// TIA Portal V17 export
// export: Created 2025-03-07T09:17:06.8122535Z, ExportSetting WithDefaults, DisplayName Totally Integrated Automation Portal, DisplayVersion V17 Update 8, DisplayName TIA Portal Openness, DisplayVersion V17 Update 8, DisplayName TIA Portal Version Control Interface, DisplayVersion V17, DisplayName SINAMICS Startdrive Advanced, DisplayVersion V17 SP2, DisplayName SINAMICS Startdrive G110M, G120, G120C, G120D, G120P, G115D, DisplayVersion V17 SP2, DisplayName SINAMICS Startdrive G130, G150, S120, S150, SINAMICS MV, S210, DisplayVersion V17 SP2, DisplayName STEP 7 Professional, DisplayVersion V17 Update 8, DisplayName SINUMERIK ONE STEP 7 Toolbox, DisplayVersion V17 Update 12, DisplayName SINUMERIK 840D sl STEP 7 Toolbox, DisplayVersion V17 Update 12, DisplayName STEP 7 Safety, DisplayVersion V17 Update 6, DisplayName WinCC Advanced, DisplayVersion V17 Update 8
FUNCTION "FC8002_UNIT_01_CLADDING" : Void   // FC8002, LAD
{ S7_Optimized_Access := 'FALSE' }
AUTHOR : ETXETAR
VERSION : 1.0
// stored: AutoNumber false, IsIECCheckEnabled false, SetENOAutomatically false, UDAEnableTagReadback false
   VAR_TEMP
      ZERO : Byte;   // ZERO
      STATUS_BLKMOV : Int;   // STATUS BLKMOV
      STATUS_FILL : Int;   // STATUS FILL
      aux_string : String;
      Cnt_Chars : Int;
      Chars_Array : Array[0..63] of Char;
   END_VAR
   VAR CONSTANT
      FC_NUMBER : DInt := 8002;   // FC NUMBER
   END_VAR
   VAR_TEMP   // added for the SCL form of the ladder/FBD networks
      _w1 : Bool;
      _w2 : Bool;
      _w3 : Bool;
      _w4 : Bool;
      _w5 : Bool;
      _w6 : Bool;
      _w7 : Bool;
      _w8 : Bool;
      _w9 : Bool;
   END_VAR
BEGIN

REGION Network 1: ZERO
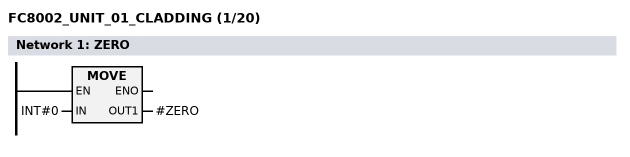
   RUNG wire#powerrail
      { S7_GenerateENO := "TRUE" } Move(in := INT#0, out1 => #ZERO)
   END_RUNG
   // the same network as SCL:
   #ZERO := INT#0;
END_REGION

REGION Network 2: HMI MANUAL PART A FIXTURE 1, 2, 3, 4 STATUS
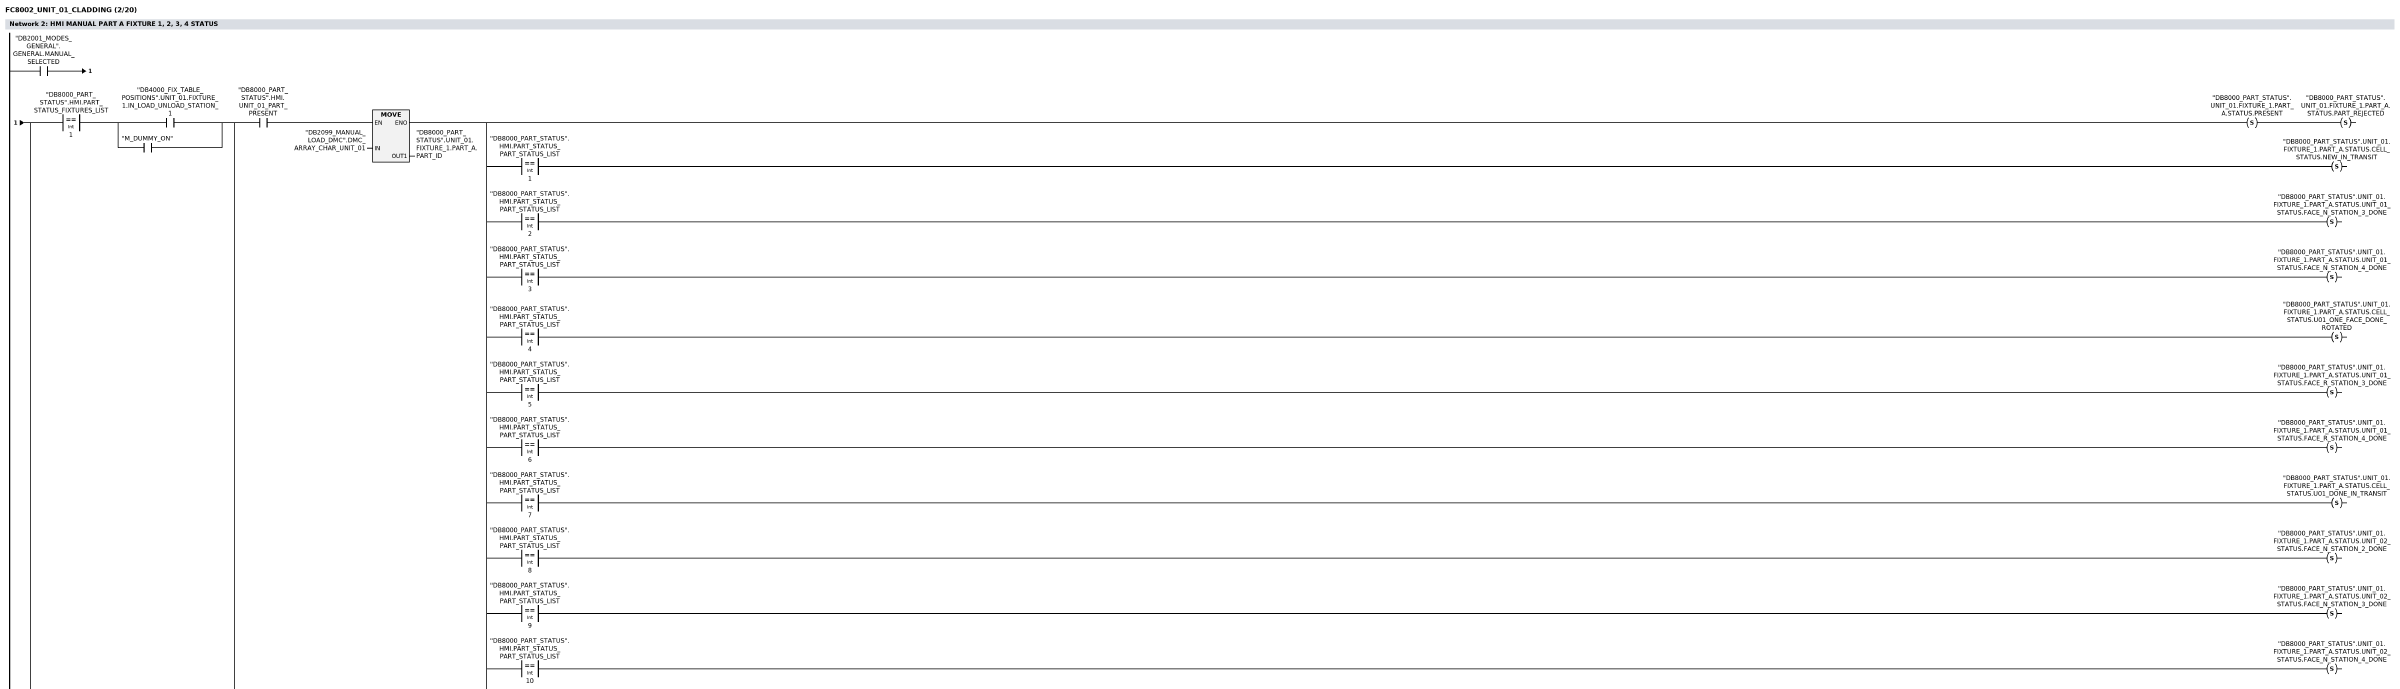
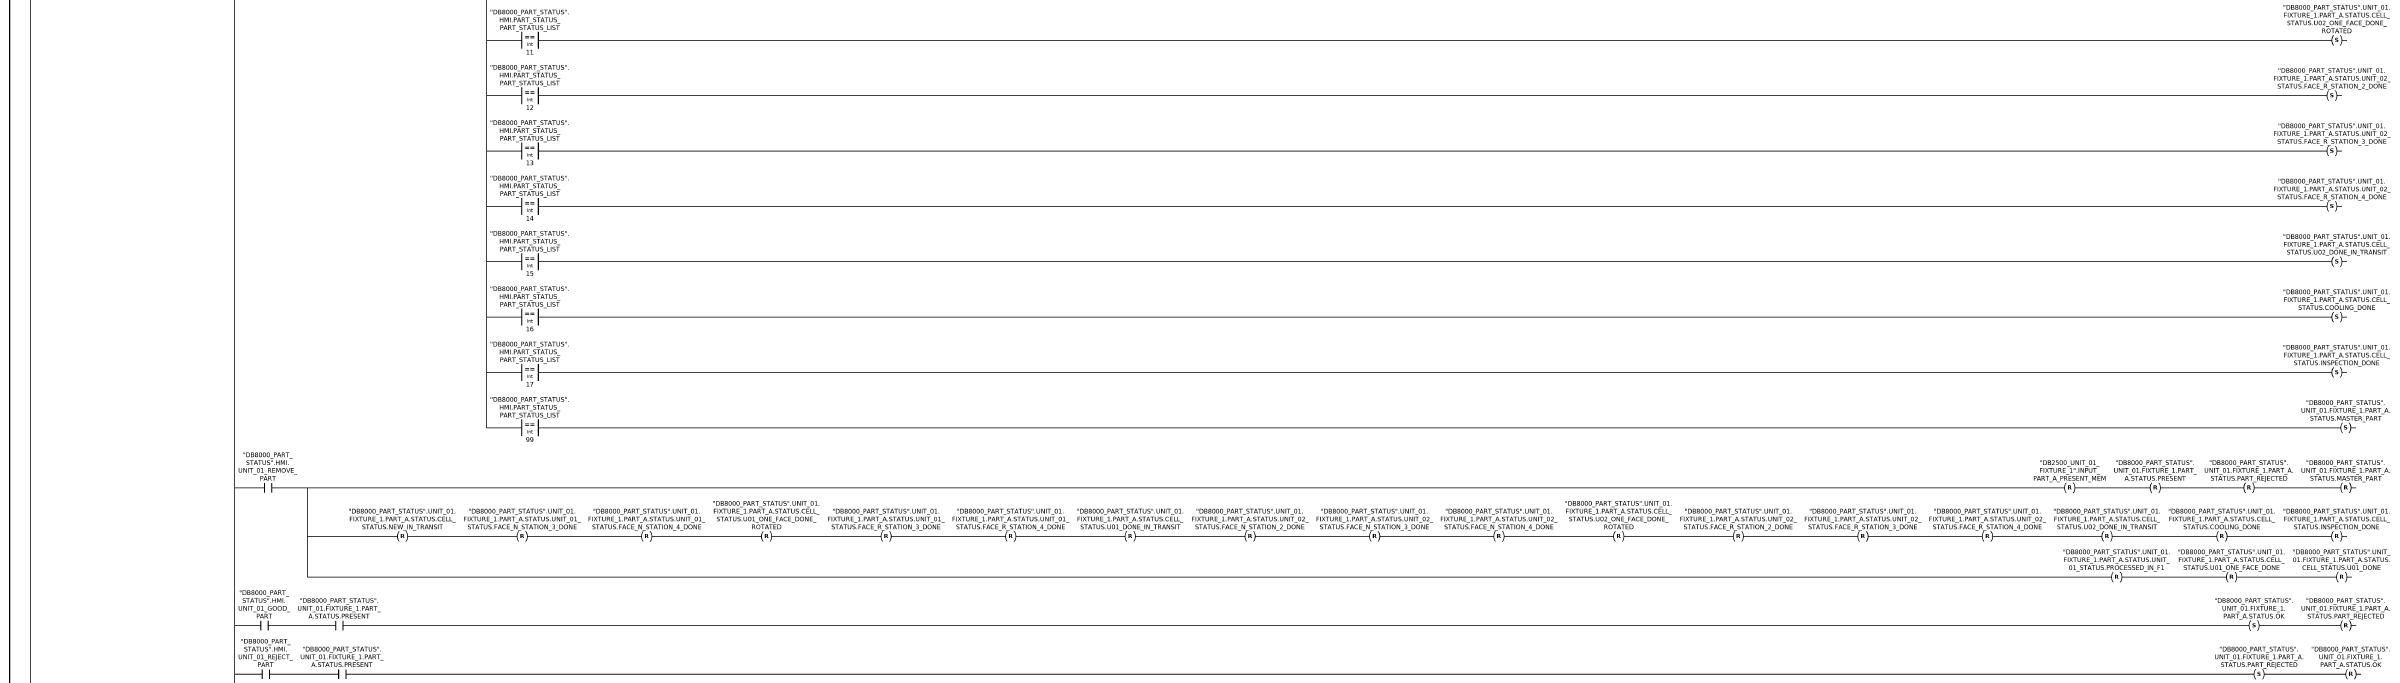
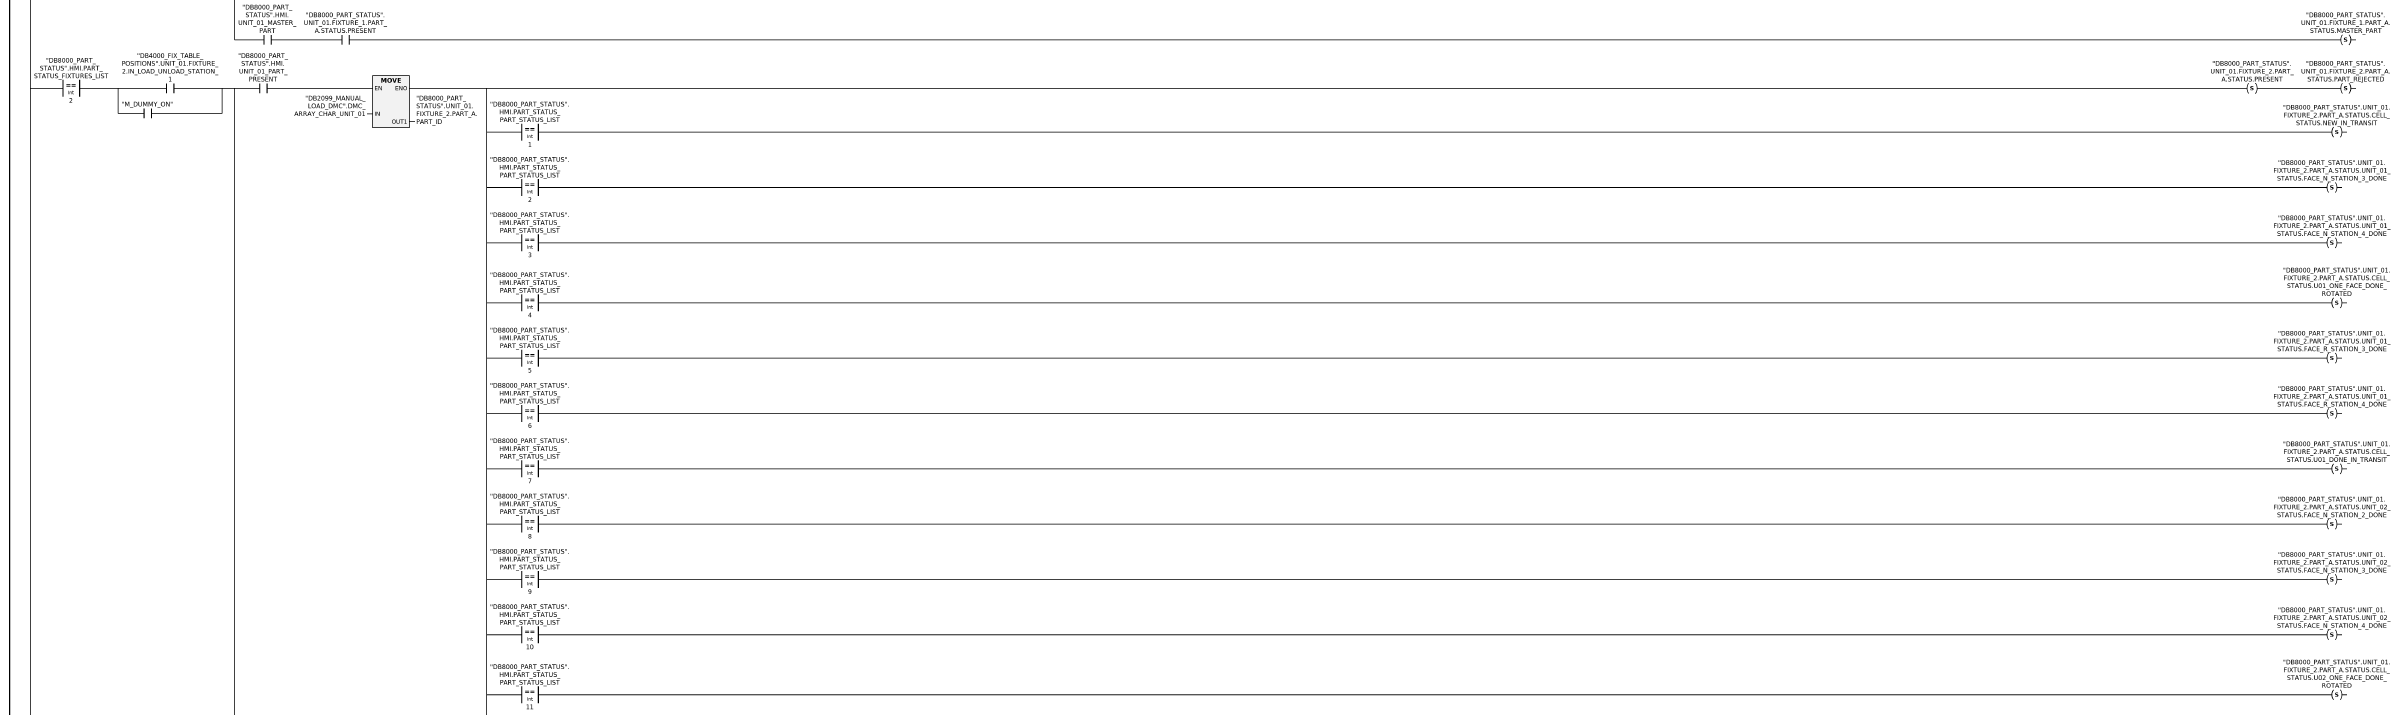
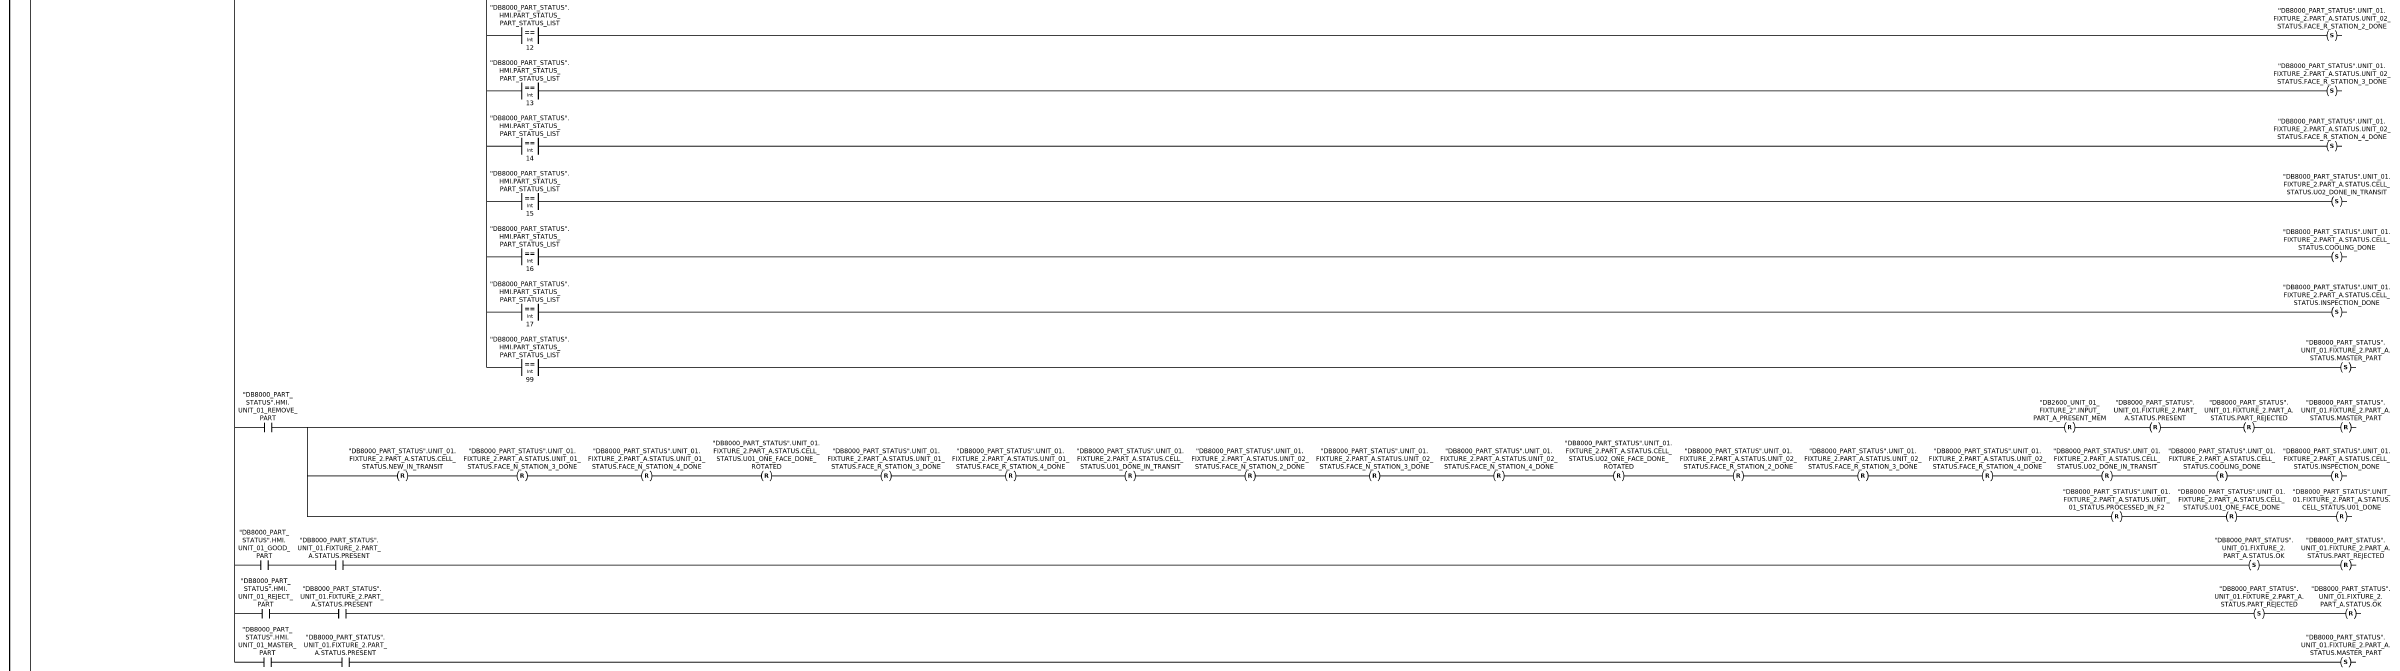
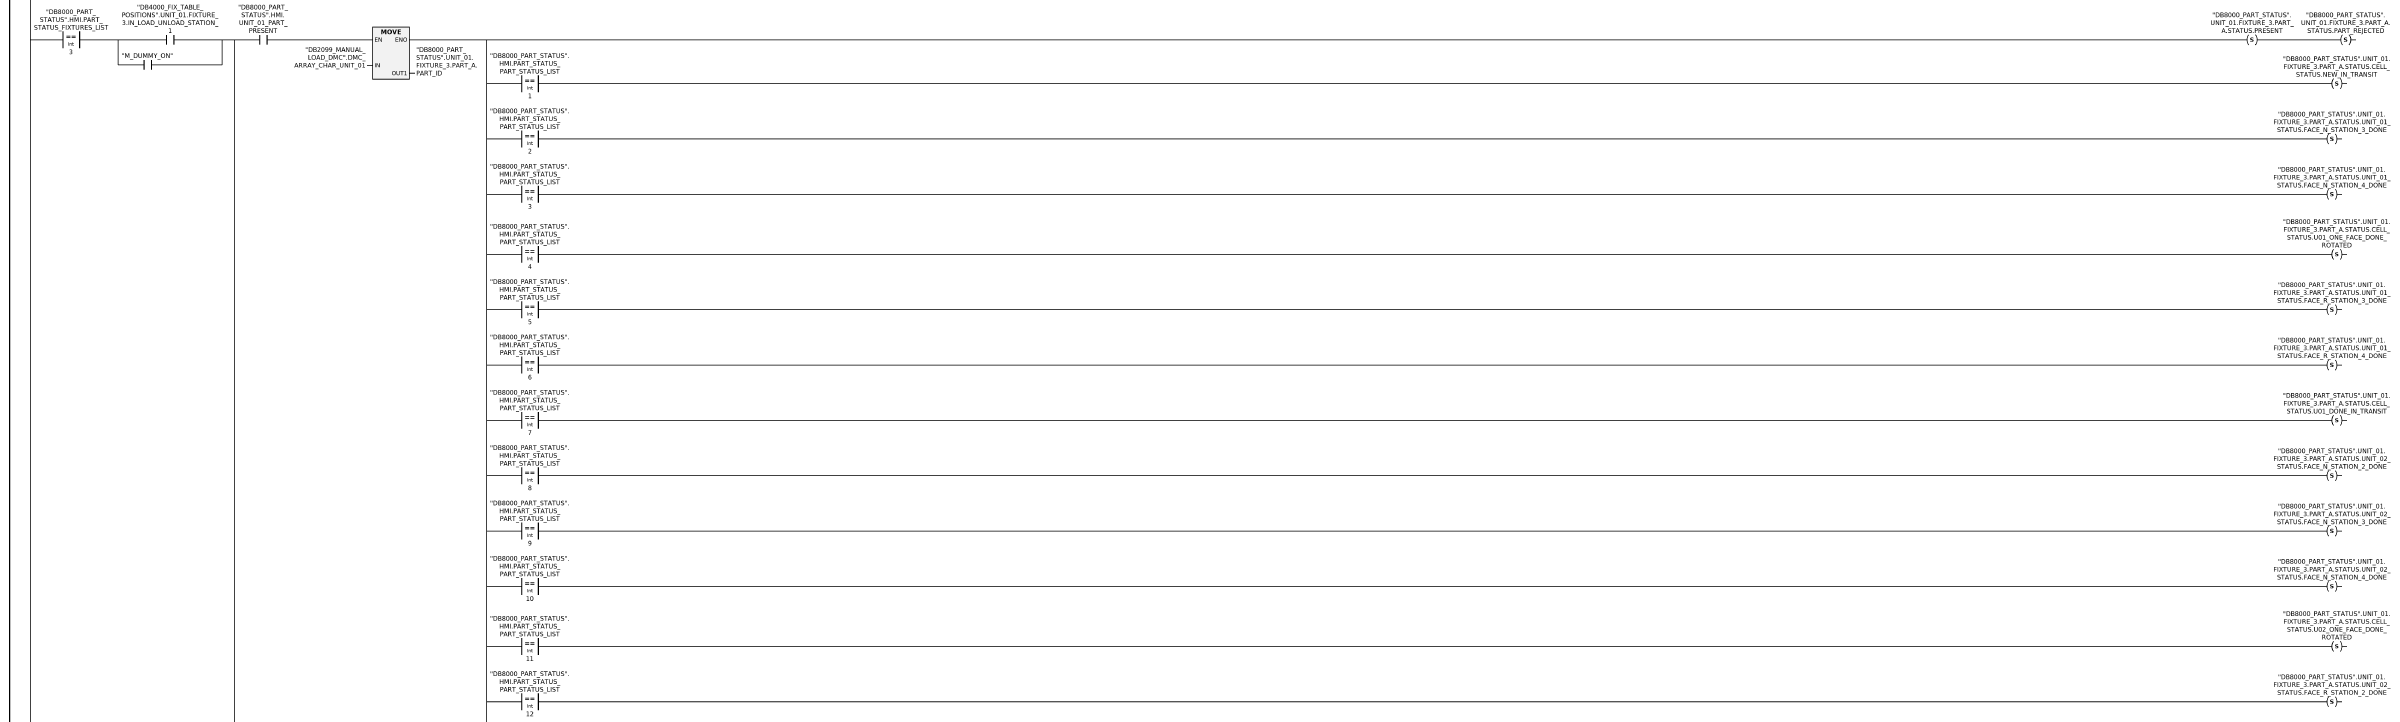
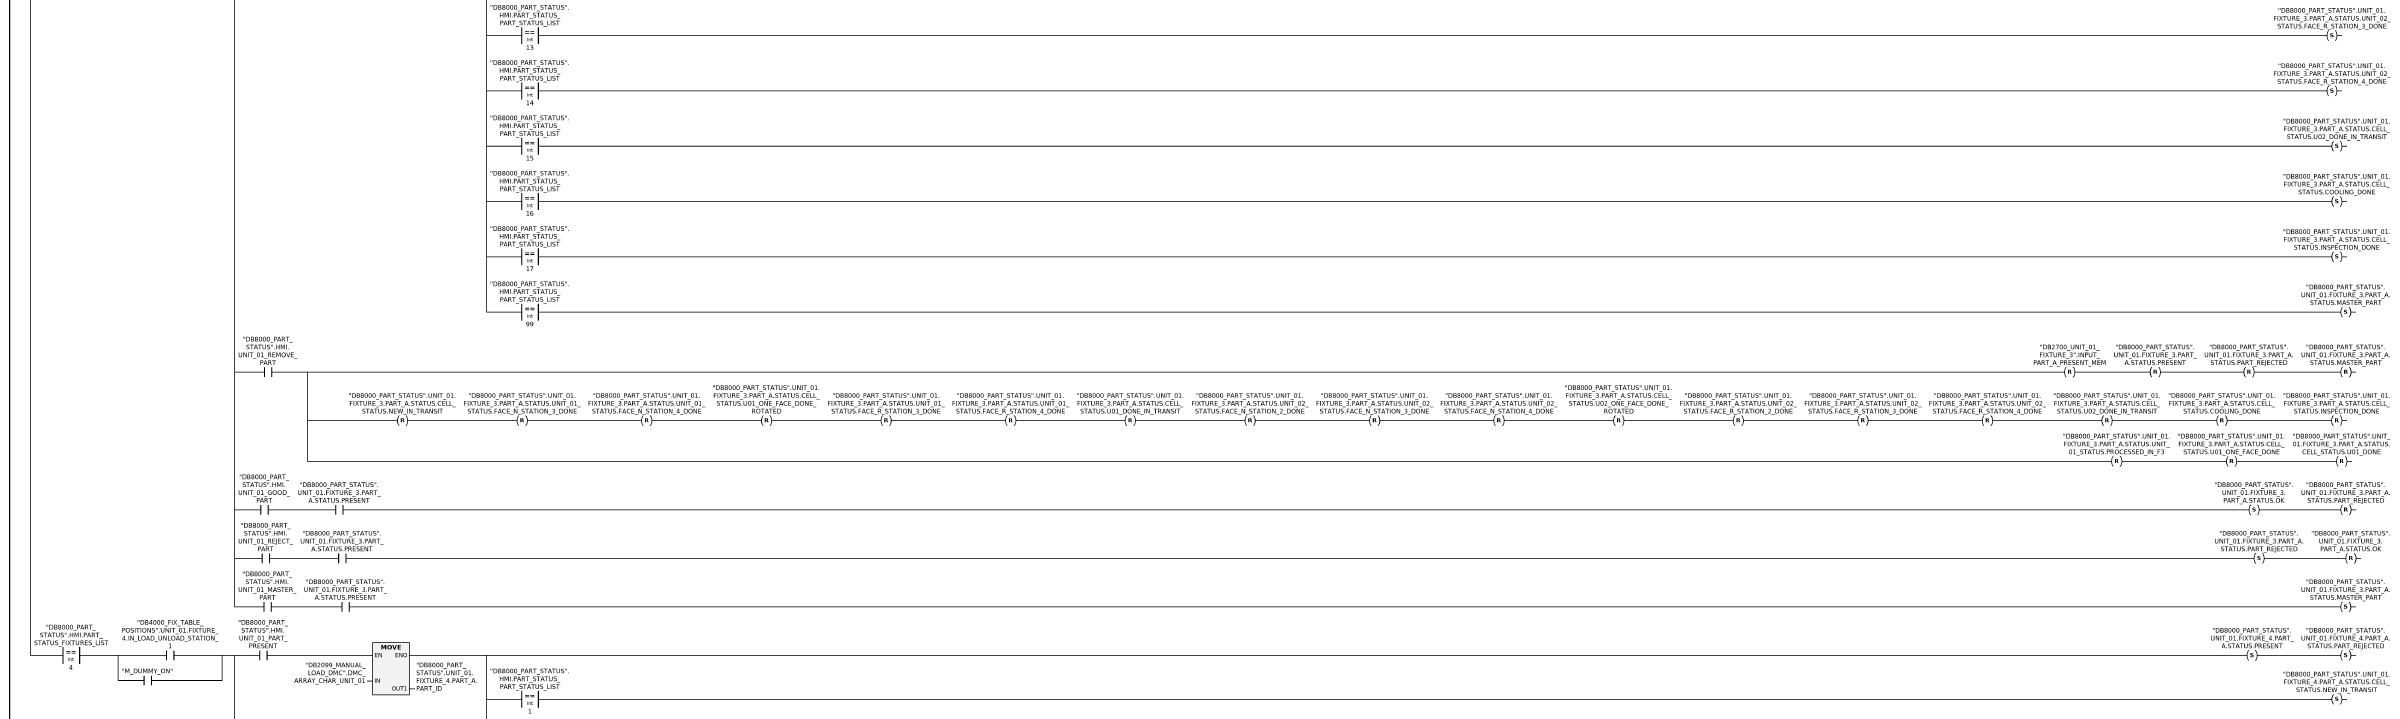
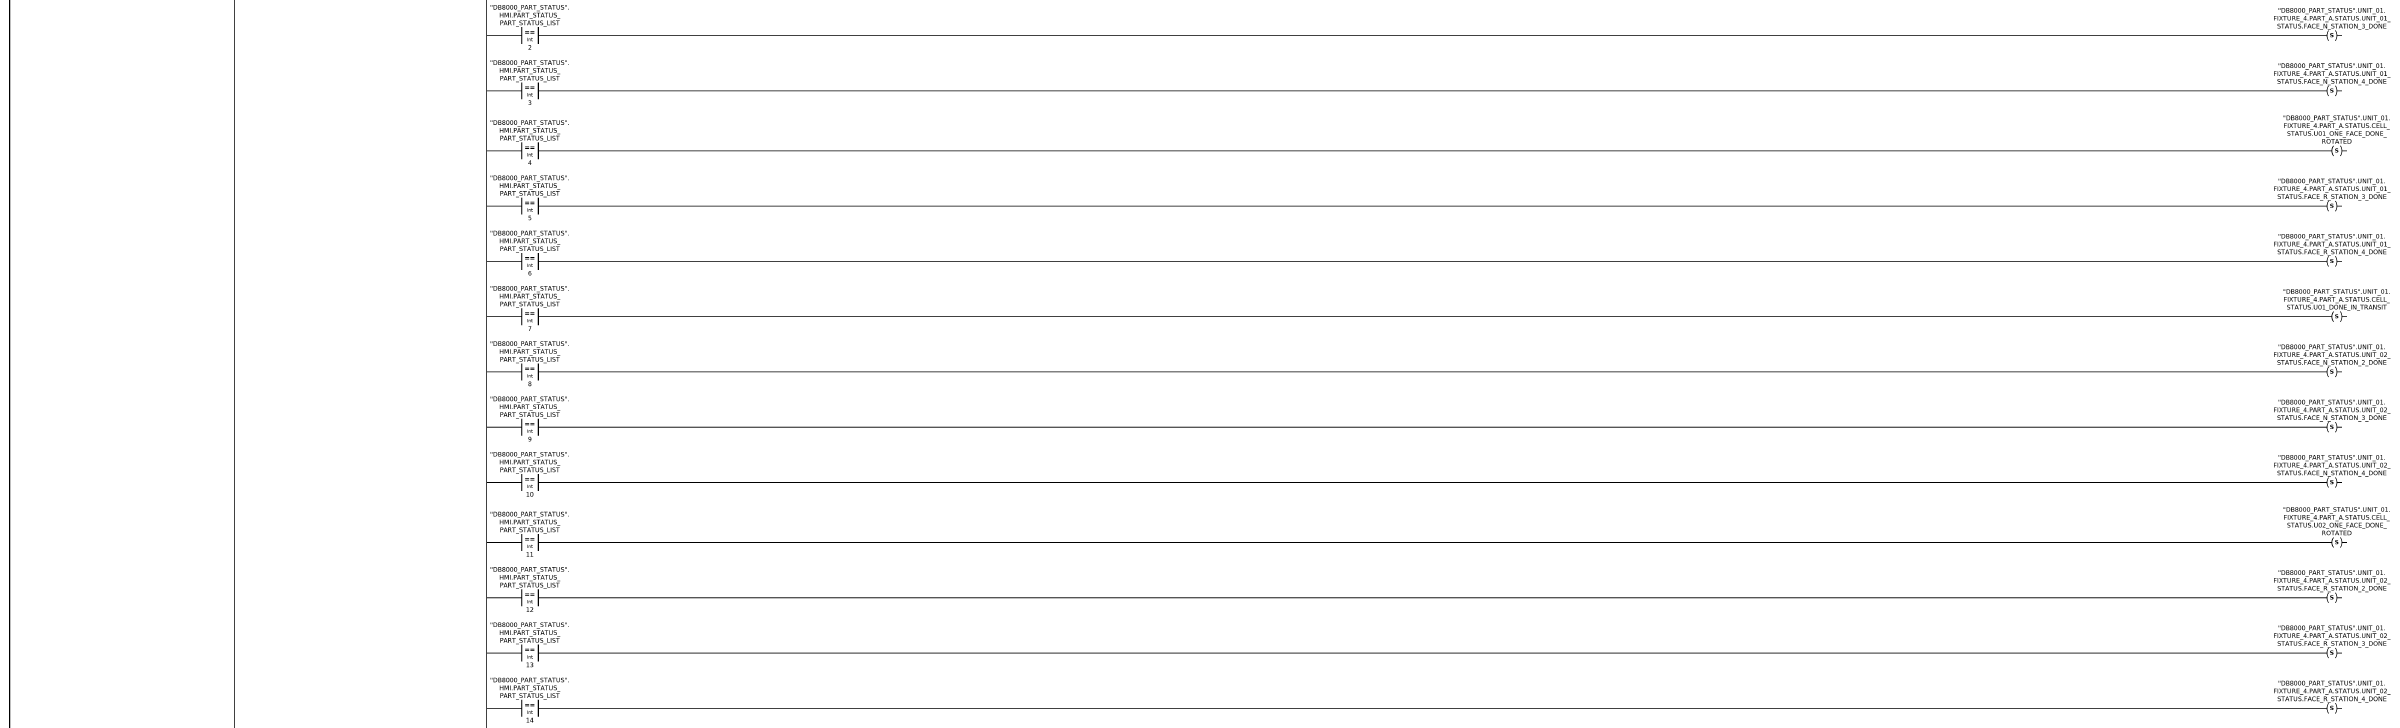
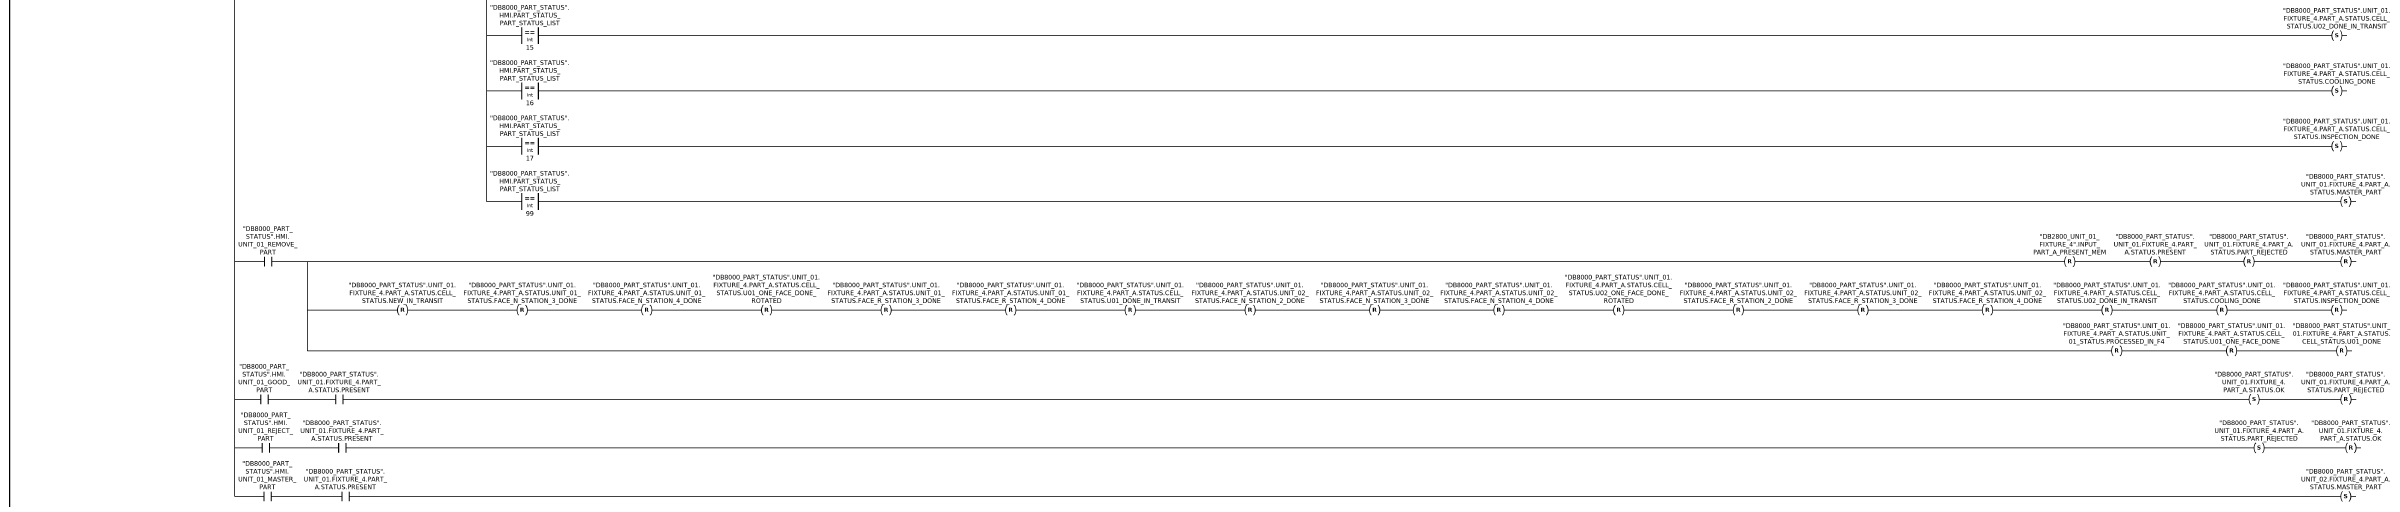
   RUNG wire#powerrail
      Contact( "DB2001_MODES_GENERAL".GENERAL.MANUAL_SELECTED )
      wire#w1
      { S7_Templates := "SrcType := Int" } EQ_Contact(in1 := "DB8000_PART_STATUS".HMI.PART_STATUS_FIXTURES_LIST, in2 := 1)
      wire#w2
      Contact( "DB4000_FIX_TABLE_POSITIONS".UNIT_01.FIXTURE_1.IN_LOAD_UNLOAD_STATION_1 )
      wire#w3
      Contact( "DB8000_PART_STATUS".HMI.UNIT_01_PART_PRESENT )
      Move(in := "DB2099_MANUAL_LOAD_DMC".DMC_ARRAY_CHAR_UNIT_01, out1 => "DB8000_PART_STATUS".UNIT_01.FIXTURE_1.PART_A.PART_ID)
      wire#w4
      S_Coil( "DB8000_PART_STATUS".UNIT_01.FIXTURE_1.PART_A.STATUS.PRESENT )
      S_Coil( "DB8000_PART_STATUS".UNIT_01.FIXTURE_1.PART_A.STATUS.PART_REJECTED )
   END_RUNG
   RUNG wire#w2
      Contact( "M_DUMMY_ON" )
   END_RUNG wire#w3
   RUNG wire#w4
      { S7_Templates := "SrcType := Int" } EQ_Contact(in1 := "DB8000_PART_STATUS".HMI.PART_STATUS_PART_STATUS_LIST, in2 := 1)
      S_Coil( "DB8000_PART_STATUS".UNIT_01.FIXTURE_1.PART_A.STATUS.CELL_STATUS.NEW_IN_TRANSIT )
   END_RUNG
   RUNG wire#w4
      { S7_Templates := "SrcType := Int" } EQ_Contact(in1 := "DB8000_PART_STATUS".HMI.PART_STATUS_PART_STATUS_LIST, in2 := 2)
      S_Coil( "DB8000_PART_STATUS".UNIT_01.FIXTURE_1.PART_A.STATUS.UNIT_01_STATUS.FACE_N_STATION_3_DONE )
   END_RUNG
   RUNG wire#w4
      { S7_Templates := "SrcType := Int" } EQ_Contact(in1 := "DB8000_PART_STATUS".HMI.PART_STATUS_PART_STATUS_LIST, in2 := 3)
      S_Coil( "DB8000_PART_STATUS".UNIT_01.FIXTURE_1.PART_A.STATUS.UNIT_01_STATUS.FACE_N_STATION_4_DONE )
   END_RUNG
   RUNG wire#w4
      { S7_Templates := "SrcType := Int" } EQ_Contact(in1 := "DB8000_PART_STATUS".HMI.PART_STATUS_PART_STATUS_LIST, in2 := 4)
      S_Coil( "DB8000_PART_STATUS".UNIT_01.FIXTURE_1.PART_A.STATUS.CELL_STATUS.U01_ONE_FACE_DONE_ROTATED )
   END_RUNG
   RUNG wire#w4
      { S7_Templates := "SrcType := Int" } EQ_Contact(in1 := "DB8000_PART_STATUS".HMI.PART_STATUS_PART_STATUS_LIST, in2 := 5)
      S_Coil( "DB8000_PART_STATUS".UNIT_01.FIXTURE_1.PART_A.STATUS.UNIT_01_STATUS.FACE_R_STATION_3_DONE )
   END_RUNG
   RUNG wire#w4
      { S7_Templates := "SrcType := Int" } EQ_Contact(in1 := "DB8000_PART_STATUS".HMI.PART_STATUS_PART_STATUS_LIST, in2 := 6)
      S_Coil( "DB8000_PART_STATUS".UNIT_01.FIXTURE_1.PART_A.STATUS.UNIT_01_STATUS.FACE_R_STATION_4_DONE )
   END_RUNG
   RUNG wire#w4
      { S7_Templates := "SrcType := Int" } EQ_Contact(in1 := "DB8000_PART_STATUS".HMI.PART_STATUS_PART_STATUS_LIST, in2 := 7)
      S_Coil( "DB8000_PART_STATUS".UNIT_01.FIXTURE_1.PART_A.STATUS.CELL_STATUS.U01_DONE_IN_TRANSIT )
   END_RUNG
   RUNG wire#w4
      { S7_Templates := "SrcType := Int" } EQ_Contact(in1 := "DB8000_PART_STATUS".HMI.PART_STATUS_PART_STATUS_LIST, in2 := 8)
      S_Coil( "DB8000_PART_STATUS".UNIT_01.FIXTURE_1.PART_A.STATUS.UNIT_02_STATUS.FACE_N_STATION_2_DONE )
   END_RUNG
   RUNG wire#w4
      { S7_Templates := "SrcType := Int" } EQ_Contact(in1 := "DB8000_PART_STATUS".HMI.PART_STATUS_PART_STATUS_LIST, in2 := 9)
      S_Coil( "DB8000_PART_STATUS".UNIT_01.FIXTURE_1.PART_A.STATUS.UNIT_02_STATUS.FACE_N_STATION_3_DONE )
   END_RUNG
   RUNG wire#w4
      { S7_Templates := "SrcType := Int" } EQ_Contact(in1 := "DB8000_PART_STATUS".HMI.PART_STATUS_PART_STATUS_LIST, in2 := 10)
      S_Coil( "DB8000_PART_STATUS".UNIT_01.FIXTURE_1.PART_A.STATUS.UNIT_02_STATUS.FACE_N_STATION_4_DONE )
   END_RUNG
   RUNG wire#w4
      { S7_Templates := "SrcType := Int" } EQ_Contact(in1 := "DB8000_PART_STATUS".HMI.PART_STATUS_PART_STATUS_LIST, in2 := 11)
      S_Coil( "DB8000_PART_STATUS".UNIT_01.FIXTURE_1.PART_A.STATUS.CELL_STATUS.U02_ONE_FACE_DONE_ROTATED )
   END_RUNG
   RUNG wire#w4
      { S7_Templates := "SrcType := Int" } EQ_Contact(in1 := "DB8000_PART_STATUS".HMI.PART_STATUS_PART_STATUS_LIST, in2 := 12)
      S_Coil( "DB8000_PART_STATUS".UNIT_01.FIXTURE_1.PART_A.STATUS.UNIT_02_STATUS.FACE_R_STATION_2_DONE )
   END_RUNG
   RUNG wire#w4
      { S7_Templates := "SrcType := Int" } EQ_Contact(in1 := "DB8000_PART_STATUS".HMI.PART_STATUS_PART_STATUS_LIST, in2 := 13)
      S_Coil( "DB8000_PART_STATUS".UNIT_01.FIXTURE_1.PART_A.STATUS.UNIT_02_STATUS.FACE_R_STATION_3_DONE )
   END_RUNG
   RUNG wire#w4
      { S7_Templates := "SrcType := Int" } EQ_Contact(in1 := "DB8000_PART_STATUS".HMI.PART_STATUS_PART_STATUS_LIST, in2 := 14)
      S_Coil( "DB8000_PART_STATUS".UNIT_01.FIXTURE_1.PART_A.STATUS.UNIT_02_STATUS.FACE_R_STATION_4_DONE )
   END_RUNG
   RUNG wire#w4
      { S7_Templates := "SrcType := Int" } EQ_Contact(in1 := "DB8000_PART_STATUS".HMI.PART_STATUS_PART_STATUS_LIST, in2 := 15)
      S_Coil( "DB8000_PART_STATUS".UNIT_01.FIXTURE_1.PART_A.STATUS.CELL_STATUS.U02_DONE_IN_TRANSIT )
   END_RUNG
   RUNG wire#w4
      { S7_Templates := "SrcType := Int" } EQ_Contact(in1 := "DB8000_PART_STATUS".HMI.PART_STATUS_PART_STATUS_LIST, in2 := 16)
      S_Coil( "DB8000_PART_STATUS".UNIT_01.FIXTURE_1.PART_A.STATUS.CELL_STATUS.COOLING_DONE )
   END_RUNG
   RUNG wire#w4
      { S7_Templates := "SrcType := Int" } EQ_Contact(in1 := "DB8000_PART_STATUS".HMI.PART_STATUS_PART_STATUS_LIST, in2 := 17)
      S_Coil( "DB8000_PART_STATUS".UNIT_01.FIXTURE_1.PART_A.STATUS.CELL_STATUS.INSPECTION_DONE )
   END_RUNG
   RUNG wire#w4
      { S7_Templates := "SrcType := Int" } EQ_Contact(in1 := "DB8000_PART_STATUS".HMI.PART_STATUS_PART_STATUS_LIST, in2 := 99)
      S_Coil( "DB8000_PART_STATUS".UNIT_01.FIXTURE_1.PART_A.STATUS.MASTER_PART )
   END_RUNG
   RUNG wire#w3
      Contact( "DB8000_PART_STATUS".HMI.UNIT_01_REMOVE_PART )
      wire#w5
      R_Coil( "DB2500_UNIT_01_FIXTURE_1".INPUT_PART_A_PRESENT_MEM )
      R_Coil( "DB8000_PART_STATUS".UNIT_01.FIXTURE_1.PART_A.STATUS.PRESENT )
      R_Coil( "DB8000_PART_STATUS".UNIT_01.FIXTURE_1.PART_A.STATUS.PART_REJECTED )
      R_Coil( "DB8000_PART_STATUS".UNIT_01.FIXTURE_1.PART_A.STATUS.MASTER_PART )
   END_RUNG
   RUNG wire#w5
      R_Coil( "DB8000_PART_STATUS".UNIT_01.FIXTURE_1.PART_A.STATUS.CELL_STATUS.NEW_IN_TRANSIT )
      R_Coil( "DB8000_PART_STATUS".UNIT_01.FIXTURE_1.PART_A.STATUS.UNIT_01_STATUS.FACE_N_STATION_3_DONE )
      R_Coil( "DB8000_PART_STATUS".UNIT_01.FIXTURE_1.PART_A.STATUS.UNIT_01_STATUS.FACE_N_STATION_4_DONE )
      R_Coil( "DB8000_PART_STATUS".UNIT_01.FIXTURE_1.PART_A.STATUS.CELL_STATUS.U01_ONE_FACE_DONE_ROTATED )
      R_Coil( "DB8000_PART_STATUS".UNIT_01.FIXTURE_1.PART_A.STATUS.UNIT_01_STATUS.FACE_R_STATION_3_DONE )
      R_Coil( "DB8000_PART_STATUS".UNIT_01.FIXTURE_1.PART_A.STATUS.UNIT_01_STATUS.FACE_R_STATION_4_DONE )
      R_Coil( "DB8000_PART_STATUS".UNIT_01.FIXTURE_1.PART_A.STATUS.CELL_STATUS.U01_DONE_IN_TRANSIT )
      R_Coil( "DB8000_PART_STATUS".UNIT_01.FIXTURE_1.PART_A.STATUS.UNIT_02_STATUS.FACE_N_STATION_2_DONE )
      R_Coil( "DB8000_PART_STATUS".UNIT_01.FIXTURE_1.PART_A.STATUS.UNIT_02_STATUS.FACE_N_STATION_3_DONE )
      R_Coil( "DB8000_PART_STATUS".UNIT_01.FIXTURE_1.PART_A.STATUS.UNIT_02_STATUS.FACE_N_STATION_4_DONE )
      R_Coil( "DB8000_PART_STATUS".UNIT_01.FIXTURE_1.PART_A.STATUS.CELL_STATUS.U02_ONE_FACE_DONE_ROTATED )
      R_Coil( "DB8000_PART_STATUS".UNIT_01.FIXTURE_1.PART_A.STATUS.UNIT_02_STATUS.FACE_R_STATION_2_DONE )
      R_Coil( "DB8000_PART_STATUS".UNIT_01.FIXTURE_1.PART_A.STATUS.UNIT_02_STATUS.FACE_R_STATION_3_DONE )
      R_Coil( "DB8000_PART_STATUS".UNIT_01.FIXTURE_1.PART_A.STATUS.UNIT_02_STATUS.FACE_R_STATION_4_DONE )
      R_Coil( "DB8000_PART_STATUS".UNIT_01.FIXTURE_1.PART_A.STATUS.CELL_STATUS.U02_DONE_IN_TRANSIT )
      R_Coil( "DB8000_PART_STATUS".UNIT_01.FIXTURE_1.PART_A.STATUS.CELL_STATUS.COOLING_DONE )
      R_Coil( "DB8000_PART_STATUS".UNIT_01.FIXTURE_1.PART_A.STATUS.CELL_STATUS.INSPECTION_DONE )
   END_RUNG
   RUNG wire#w5
      R_Coil( "DB8000_PART_STATUS".UNIT_01.FIXTURE_1.PART_A.STATUS.UNIT_01_STATUS.PROCESSED_IN_F1 )
      R_Coil( "DB8000_PART_STATUS".UNIT_01.FIXTURE_1.PART_A.STATUS.CELL_STATUS.U01_ONE_FACE_DONE )
      R_Coil( "DB8000_PART_STATUS".UNIT_01.FIXTURE_1.PART_A.STATUS.CELL_STATUS.U01_DONE )
   END_RUNG
   RUNG wire#w3
      Contact( "DB8000_PART_STATUS".HMI.UNIT_01_GOOD_PART )
      Contact( "DB8000_PART_STATUS".UNIT_01.FIXTURE_1.PART_A.STATUS.PRESENT )
      S_Coil( "DB8000_PART_STATUS".UNIT_01.FIXTURE_1.PART_A.STATUS.OK )
      R_Coil( "DB8000_PART_STATUS".UNIT_01.FIXTURE_1.PART_A.STATUS.PART_REJECTED )
   END_RUNG
   RUNG wire#w3
      Contact( "DB8000_PART_STATUS".HMI.UNIT_01_REJECT_PART )
      Contact( "DB8000_PART_STATUS".UNIT_01.FIXTURE_1.PART_A.STATUS.PRESENT )
      S_Coil( "DB8000_PART_STATUS".UNIT_01.FIXTURE_1.PART_A.STATUS.PART_REJECTED )
      R_Coil( "DB8000_PART_STATUS".UNIT_01.FIXTURE_1.PART_A.STATUS.OK )
   END_RUNG
   RUNG wire#w3
      Contact( "DB8000_PART_STATUS".HMI.UNIT_01_MASTER_PART )
      Contact( "DB8000_PART_STATUS".UNIT_01.FIXTURE_1.PART_A.STATUS.PRESENT )
      S_Coil( "DB8000_PART_STATUS".UNIT_01.FIXTURE_1.PART_A.STATUS.MASTER_PART )
   END_RUNG
   RUNG wire#w1
      { S7_Templates := "SrcType := Int" } EQ_Contact(in1 := "DB8000_PART_STATUS".HMI.PART_STATUS_FIXTURES_LIST, in2 := 2)
      wire#w6
      Contact( "DB4000_FIX_TABLE_POSITIONS".UNIT_01.FIXTURE_2.IN_LOAD_UNLOAD_STATION_1 )
      wire#w7
      Contact( "DB8000_PART_STATUS".HMI.UNIT_01_PART_PRESENT )
      Move(in := "DB2099_MANUAL_LOAD_DMC".DMC_ARRAY_CHAR_UNIT_01, out1 => "DB8000_PART_STATUS".UNIT_01.FIXTURE_2.PART_A.PART_ID)
      wire#w8
      S_Coil( "DB8000_PART_STATUS".UNIT_01.FIXTURE_2.PART_A.STATUS.PRESENT )
      S_Coil( "DB8000_PART_STATUS".UNIT_01.FIXTURE_2.PART_A.STATUS.PART_REJECTED )
   END_RUNG
   RUNG wire#w6
      Contact( "M_DUMMY_ON" )
   END_RUNG wire#w7
   RUNG wire#w8
      { S7_Templates := "SrcType := Int" } EQ_Contact(in1 := "DB8000_PART_STATUS".HMI.PART_STATUS_PART_STATUS_LIST, in2 := 1)
      S_Coil( "DB8000_PART_STATUS".UNIT_01.FIXTURE_2.PART_A.STATUS.CELL_STATUS.NEW_IN_TRANSIT )
   END_RUNG
   RUNG wire#w8
      { S7_Templates := "SrcType := Int" } EQ_Contact(in1 := "DB8000_PART_STATUS".HMI.PART_STATUS_PART_STATUS_LIST, in2 := 2)
      S_Coil( "DB8000_PART_STATUS".UNIT_01.FIXTURE_2.PART_A.STATUS.UNIT_01_STATUS.FACE_N_STATION_3_DONE )
   END_RUNG
   RUNG wire#w8
      { S7_Templates := "SrcType := Int" } EQ_Contact(in1 := "DB8000_PART_STATUS".HMI.PART_STATUS_PART_STATUS_LIST, in2 := 3)
      S_Coil( "DB8000_PART_STATUS".UNIT_01.FIXTURE_2.PART_A.STATUS.UNIT_01_STATUS.FACE_N_STATION_4_DONE )
   END_RUNG
   RUNG wire#w8
      { S7_Templates := "SrcType := Int" } EQ_Contact(in1 := "DB8000_PART_STATUS".HMI.PART_STATUS_PART_STATUS_LIST, in2 := 4)
      S_Coil( "DB8000_PART_STATUS".UNIT_01.FIXTURE_2.PART_A.STATUS.CELL_STATUS.U01_ONE_FACE_DONE_ROTATED )
   END_RUNG
   RUNG wire#w8
      { S7_Templates := "SrcType := Int" } EQ_Contact(in1 := "DB8000_PART_STATUS".HMI.PART_STATUS_PART_STATUS_LIST, in2 := 5)
      S_Coil( "DB8000_PART_STATUS".UNIT_01.FIXTURE_2.PART_A.STATUS.UNIT_01_STATUS.FACE_R_STATION_3_DONE )
   END_RUNG
   RUNG wire#w8
      { S7_Templates := "SrcType := Int" } EQ_Contact(in1 := "DB8000_PART_STATUS".HMI.PART_STATUS_PART_STATUS_LIST, in2 := 6)
      S_Coil( "DB8000_PART_STATUS".UNIT_01.FIXTURE_2.PART_A.STATUS.UNIT_01_STATUS.FACE_R_STATION_4_DONE )
   END_RUNG
   RUNG wire#w8
      { S7_Templates := "SrcType := Int" } EQ_Contact(in1 := "DB8000_PART_STATUS".HMI.PART_STATUS_PART_STATUS_LIST, in2 := 7)
      S_Coil( "DB8000_PART_STATUS".UNIT_01.FIXTURE_2.PART_A.STATUS.CELL_STATUS.U01_DONE_IN_TRANSIT )
   END_RUNG
   RUNG wire#w8
      { S7_Templates := "SrcType := Int" } EQ_Contact(in1 := "DB8000_PART_STATUS".HMI.PART_STATUS_PART_STATUS_LIST, in2 := 8)
      S_Coil( "DB8000_PART_STATUS".UNIT_01.FIXTURE_2.PART_A.STATUS.UNIT_02_STATUS.FACE_N_STATION_2_DONE )
   END_RUNG
   RUNG wire#w8
      { S7_Templates := "SrcType := Int" } EQ_Contact(in1 := "DB8000_PART_STATUS".HMI.PART_STATUS_PART_STATUS_LIST, in2 := 9)
      S_Coil( "DB8000_PART_STATUS".UNIT_01.FIXTURE_2.PART_A.STATUS.UNIT_02_STATUS.FACE_N_STATION_3_DONE )
   END_RUNG
   RUNG wire#w8
      { S7_Templates := "SrcType := Int" } EQ_Contact(in1 := "DB8000_PART_STATUS".HMI.PART_STATUS_PART_STATUS_LIST, in2 := 10)
      S_Coil( "DB8000_PART_STATUS".UNIT_01.FIXTURE_2.PART_A.STATUS.UNIT_02_STATUS.FACE_N_STATION_4_DONE )
   END_RUNG
   RUNG wire#w8
      { S7_Templates := "SrcType := Int" } EQ_Contact(in1 := "DB8000_PART_STATUS".HMI.PART_STATUS_PART_STATUS_LIST, in2 := 11)
      S_Coil( "DB8000_PART_STATUS".UNIT_01.FIXTURE_2.PART_A.STATUS.CELL_STATUS.U02_ONE_FACE_DONE_ROTATED )
   END_RUNG
   RUNG wire#w8
      { S7_Templates := "SrcType := Int" } EQ_Contact(in1 := "DB8000_PART_STATUS".HMI.PART_STATUS_PART_STATUS_LIST, in2 := 12)
      S_Coil( "DB8000_PART_STATUS".UNIT_01.FIXTURE_2.PART_A.STATUS.UNIT_02_STATUS.FACE_R_STATION_2_DONE )
   END_RUNG
   RUNG wire#w8
      { S7_Templates := "SrcType := Int" } EQ_Contact(in1 := "DB8000_PART_STATUS".HMI.PART_STATUS_PART_STATUS_LIST, in2 := 13)
      S_Coil( "DB8000_PART_STATUS".UNIT_01.FIXTURE_2.PART_A.STATUS.UNIT_02_STATUS.FACE_R_STATION_3_DONE )
   END_RUNG
   RUNG wire#w8
      { S7_Templates := "SrcType := Int" } EQ_Contact(in1 := "DB8000_PART_STATUS".HMI.PART_STATUS_PART_STATUS_LIST, in2 := 14)
      S_Coil( "DB8000_PART_STATUS".UNIT_01.FIXTURE_2.PART_A.STATUS.UNIT_02_STATUS.FACE_R_STATION_4_DONE )
   END_RUNG
   RUNG wire#w8
      { S7_Templates := "SrcType := Int" } EQ_Contact(in1 := "DB8000_PART_STATUS".HMI.PART_STATUS_PART_STATUS_LIST, in2 := 15)
      S_Coil( "DB8000_PART_STATUS".UNIT_01.FIXTURE_2.PART_A.STATUS.CELL_STATUS.U02_DONE_IN_TRANSIT )
   END_RUNG
   RUNG wire#w8
      { S7_Templates := "SrcType := Int" } EQ_Contact(in1 := "DB8000_PART_STATUS".HMI.PART_STATUS_PART_STATUS_LIST, in2 := 16)
      S_Coil( "DB8000_PART_STATUS".UNIT_01.FIXTURE_2.PART_A.STATUS.CELL_STATUS.COOLING_DONE )
   END_RUNG
   RUNG wire#w8
      { S7_Templates := "SrcType := Int" } EQ_Contact(in1 := "DB8000_PART_STATUS".HMI.PART_STATUS_PART_STATUS_LIST, in2 := 17)
      S_Coil( "DB8000_PART_STATUS".UNIT_01.FIXTURE_2.PART_A.STATUS.CELL_STATUS.INSPECTION_DONE )
   END_RUNG
   RUNG wire#w8
      { S7_Templates := "SrcType := Int" } EQ_Contact(in1 := "DB8000_PART_STATUS".HMI.PART_STATUS_PART_STATUS_LIST, in2 := 99)
      S_Coil( "DB8000_PART_STATUS".UNIT_01.FIXTURE_2.PART_A.STATUS.MASTER_PART )
   END_RUNG
   RUNG wire#w7
      Contact( "DB8000_PART_STATUS".HMI.UNIT_01_REMOVE_PART )
      wire#w9
      R_Coil( "DB2600_UNIT_01_FIXTURE_2".INPUT_PART_A_PRESENT_MEM )
      R_Coil( "DB8000_PART_STATUS".UNIT_01.FIXTURE_2.PART_A.STATUS.PRESENT )
      R_Coil( "DB8000_PART_STATUS".UNIT_01.FIXTURE_2.PART_A.STATUS.PART_REJECTED )
      R_Coil( "DB8000_PART_STATUS".UNIT_01.FIXTURE_2.PART_A.STATUS.MASTER_PART )
   END_RUNG
   RUNG wire#w9
      R_Coil( "DB8000_PART_STATUS".UNIT_01.FIXTURE_2.PART_A.STATUS.CELL_STATUS.NEW_IN_TRANSIT )
      R_Coil( "DB8000_PART_STATUS".UNIT_01.FIXTURE_2.PART_A.STATUS.UNIT_01_STATUS.FACE_N_STATION_3_DONE )
      R_Coil( "DB8000_PART_STATUS".UNIT_01.FIXTURE_2.PART_A.STATUS.UNIT_01_STATUS.FACE_N_STATION_4_DONE )
      R_Coil( "DB8000_PART_STATUS".UNIT_01.FIXTURE_2.PART_A.STATUS.CELL_STATUS.U01_ONE_FACE_DONE_ROTATED )
      R_Coil( "DB8000_PART_STATUS".UNIT_01.FIXTURE_2.PART_A.STATUS.UNIT_01_STATUS.FACE_R_STATION_3_DONE )
      R_Coil( "DB8000_PART_STATUS".UNIT_01.FIXTURE_2.PART_A.STATUS.UNIT_01_STATUS.FACE_R_STATION_4_DONE )
      R_Coil( "DB8000_PART_STATUS".UNIT_01.FIXTURE_2.PART_A.STATUS.CELL_STATUS.U01_DONE_IN_TRANSIT )
      R_Coil( "DB8000_PART_STATUS".UNIT_01.FIXTURE_2.PART_A.STATUS.UNIT_02_STATUS.FACE_N_STATION_2_DONE )
      R_Coil( "DB8000_PART_STATUS".UNIT_01.FIXTURE_2.PART_A.STATUS.UNIT_02_STATUS.FACE_N_STATION_3_DONE )
      R_Coil( "DB8000_PART_STATUS".UNIT_01.FIXTURE_2.PART_A.STATUS.UNIT_02_STATUS.FACE_N_STATION_4_DONE )
      R_Coil( "DB8000_PART_STATUS".UNIT_01.FIXTURE_2.PART_A.STATUS.CELL_STATUS.U02_ONE_FACE_DONE_ROTATED )
      R_Coil( "DB8000_PART_STATUS".UNIT_01.FIXTURE_2.PART_A.STATUS.UNIT_02_STATUS.FACE_R_STATION_2_DONE )
      R_Coil( "DB8000_PART_STATUS".UNIT_01.FIXTURE_2.PART_A.STATUS.UNIT_02_STATUS.FACE_R_STATION_3_DONE )
      R_Coil( "DB8000_PART_STATUS".UNIT_01.FIXTURE_2.PART_A.STATUS.UNIT_02_STATUS.FACE_R_STATION_4_DONE )
      R_Coil( "DB8000_PART_STATUS".UNIT_01.FIXTURE_2.PART_A.STATUS.CELL_STATUS.U02_DONE_IN_TRANSIT )
      R_Coil( "DB8000_PART_STATUS".UNIT_01.FIXTURE_2.PART_A.STATUS.CELL_STATUS.COOLING_DONE )
      R_Coil( "DB8000_PART_STATUS".UNIT_01.FIXTURE_2.PART_A.STATUS.CELL_STATUS.INSPECTION_DONE )
   END_RUNG
   RUNG wire#w9
      R_Coil( "DB8000_PART_STATUS".UNIT_01.FIXTURE_2.PART_A.STATUS.UNIT_01_STATUS.PROCESSED_IN_F2 )
      R_Coil( "DB8000_PART_STATUS".UNIT_01.FIXTURE_2.PART_A.STATUS.CELL_STATUS.U01_ONE_FACE_DONE )
      R_Coil( "DB8000_PART_STATUS".UNIT_01.FIXTURE_2.PART_A.STATUS.CELL_STATUS.U01_DONE )
   END_RUNG
   RUNG wire#w7
      Contact( "DB8000_PART_STATUS".HMI.UNIT_01_GOOD_PART )
      Contact( "DB8000_PART_STATUS".UNIT_01.FIXTURE_2.PART_A.STATUS.PRESENT )
      S_Coil( "DB8000_PART_STATUS".UNIT_01.FIXTURE_2.PART_A.STATUS.OK )
      R_Coil( "DB8000_PART_STATUS".UNIT_01.FIXTURE_2.PART_A.STATUS.PART_REJECTED )
   END_RUNG
   RUNG wire#w7
      Contact( "DB8000_PART_STATUS".HMI.UNIT_01_REJECT_PART )
      Contact( "DB8000_PART_STATUS".UNIT_01.FIXTURE_2.PART_A.STATUS.PRESENT )
      S_Coil( "DB8000_PART_STATUS".UNIT_01.FIXTURE_2.PART_A.STATUS.PART_REJECTED )
      R_Coil( "DB8000_PART_STATUS".UNIT_01.FIXTURE_2.PART_A.STATUS.OK )
   END_RUNG
   RUNG wire#w7
      Contact( "DB8000_PART_STATUS".HMI.UNIT_01_MASTER_PART )
      Contact( "DB8000_PART_STATUS".UNIT_01.FIXTURE_2.PART_A.STATUS.PRESENT )
      S_Coil( "DB8000_PART_STATUS".UNIT_01.FIXTURE_2.PART_A.STATUS.MASTER_PART )
   END_RUNG
   RUNG wire#w1
      { S7_Templates := "SrcType := Int" } EQ_Contact(in1 := "DB8000_PART_STATUS".HMI.PART_STATUS_FIXTURES_LIST, in2 := 3)
      wire#w10
      Contact( "DB4000_FIX_TABLE_POSITIONS".UNIT_01.FIXTURE_3.IN_LOAD_UNLOAD_STATION_1 )
      wire#w11
      Contact( "DB8000_PART_STATUS".HMI.UNIT_01_PART_PRESENT )
      Move(in := "DB2099_MANUAL_LOAD_DMC".DMC_ARRAY_CHAR_UNIT_01, out1 => "DB8000_PART_STATUS".UNIT_01.FIXTURE_3.PART_A.PART_ID)
      wire#w12
      S_Coil( "DB8000_PART_STATUS".UNIT_01.FIXTURE_3.PART_A.STATUS.PRESENT )
      S_Coil( "DB8000_PART_STATUS".UNIT_01.FIXTURE_3.PART_A.STATUS.PART_REJECTED )
   END_RUNG
   RUNG wire#w10
      Contact( "M_DUMMY_ON" )
   END_RUNG wire#w11
   RUNG wire#w12
      { S7_Templates := "SrcType := Int" } EQ_Contact(in1 := "DB8000_PART_STATUS".HMI.PART_STATUS_PART_STATUS_LIST, in2 := 1)
      S_Coil( "DB8000_PART_STATUS".UNIT_01.FIXTURE_3.PART_A.STATUS.CELL_STATUS.NEW_IN_TRANSIT )
   END_RUNG
   RUNG wire#w12
      { S7_Templates := "SrcType := Int" } EQ_Contact(in1 := "DB8000_PART_STATUS".HMI.PART_STATUS_PART_STATUS_LIST, in2 := 2)
      S_Coil( "DB8000_PART_STATUS".UNIT_01.FIXTURE_3.PART_A.STATUS.UNIT_01_STATUS.FACE_N_STATION_3_DONE )
   END_RUNG
   RUNG wire#w12
      { S7_Templates := "SrcType := Int" } EQ_Contact(in1 := "DB8000_PART_STATUS".HMI.PART_STATUS_PART_STATUS_LIST, in2 := 3)
      S_Coil( "DB8000_PART_STATUS".UNIT_01.FIXTURE_3.PART_A.STATUS.UNIT_01_STATUS.FACE_N_STATION_4_DONE )
   END_RUNG
   RUNG wire#w12
      { S7_Templates := "SrcType := Int" } EQ_Contact(in1 := "DB8000_PART_STATUS".HMI.PART_STATUS_PART_STATUS_LIST, in2 := 4)
      S_Coil( "DB8000_PART_STATUS".UNIT_01.FIXTURE_3.PART_A.STATUS.CELL_STATUS.U01_ONE_FACE_DONE_ROTATED )
   END_RUNG
   RUNG wire#w12
      { S7_Templates := "SrcType := Int" } EQ_Contact(in1 := "DB8000_PART_STATUS".HMI.PART_STATUS_PART_STATUS_LIST, in2 := 5)
      S_Coil( "DB8000_PART_STATUS".UNIT_01.FIXTURE_3.PART_A.STATUS.UNIT_01_STATUS.FACE_R_STATION_3_DONE )
   END_RUNG
   RUNG wire#w12
      { S7_Templates := "SrcType := Int" } EQ_Contact(in1 := "DB8000_PART_STATUS".HMI.PART_STATUS_PART_STATUS_LIST, in2 := 6)
      S_Coil( "DB8000_PART_STATUS".UNIT_01.FIXTURE_3.PART_A.STATUS.UNIT_01_STATUS.FACE_R_STATION_4_DONE )
   END_RUNG
   RUNG wire#w12
      { S7_Templates := "SrcType := Int" } EQ_Contact(in1 := "DB8000_PART_STATUS".HMI.PART_STATUS_PART_STATUS_LIST, in2 := 7)
      S_Coil( "DB8000_PART_STATUS".UNIT_01.FIXTURE_3.PART_A.STATUS.CELL_STATUS.U01_DONE_IN_TRANSIT )
   END_RUNG
   RUNG wire#w12
      { S7_Templates := "SrcType := Int" } EQ_Contact(in1 := "DB8000_PART_STATUS".HMI.PART_STATUS_PART_STATUS_LIST, in2 := 8)
      S_Coil( "DB8000_PART_STATUS".UNIT_01.FIXTURE_3.PART_A.STATUS.UNIT_02_STATUS.FACE_N_STATION_2_DONE )
   END_RUNG
   RUNG wire#w12
      { S7_Templates := "SrcType := Int" } EQ_Contact(in1 := "DB8000_PART_STATUS".HMI.PART_STATUS_PART_STATUS_LIST, in2 := 9)
      S_Coil( "DB8000_PART_STATUS".UNIT_01.FIXTURE_3.PART_A.STATUS.UNIT_02_STATUS.FACE_N_STATION_3_DONE )
   END_RUNG
   RUNG wire#w12
      { S7_Templates := "SrcType := Int" } EQ_Contact(in1 := "DB8000_PART_STATUS".HMI.PART_STATUS_PART_STATUS_LIST, in2 := 10)
      S_Coil( "DB8000_PART_STATUS".UNIT_01.FIXTURE_3.PART_A.STATUS.UNIT_02_STATUS.FACE_N_STATION_4_DONE )
   END_RUNG
   RUNG wire#w12
      { S7_Templates := "SrcType := Int" } EQ_Contact(in1 := "DB8000_PART_STATUS".HMI.PART_STATUS_PART_STATUS_LIST, in2 := 11)
      S_Coil( "DB8000_PART_STATUS".UNIT_01.FIXTURE_3.PART_A.STATUS.CELL_STATUS.U02_ONE_FACE_DONE_ROTATED )
   END_RUNG
   RUNG wire#w12
      { S7_Templates := "SrcType := Int" } EQ_Contact(in1 := "DB8000_PART_STATUS".HMI.PART_STATUS_PART_STATUS_LIST, in2 := 12)
      S_Coil( "DB8000_PART_STATUS".UNIT_01.FIXTURE_3.PART_A.STATUS.UNIT_02_STATUS.FACE_R_STATION_2_DONE )
   END_RUNG
   RUNG wire#w12
      { S7_Templates := "SrcType := Int" } EQ_Contact(in1 := "DB8000_PART_STATUS".HMI.PART_STATUS_PART_STATUS_LIST, in2 := 13)
      S_Coil( "DB8000_PART_STATUS".UNIT_01.FIXTURE_3.PART_A.STATUS.UNIT_02_STATUS.FACE_R_STATION_3_DONE )
   END_RUNG
   RUNG wire#w12
      { S7_Templates := "SrcType := Int" } EQ_Contact(in1 := "DB8000_PART_STATUS".HMI.PART_STATUS_PART_STATUS_LIST, in2 := 14)
      S_Coil( "DB8000_PART_STATUS".UNIT_01.FIXTURE_3.PART_A.STATUS.UNIT_02_STATUS.FACE_R_STATION_4_DONE )
   END_RUNG
   RUNG wire#w12
      { S7_Templates := "SrcType := Int" } EQ_Contact(in1 := "DB8000_PART_STATUS".HMI.PART_STATUS_PART_STATUS_LIST, in2 := 15)
      S_Coil( "DB8000_PART_STATUS".UNIT_01.FIXTURE_3.PART_A.STATUS.CELL_STATUS.U02_DONE_IN_TRANSIT )
   END_RUNG
   RUNG wire#w12
      { S7_Templates := "SrcType := Int" } EQ_Contact(in1 := "DB8000_PART_STATUS".HMI.PART_STATUS_PART_STATUS_LIST, in2 := 16)
      S_Coil( "DB8000_PART_STATUS".UNIT_01.FIXTURE_3.PART_A.STATUS.CELL_STATUS.COOLING_DONE )
   END_RUNG
   RUNG wire#w12
      { S7_Templates := "SrcType := Int" } EQ_Contact(in1 := "DB8000_PART_STATUS".HMI.PART_STATUS_PART_STATUS_LIST, in2 := 17)
      S_Coil( "DB8000_PART_STATUS".UNIT_01.FIXTURE_3.PART_A.STATUS.CELL_STATUS.INSPECTION_DONE )
   END_RUNG
   RUNG wire#w12
      { S7_Templates := "SrcType := Int" } EQ_Contact(in1 := "DB8000_PART_STATUS".HMI.PART_STATUS_PART_STATUS_LIST, in2 := 99)
      S_Coil( "DB8000_PART_STATUS".UNIT_01.FIXTURE_3.PART_A.STATUS.MASTER_PART )
   END_RUNG
   RUNG wire#w11
      Contact( "DB8000_PART_STATUS".HMI.UNIT_01_REMOVE_PART )
      wire#w13
      R_Coil( "DB2700_UNIT_01_FIXTURE_3".INPUT_PART_A_PRESENT_MEM )
      R_Coil( "DB8000_PART_STATUS".UNIT_01.FIXTURE_3.PART_A.STATUS.PRESENT )
      R_Coil( "DB8000_PART_STATUS".UNIT_01.FIXTURE_3.PART_A.STATUS.PART_REJECTED )
      R_Coil( "DB8000_PART_STATUS".UNIT_01.FIXTURE_3.PART_A.STATUS.MASTER_PART )
   END_RUNG
   RUNG wire#w13
      R_Coil( "DB8000_PART_STATUS".UNIT_01.FIXTURE_3.PART_A.STATUS.CELL_STATUS.NEW_IN_TRANSIT )
      R_Coil( "DB8000_PART_STATUS".UNIT_01.FIXTURE_3.PART_A.STATUS.UNIT_01_STATUS.FACE_N_STATION_3_DONE )
      R_Coil( "DB8000_PART_STATUS".UNIT_01.FIXTURE_3.PART_A.STATUS.UNIT_01_STATUS.FACE_N_STATION_4_DONE )
      R_Coil( "DB8000_PART_STATUS".UNIT_01.FIXTURE_3.PART_A.STATUS.CELL_STATUS.U01_ONE_FACE_DONE_ROTATED )
      R_Coil( "DB8000_PART_STATUS".UNIT_01.FIXTURE_3.PART_A.STATUS.UNIT_01_STATUS.FACE_R_STATION_3_DONE )
      R_Coil( "DB8000_PART_STATUS".UNIT_01.FIXTURE_3.PART_A.STATUS.UNIT_01_STATUS.FACE_R_STATION_4_DONE )
      R_Coil( "DB8000_PART_STATUS".UNIT_01.FIXTURE_3.PART_A.STATUS.CELL_STATUS.U01_DONE_IN_TRANSIT )
      R_Coil( "DB8000_PART_STATUS".UNIT_01.FIXTURE_3.PART_A.STATUS.UNIT_02_STATUS.FACE_N_STATION_2_DONE )
      R_Coil( "DB8000_PART_STATUS".UNIT_01.FIXTURE_3.PART_A.STATUS.UNIT_02_STATUS.FACE_N_STATION_3_DONE )
      R_Coil( "DB8000_PART_STATUS".UNIT_01.FIXTURE_3.PART_A.STATUS.UNIT_02_STATUS.FACE_N_STATION_4_DONE )
      R_Coil( "DB8000_PART_STATUS".UNIT_01.FIXTURE_3.PART_A.STATUS.CELL_STATUS.U02_ONE_FACE_DONE_ROTATED )
      R_Coil( "DB8000_PART_STATUS".UNIT_01.FIXTURE_3.PART_A.STATUS.UNIT_02_STATUS.FACE_R_STATION_2_DONE )
      R_Coil( "DB8000_PART_STATUS".UNIT_01.FIXTURE_3.PART_A.STATUS.UNIT_02_STATUS.FACE_R_STATION_3_DONE )
      R_Coil( "DB8000_PART_STATUS".UNIT_01.FIXTURE_3.PART_A.STATUS.UNIT_02_STATUS.FACE_R_STATION_4_DONE )
      R_Coil( "DB8000_PART_STATUS".UNIT_01.FIXTURE_3.PART_A.STATUS.CELL_STATUS.U02_DONE_IN_TRANSIT )
      R_Coil( "DB8000_PART_STATUS".UNIT_01.FIXTURE_3.PART_A.STATUS.CELL_STATUS.COOLING_DONE )
      R_Coil( "DB8000_PART_STATUS".UNIT_01.FIXTURE_3.PART_A.STATUS.CELL_STATUS.INSPECTION_DONE )
   END_RUNG
   RUNG wire#w13
      R_Coil( "DB8000_PART_STATUS".UNIT_01.FIXTURE_3.PART_A.STATUS.UNIT_01_STATUS.PROCESSED_IN_F3 )
      R_Coil( "DB8000_PART_STATUS".UNIT_01.FIXTURE_3.PART_A.STATUS.CELL_STATUS.U01_ONE_FACE_DONE )
      R_Coil( "DB8000_PART_STATUS".UNIT_01.FIXTURE_3.PART_A.STATUS.CELL_STATUS.U01_DONE )
   END_RUNG
   RUNG wire#w11
      Contact( "DB8000_PART_STATUS".HMI.UNIT_01_GOOD_PART )
      Contact( "DB8000_PART_STATUS".UNIT_01.FIXTURE_3.PART_A.STATUS.PRESENT )
      S_Coil( "DB8000_PART_STATUS".UNIT_01.FIXTURE_3.PART_A.STATUS.OK )
      R_Coil( "DB8000_PART_STATUS".UNIT_01.FIXTURE_3.PART_A.STATUS.PART_REJECTED )
   END_RUNG
   RUNG wire#w11
      Contact( "DB8000_PART_STATUS".HMI.UNIT_01_REJECT_PART )
      Contact( "DB8000_PART_STATUS".UNIT_01.FIXTURE_3.PART_A.STATUS.PRESENT )
      S_Coil( "DB8000_PART_STATUS".UNIT_01.FIXTURE_3.PART_A.STATUS.PART_REJECTED )
      R_Coil( "DB8000_PART_STATUS".UNIT_01.FIXTURE_3.PART_A.STATUS.OK )
   END_RUNG
   RUNG wire#w11
      Contact( "DB8000_PART_STATUS".HMI.UNIT_01_MASTER_PART )
      Contact( "DB8000_PART_STATUS".UNIT_01.FIXTURE_3.PART_A.STATUS.PRESENT )
      S_Coil( "DB8000_PART_STATUS".UNIT_01.FIXTURE_3.PART_A.STATUS.MASTER_PART )
   END_RUNG
   RUNG wire#w1
      { S7_Templates := "SrcType := Int" } EQ_Contact(in1 := "DB8000_PART_STATUS".HMI.PART_STATUS_FIXTURES_LIST, in2 := 4)
      wire#w14
      Contact( "DB4000_FIX_TABLE_POSITIONS".UNIT_01.FIXTURE_4.IN_LOAD_UNLOAD_STATION_1 )
      wire#w15
      Contact( "DB8000_PART_STATUS".HMI.UNIT_01_PART_PRESENT )
      Move(in := "DB2099_MANUAL_LOAD_DMC".DMC_ARRAY_CHAR_UNIT_01, out1 => "DB8000_PART_STATUS".UNIT_01.FIXTURE_4.PART_A.PART_ID)
      wire#w16
      S_Coil( "DB8000_PART_STATUS".UNIT_01.FIXTURE_4.PART_A.STATUS.PRESENT )
      S_Coil( "DB8000_PART_STATUS".UNIT_01.FIXTURE_4.PART_A.STATUS.PART_REJECTED )
   END_RUNG
   RUNG wire#w14
      Contact( "M_DUMMY_ON" )
   END_RUNG wire#w15
   RUNG wire#w16
      { S7_Templates := "SrcType := Int" } EQ_Contact(in1 := "DB8000_PART_STATUS".HMI.PART_STATUS_PART_STATUS_LIST, in2 := 1)
      S_Coil( "DB8000_PART_STATUS".UNIT_01.FIXTURE_4.PART_A.STATUS.CELL_STATUS.NEW_IN_TRANSIT )
   END_RUNG
   RUNG wire#w16
      { S7_Templates := "SrcType := Int" } EQ_Contact(in1 := "DB8000_PART_STATUS".HMI.PART_STATUS_PART_STATUS_LIST, in2 := 2)
      S_Coil( "DB8000_PART_STATUS".UNIT_01.FIXTURE_4.PART_A.STATUS.UNIT_01_STATUS.FACE_N_STATION_3_DONE )
   END_RUNG
   RUNG wire#w16
      { S7_Templates := "SrcType := Int" } EQ_Contact(in1 := "DB8000_PART_STATUS".HMI.PART_STATUS_PART_STATUS_LIST, in2 := 3)
      S_Coil( "DB8000_PART_STATUS".UNIT_01.FIXTURE_4.PART_A.STATUS.UNIT_01_STATUS.FACE_N_STATION_4_DONE )
   END_RUNG
   RUNG wire#w16
      { S7_Templates := "SrcType := Int" } EQ_Contact(in1 := "DB8000_PART_STATUS".HMI.PART_STATUS_PART_STATUS_LIST, in2 := 4)
      S_Coil( "DB8000_PART_STATUS".UNIT_01.FIXTURE_4.PART_A.STATUS.CELL_STATUS.U01_ONE_FACE_DONE_ROTATED )
   END_RUNG
   RUNG wire#w16
      { S7_Templates := "SrcType := Int" } EQ_Contact(in1 := "DB8000_PART_STATUS".HMI.PART_STATUS_PART_STATUS_LIST, in2 := 5)
      S_Coil( "DB8000_PART_STATUS".UNIT_01.FIXTURE_4.PART_A.STATUS.UNIT_01_STATUS.FACE_R_STATION_3_DONE )
   END_RUNG
   RUNG wire#w16
      { S7_Templates := "SrcType := Int" } EQ_Contact(in1 := "DB8000_PART_STATUS".HMI.PART_STATUS_PART_STATUS_LIST, in2 := 6)
      S_Coil( "DB8000_PART_STATUS".UNIT_01.FIXTURE_4.PART_A.STATUS.UNIT_01_STATUS.FACE_R_STATION_4_DONE )
   END_RUNG
   RUNG wire#w16
      { S7_Templates := "SrcType := Int" } EQ_Contact(in1 := "DB8000_PART_STATUS".HMI.PART_STATUS_PART_STATUS_LIST, in2 := 7)
      S_Coil( "DB8000_PART_STATUS".UNIT_01.FIXTURE_4.PART_A.STATUS.CELL_STATUS.U01_DONE_IN_TRANSIT )
   END_RUNG
   RUNG wire#w16
      { S7_Templates := "SrcType := Int" } EQ_Contact(in1 := "DB8000_PART_STATUS".HMI.PART_STATUS_PART_STATUS_LIST, in2 := 8)
      S_Coil( "DB8000_PART_STATUS".UNIT_01.FIXTURE_4.PART_A.STATUS.UNIT_02_STATUS.FACE_N_STATION_2_DONE )
   END_RUNG
   RUNG wire#w16
      { S7_Templates := "SrcType := Int" } EQ_Contact(in1 := "DB8000_PART_STATUS".HMI.PART_STATUS_PART_STATUS_LIST, in2 := 9)
      S_Coil( "DB8000_PART_STATUS".UNIT_01.FIXTURE_4.PART_A.STATUS.UNIT_02_STATUS.FACE_N_STATION_3_DONE )
   END_RUNG
   RUNG wire#w16
      { S7_Templates := "SrcType := Int" } EQ_Contact(in1 := "DB8000_PART_STATUS".HMI.PART_STATUS_PART_STATUS_LIST, in2 := 10)
      S_Coil( "DB8000_PART_STATUS".UNIT_01.FIXTURE_4.PART_A.STATUS.UNIT_02_STATUS.FACE_N_STATION_4_DONE )
   END_RUNG
   RUNG wire#w16
      { S7_Templates := "SrcType := Int" } EQ_Contact(in1 := "DB8000_PART_STATUS".HMI.PART_STATUS_PART_STATUS_LIST, in2 := 11)
      S_Coil( "DB8000_PART_STATUS".UNIT_01.FIXTURE_4.PART_A.STATUS.CELL_STATUS.U02_ONE_FACE_DONE_ROTATED )
   END_RUNG
   RUNG wire#w16
      { S7_Templates := "SrcType := Int" } EQ_Contact(in1 := "DB8000_PART_STATUS".HMI.PART_STATUS_PART_STATUS_LIST, in2 := 12)
      S_Coil( "DB8000_PART_STATUS".UNIT_01.FIXTURE_4.PART_A.STATUS.UNIT_02_STATUS.FACE_R_STATION_2_DONE )
   END_RUNG
   RUNG wire#w16
      { S7_Templates := "SrcType := Int" } EQ_Contact(in1 := "DB8000_PART_STATUS".HMI.PART_STATUS_PART_STATUS_LIST, in2 := 13)
      S_Coil( "DB8000_PART_STATUS".UNIT_01.FIXTURE_4.PART_A.STATUS.UNIT_02_STATUS.FACE_R_STATION_3_DONE )
   END_RUNG
   RUNG wire#w16
      { S7_Templates := "SrcType := Int" } EQ_Contact(in1 := "DB8000_PART_STATUS".HMI.PART_STATUS_PART_STATUS_LIST, in2 := 14)
      S_Coil( "DB8000_PART_STATUS".UNIT_01.FIXTURE_4.PART_A.STATUS.UNIT_02_STATUS.FACE_R_STATION_4_DONE )
   END_RUNG
   RUNG wire#w16
      { S7_Templates := "SrcType := Int" } EQ_Contact(in1 := "DB8000_PART_STATUS".HMI.PART_STATUS_PART_STATUS_LIST, in2 := 15)
      S_Coil( "DB8000_PART_STATUS".UNIT_01.FIXTURE_4.PART_A.STATUS.CELL_STATUS.U02_DONE_IN_TRANSIT )
   END_RUNG
   RUNG wire#w16
      { S7_Templates := "SrcType := Int" } EQ_Contact(in1 := "DB8000_PART_STATUS".HMI.PART_STATUS_PART_STATUS_LIST, in2 := 16)
      S_Coil( "DB8000_PART_STATUS".UNIT_01.FIXTURE_4.PART_A.STATUS.CELL_STATUS.COOLING_DONE )
   END_RUNG
   RUNG wire#w16
      { S7_Templates := "SrcType := Int" } EQ_Contact(in1 := "DB8000_PART_STATUS".HMI.PART_STATUS_PART_STATUS_LIST, in2 := 17)
      S_Coil( "DB8000_PART_STATUS".UNIT_01.FIXTURE_4.PART_A.STATUS.CELL_STATUS.INSPECTION_DONE )
   END_RUNG
   RUNG wire#w16
      { S7_Templates := "SrcType := Int" } EQ_Contact(in1 := "DB8000_PART_STATUS".HMI.PART_STATUS_PART_STATUS_LIST, in2 := 99)
      S_Coil( "DB8000_PART_STATUS".UNIT_01.FIXTURE_4.PART_A.STATUS.MASTER_PART )
   END_RUNG
   RUNG wire#w15
      Contact( "DB8000_PART_STATUS".HMI.UNIT_01_REMOVE_PART )
      wire#w17
      R_Coil( "DB2800_UNIT_01_FIXTURE_4".INPUT_PART_A_PRESENT_MEM )
      R_Coil( "DB8000_PART_STATUS".UNIT_01.FIXTURE_4.PART_A.STATUS.PRESENT )
      R_Coil( "DB8000_PART_STATUS".UNIT_01.FIXTURE_4.PART_A.STATUS.PART_REJECTED )
      R_Coil( "DB8000_PART_STATUS".UNIT_01.FIXTURE_4.PART_A.STATUS.MASTER_PART )
   END_RUNG
   RUNG wire#w17
      R_Coil( "DB8000_PART_STATUS".UNIT_01.FIXTURE_4.PART_A.STATUS.CELL_STATUS.NEW_IN_TRANSIT )
      R_Coil( "DB8000_PART_STATUS".UNIT_01.FIXTURE_4.PART_A.STATUS.UNIT_01_STATUS.FACE_N_STATION_3_DONE )
      R_Coil( "DB8000_PART_STATUS".UNIT_01.FIXTURE_4.PART_A.STATUS.UNIT_01_STATUS.FACE_N_STATION_4_DONE )
      R_Coil( "DB8000_PART_STATUS".UNIT_01.FIXTURE_4.PART_A.STATUS.CELL_STATUS.U01_ONE_FACE_DONE_ROTATED )
      R_Coil( "DB8000_PART_STATUS".UNIT_01.FIXTURE_4.PART_A.STATUS.UNIT_01_STATUS.FACE_R_STATION_3_DONE )
      R_Coil( "DB8000_PART_STATUS".UNIT_01.FIXTURE_4.PART_A.STATUS.UNIT_01_STATUS.FACE_R_STATION_4_DONE )
      R_Coil( "DB8000_PART_STATUS".UNIT_01.FIXTURE_4.PART_A.STATUS.CELL_STATUS.U01_DONE_IN_TRANSIT )
      R_Coil( "DB8000_PART_STATUS".UNIT_01.FIXTURE_4.PART_A.STATUS.UNIT_02_STATUS.FACE_N_STATION_2_DONE )
      R_Coil( "DB8000_PART_STATUS".UNIT_01.FIXTURE_4.PART_A.STATUS.UNIT_02_STATUS.FACE_N_STATION_3_DONE )
      R_Coil( "DB8000_PART_STATUS".UNIT_01.FIXTURE_4.PART_A.STATUS.UNIT_02_STATUS.FACE_N_STATION_4_DONE )
      R_Coil( "DB8000_PART_STATUS".UNIT_01.FIXTURE_4.PART_A.STATUS.CELL_STATUS.U02_ONE_FACE_DONE_ROTATED )
      R_Coil( "DB8000_PART_STATUS".UNIT_01.FIXTURE_4.PART_A.STATUS.UNIT_02_STATUS.FACE_R_STATION_2_DONE )
      R_Coil( "DB8000_PART_STATUS".UNIT_01.FIXTURE_4.PART_A.STATUS.UNIT_02_STATUS.FACE_R_STATION_3_DONE )
      R_Coil( "DB8000_PART_STATUS".UNIT_01.FIXTURE_4.PART_A.STATUS.UNIT_02_STATUS.FACE_R_STATION_4_DONE )
      R_Coil( "DB8000_PART_STATUS".UNIT_01.FIXTURE_4.PART_A.STATUS.CELL_STATUS.U02_DONE_IN_TRANSIT )
      R_Coil( "DB8000_PART_STATUS".UNIT_01.FIXTURE_4.PART_A.STATUS.CELL_STATUS.COOLING_DONE )
      R_Coil( "DB8000_PART_STATUS".UNIT_01.FIXTURE_4.PART_A.STATUS.CELL_STATUS.INSPECTION_DONE )
   END_RUNG
   RUNG wire#w17
      R_Coil( "DB8000_PART_STATUS".UNIT_01.FIXTURE_4.PART_A.STATUS.UNIT_01_STATUS.PROCESSED_IN_F4 )
      R_Coil( "DB8000_PART_STATUS".UNIT_01.FIXTURE_4.PART_A.STATUS.CELL_STATUS.U01_ONE_FACE_DONE )
      R_Coil( "DB8000_PART_STATUS".UNIT_01.FIXTURE_4.PART_A.STATUS.CELL_STATUS.U01_DONE )
   END_RUNG
   RUNG wire#w15
      Contact( "DB8000_PART_STATUS".HMI.UNIT_01_GOOD_PART )
      Contact( "DB8000_PART_STATUS".UNIT_01.FIXTURE_4.PART_A.STATUS.PRESENT )
      S_Coil( "DB8000_PART_STATUS".UNIT_01.FIXTURE_4.PART_A.STATUS.OK )
      R_Coil( "DB8000_PART_STATUS".UNIT_01.FIXTURE_4.PART_A.STATUS.PART_REJECTED )
   END_RUNG
   RUNG wire#w15
      Contact( "DB8000_PART_STATUS".HMI.UNIT_01_REJECT_PART )
      Contact( "DB8000_PART_STATUS".UNIT_01.FIXTURE_4.PART_A.STATUS.PRESENT )
      S_Coil( "DB8000_PART_STATUS".UNIT_01.FIXTURE_4.PART_A.STATUS.PART_REJECTED )
      R_Coil( "DB8000_PART_STATUS".UNIT_01.FIXTURE_4.PART_A.STATUS.OK )
   END_RUNG
   RUNG wire#w15
      Contact( "DB8000_PART_STATUS".HMI.UNIT_01_MASTER_PART )
      Contact( "DB8000_PART_STATUS".UNIT_01.FIXTURE_4.PART_A.STATUS.PRESENT )
      S_Coil( "DB8000_PART_STATUS".UNIT_02.FIXTURE_4.PART_A.STATUS.MASTER_PART )
   END_RUNG
   // the same network as SCL:
   #_w1 := "DB2001_MODES_GENERAL".GENERAL.MANUAL_SELECTED AND ("DB8000_PART_STATUS".HMI.PART_STATUS_FIXTURES_LIST = 1) AND ("DB4000_FIX_TABLE_POSITIONS".UNIT_01.FIXTURE_1.IN_LOAD_UNLOAD_STATION_1 OR "M_DUMMY_ON");
   #_w2 := #_w1 AND "DB8000_PART_STATUS".HMI.UNIT_01_PART_PRESENT;
   IF #_w2 THEN
       "DB8000_PART_STATUS".UNIT_01.FIXTURE_1.PART_A.PART_ID := "DB2099_MANUAL_LOAD_DMC".DMC_ARRAY_CHAR_UNIT_01;
       "DB8000_PART_STATUS".UNIT_01.FIXTURE_1.PART_A.STATUS.PRESENT := TRUE;
       "DB8000_PART_STATUS".UNIT_01.FIXTURE_1.PART_A.STATUS.PART_REJECTED := TRUE;
   END_IF;
   IF #_w2 AND ("DB8000_PART_STATUS".HMI.PART_STATUS_PART_STATUS_LIST = 1) THEN
       "DB8000_PART_STATUS".UNIT_01.FIXTURE_1.PART_A.STATUS.CELL_STATUS.NEW_IN_TRANSIT := TRUE;
   END_IF;
   IF #_w2 AND ("DB8000_PART_STATUS".HMI.PART_STATUS_PART_STATUS_LIST = 2) THEN
       "DB8000_PART_STATUS".UNIT_01.FIXTURE_1.PART_A.STATUS.UNIT_01_STATUS.FACE_N_STATION_3_DONE := TRUE;
   END_IF;
   IF #_w2 AND ("DB8000_PART_STATUS".HMI.PART_STATUS_PART_STATUS_LIST = 3) THEN
       "DB8000_PART_STATUS".UNIT_01.FIXTURE_1.PART_A.STATUS.UNIT_01_STATUS.FACE_N_STATION_4_DONE := TRUE;
   END_IF;
   IF #_w2 AND ("DB8000_PART_STATUS".HMI.PART_STATUS_PART_STATUS_LIST = 4) THEN
       "DB8000_PART_STATUS".UNIT_01.FIXTURE_1.PART_A.STATUS.CELL_STATUS.U01_ONE_FACE_DONE_ROTATED := TRUE;
   END_IF;
   IF #_w2 AND ("DB8000_PART_STATUS".HMI.PART_STATUS_PART_STATUS_LIST = 5) THEN
       "DB8000_PART_STATUS".UNIT_01.FIXTURE_1.PART_A.STATUS.UNIT_01_STATUS.FACE_R_STATION_3_DONE := TRUE;
   END_IF;
   IF #_w2 AND ("DB8000_PART_STATUS".HMI.PART_STATUS_PART_STATUS_LIST = 6) THEN
       "DB8000_PART_STATUS".UNIT_01.FIXTURE_1.PART_A.STATUS.UNIT_01_STATUS.FACE_R_STATION_4_DONE := TRUE;
   END_IF;
   IF #_w2 AND ("DB8000_PART_STATUS".HMI.PART_STATUS_PART_STATUS_LIST = 7) THEN
       "DB8000_PART_STATUS".UNIT_01.FIXTURE_1.PART_A.STATUS.CELL_STATUS.U01_DONE_IN_TRANSIT := TRUE;
   END_IF;
   IF #_w2 AND ("DB8000_PART_STATUS".HMI.PART_STATUS_PART_STATUS_LIST = 8) THEN
       "DB8000_PART_STATUS".UNIT_01.FIXTURE_1.PART_A.STATUS.UNIT_02_STATUS.FACE_N_STATION_2_DONE := TRUE;
   END_IF;
   IF #_w2 AND ("DB8000_PART_STATUS".HMI.PART_STATUS_PART_STATUS_LIST = 9) THEN
       "DB8000_PART_STATUS".UNIT_01.FIXTURE_1.PART_A.STATUS.UNIT_02_STATUS.FACE_N_STATION_3_DONE := TRUE;
   END_IF;
   IF #_w2 AND ("DB8000_PART_STATUS".HMI.PART_STATUS_PART_STATUS_LIST = 10) THEN
       "DB8000_PART_STATUS".UNIT_01.FIXTURE_1.PART_A.STATUS.UNIT_02_STATUS.FACE_N_STATION_4_DONE := TRUE;
   END_IF;
   IF #_w2 AND ("DB8000_PART_STATUS".HMI.PART_STATUS_PART_STATUS_LIST = 11) THEN
       "DB8000_PART_STATUS".UNIT_01.FIXTURE_1.PART_A.STATUS.CELL_STATUS.U02_ONE_FACE_DONE_ROTATED := TRUE;
   END_IF;
   IF #_w2 AND ("DB8000_PART_STATUS".HMI.PART_STATUS_PART_STATUS_LIST = 12) THEN
       "DB8000_PART_STATUS".UNIT_01.FIXTURE_1.PART_A.STATUS.UNIT_02_STATUS.FACE_R_STATION_2_DONE := TRUE;
   END_IF;
   IF #_w2 AND ("DB8000_PART_STATUS".HMI.PART_STATUS_PART_STATUS_LIST = 13) THEN
       "DB8000_PART_STATUS".UNIT_01.FIXTURE_1.PART_A.STATUS.UNIT_02_STATUS.FACE_R_STATION_3_DONE := TRUE;
   END_IF;
   IF #_w2 AND ("DB8000_PART_STATUS".HMI.PART_STATUS_PART_STATUS_LIST = 14) THEN
       "DB8000_PART_STATUS".UNIT_01.FIXTURE_1.PART_A.STATUS.UNIT_02_STATUS.FACE_R_STATION_4_DONE := TRUE;
   END_IF;
   IF #_w2 AND ("DB8000_PART_STATUS".HMI.PART_STATUS_PART_STATUS_LIST = 15) THEN
       "DB8000_PART_STATUS".UNIT_01.FIXTURE_1.PART_A.STATUS.CELL_STATUS.U02_DONE_IN_TRANSIT := TRUE;
   END_IF;
   IF #_w2 AND ("DB8000_PART_STATUS".HMI.PART_STATUS_PART_STATUS_LIST = 16) THEN
       "DB8000_PART_STATUS".UNIT_01.FIXTURE_1.PART_A.STATUS.CELL_STATUS.COOLING_DONE := TRUE;
   END_IF;
   IF #_w2 AND ("DB8000_PART_STATUS".HMI.PART_STATUS_PART_STATUS_LIST = 17) THEN
       "DB8000_PART_STATUS".UNIT_01.FIXTURE_1.PART_A.STATUS.CELL_STATUS.INSPECTION_DONE := TRUE;
   END_IF;
   IF #_w2 AND ("DB8000_PART_STATUS".HMI.PART_STATUS_PART_STATUS_LIST = 99) THEN
       "DB8000_PART_STATUS".UNIT_01.FIXTURE_1.PART_A.STATUS.MASTER_PART := TRUE;
   END_IF;
   IF #_w1 AND "DB8000_PART_STATUS".HMI.UNIT_01_REMOVE_PART THEN
       "DB2500_UNIT_01_FIXTURE_1".INPUT_PART_A_PRESENT_MEM := FALSE;
       "DB8000_PART_STATUS".UNIT_01.FIXTURE_1.PART_A.STATUS.PRESENT := FALSE;
       "DB8000_PART_STATUS".UNIT_01.FIXTURE_1.PART_A.STATUS.PART_REJECTED := FALSE;
       "DB8000_PART_STATUS".UNIT_01.FIXTURE_1.PART_A.STATUS.MASTER_PART := FALSE;
       "DB8000_PART_STATUS".UNIT_01.FIXTURE_1.PART_A.STATUS.CELL_STATUS.NEW_IN_TRANSIT := FALSE;
       "DB8000_PART_STATUS".UNIT_01.FIXTURE_1.PART_A.STATUS.UNIT_01_STATUS.FACE_N_STATION_3_DONE := FALSE;
       "DB8000_PART_STATUS".UNIT_01.FIXTURE_1.PART_A.STATUS.UNIT_01_STATUS.FACE_N_STATION_4_DONE := FALSE;
       "DB8000_PART_STATUS".UNIT_01.FIXTURE_1.PART_A.STATUS.CELL_STATUS.U01_ONE_FACE_DONE_ROTATED := FALSE;
       "DB8000_PART_STATUS".UNIT_01.FIXTURE_1.PART_A.STATUS.UNIT_01_STATUS.FACE_R_STATION_3_DONE := FALSE;
       "DB8000_PART_STATUS".UNIT_01.FIXTURE_1.PART_A.STATUS.UNIT_01_STATUS.FACE_R_STATION_4_DONE := FALSE;
       "DB8000_PART_STATUS".UNIT_01.FIXTURE_1.PART_A.STATUS.CELL_STATUS.U01_DONE_IN_TRANSIT := FALSE;
       "DB8000_PART_STATUS".UNIT_01.FIXTURE_1.PART_A.STATUS.UNIT_02_STATUS.FACE_N_STATION_2_DONE := FALSE;
       "DB8000_PART_STATUS".UNIT_01.FIXTURE_1.PART_A.STATUS.UNIT_02_STATUS.FACE_N_STATION_3_DONE := FALSE;
       "DB8000_PART_STATUS".UNIT_01.FIXTURE_1.PART_A.STATUS.UNIT_02_STATUS.FACE_N_STATION_4_DONE := FALSE;
       "DB8000_PART_STATUS".UNIT_01.FIXTURE_1.PART_A.STATUS.CELL_STATUS.U02_ONE_FACE_DONE_ROTATED := FALSE;
       "DB8000_PART_STATUS".UNIT_01.FIXTURE_1.PART_A.STATUS.UNIT_02_STATUS.FACE_R_STATION_2_DONE := FALSE;
       "DB8000_PART_STATUS".UNIT_01.FIXTURE_1.PART_A.STATUS.UNIT_02_STATUS.FACE_R_STATION_3_DONE := FALSE;
       "DB8000_PART_STATUS".UNIT_01.FIXTURE_1.PART_A.STATUS.UNIT_02_STATUS.FACE_R_STATION_4_DONE := FALSE;
       "DB8000_PART_STATUS".UNIT_01.FIXTURE_1.PART_A.STATUS.CELL_STATUS.U02_DONE_IN_TRANSIT := FALSE;
       "DB8000_PART_STATUS".UNIT_01.FIXTURE_1.PART_A.STATUS.CELL_STATUS.COOLING_DONE := FALSE;
       "DB8000_PART_STATUS".UNIT_01.FIXTURE_1.PART_A.STATUS.CELL_STATUS.INSPECTION_DONE := FALSE;
       "DB8000_PART_STATUS".UNIT_01.FIXTURE_1.PART_A.STATUS.UNIT_01_STATUS.PROCESSED_IN_F1 := FALSE;
       "DB8000_PART_STATUS".UNIT_01.FIXTURE_1.PART_A.STATUS.CELL_STATUS.U01_ONE_FACE_DONE := FALSE;
       "DB8000_PART_STATUS".UNIT_01.FIXTURE_1.PART_A.STATUS.CELL_STATUS.U01_DONE := FALSE;
   END_IF;
   IF #_w1 AND "DB8000_PART_STATUS".HMI.UNIT_01_GOOD_PART AND "DB8000_PART_STATUS".UNIT_01.FIXTURE_1.PART_A.STATUS.PRESENT THEN
       "DB8000_PART_STATUS".UNIT_01.FIXTURE_1.PART_A.STATUS.OK := TRUE;
       "DB8000_PART_STATUS".UNIT_01.FIXTURE_1.PART_A.STATUS.PART_REJECTED := FALSE;
   END_IF;
   IF #_w1 AND "DB8000_PART_STATUS".HMI.UNIT_01_REJECT_PART AND "DB8000_PART_STATUS".UNIT_01.FIXTURE_1.PART_A.STATUS.PRESENT THEN
       "DB8000_PART_STATUS".UNIT_01.FIXTURE_1.PART_A.STATUS.PART_REJECTED := TRUE;
       "DB8000_PART_STATUS".UNIT_01.FIXTURE_1.PART_A.STATUS.OK := FALSE;
   END_IF;
   IF #_w1 AND "DB8000_PART_STATUS".HMI.UNIT_01_MASTER_PART AND "DB8000_PART_STATUS".UNIT_01.FIXTURE_1.PART_A.STATUS.PRESENT THEN
       "DB8000_PART_STATUS".UNIT_01.FIXTURE_1.PART_A.STATUS.MASTER_PART := TRUE;
   END_IF;
   #_w3 := "DB2001_MODES_GENERAL".GENERAL.MANUAL_SELECTED AND ("DB8000_PART_STATUS".HMI.PART_STATUS_FIXTURES_LIST = 2) AND ("DB4000_FIX_TABLE_POSITIONS".UNIT_01.FIXTURE_2.IN_LOAD_UNLOAD_STATION_1 OR "M_DUMMY_ON");
   #_w4 := #_w3 AND "DB8000_PART_STATUS".HMI.UNIT_01_PART_PRESENT;
   IF #_w4 THEN
       "DB8000_PART_STATUS".UNIT_01.FIXTURE_2.PART_A.PART_ID := "DB2099_MANUAL_LOAD_DMC".DMC_ARRAY_CHAR_UNIT_01;
       "DB8000_PART_STATUS".UNIT_01.FIXTURE_2.PART_A.STATUS.PRESENT := TRUE;
       "DB8000_PART_STATUS".UNIT_01.FIXTURE_2.PART_A.STATUS.PART_REJECTED := TRUE;
   END_IF;
   IF #_w4 AND ("DB8000_PART_STATUS".HMI.PART_STATUS_PART_STATUS_LIST = 1) THEN
       "DB8000_PART_STATUS".UNIT_01.FIXTURE_2.PART_A.STATUS.CELL_STATUS.NEW_IN_TRANSIT := TRUE;
   END_IF;
   IF #_w4 AND ("DB8000_PART_STATUS".HMI.PART_STATUS_PART_STATUS_LIST = 2) THEN
       "DB8000_PART_STATUS".UNIT_01.FIXTURE_2.PART_A.STATUS.UNIT_01_STATUS.FACE_N_STATION_3_DONE := TRUE;
   END_IF;
   IF #_w4 AND ("DB8000_PART_STATUS".HMI.PART_STATUS_PART_STATUS_LIST = 3) THEN
       "DB8000_PART_STATUS".UNIT_01.FIXTURE_2.PART_A.STATUS.UNIT_01_STATUS.FACE_N_STATION_4_DONE := TRUE;
   END_IF;
   IF #_w4 AND ("DB8000_PART_STATUS".HMI.PART_STATUS_PART_STATUS_LIST = 4) THEN
       "DB8000_PART_STATUS".UNIT_01.FIXTURE_2.PART_A.STATUS.CELL_STATUS.U01_ONE_FACE_DONE_ROTATED := TRUE;
   END_IF;
   IF #_w4 AND ("DB8000_PART_STATUS".HMI.PART_STATUS_PART_STATUS_LIST = 5) THEN
       "DB8000_PART_STATUS".UNIT_01.FIXTURE_2.PART_A.STATUS.UNIT_01_STATUS.FACE_R_STATION_3_DONE := TRUE;
   END_IF;
   IF #_w4 AND ("DB8000_PART_STATUS".HMI.PART_STATUS_PART_STATUS_LIST = 6) THEN
       "DB8000_PART_STATUS".UNIT_01.FIXTURE_2.PART_A.STATUS.UNIT_01_STATUS.FACE_R_STATION_4_DONE := TRUE;
   END_IF;
   IF #_w4 AND ("DB8000_PART_STATUS".HMI.PART_STATUS_PART_STATUS_LIST = 7) THEN
       "DB8000_PART_STATUS".UNIT_01.FIXTURE_2.PART_A.STATUS.CELL_STATUS.U01_DONE_IN_TRANSIT := TRUE;
   END_IF;
   IF #_w4 AND ("DB8000_PART_STATUS".HMI.PART_STATUS_PART_STATUS_LIST = 8) THEN
       "DB8000_PART_STATUS".UNIT_01.FIXTURE_2.PART_A.STATUS.UNIT_02_STATUS.FACE_N_STATION_2_DONE := TRUE;
   END_IF;
   IF #_w4 AND ("DB8000_PART_STATUS".HMI.PART_STATUS_PART_STATUS_LIST = 9) THEN
       "DB8000_PART_STATUS".UNIT_01.FIXTURE_2.PART_A.STATUS.UNIT_02_STATUS.FACE_N_STATION_3_DONE := TRUE;
   END_IF;
   IF #_w4 AND ("DB8000_PART_STATUS".HMI.PART_STATUS_PART_STATUS_LIST = 10) THEN
       "DB8000_PART_STATUS".UNIT_01.FIXTURE_2.PART_A.STATUS.UNIT_02_STATUS.FACE_N_STATION_4_DONE := TRUE;
   END_IF;
   IF #_w4 AND ("DB8000_PART_STATUS".HMI.PART_STATUS_PART_STATUS_LIST = 11) THEN
       "DB8000_PART_STATUS".UNIT_01.FIXTURE_2.PART_A.STATUS.CELL_STATUS.U02_ONE_FACE_DONE_ROTATED := TRUE;
   END_IF;
   IF #_w4 AND ("DB8000_PART_STATUS".HMI.PART_STATUS_PART_STATUS_LIST = 12) THEN
       "DB8000_PART_STATUS".UNIT_01.FIXTURE_2.PART_A.STATUS.UNIT_02_STATUS.FACE_R_STATION_2_DONE := TRUE;
   END_IF;
   IF #_w4 AND ("DB8000_PART_STATUS".HMI.PART_STATUS_PART_STATUS_LIST = 13) THEN
       "DB8000_PART_STATUS".UNIT_01.FIXTURE_2.PART_A.STATUS.UNIT_02_STATUS.FACE_R_STATION_3_DONE := TRUE;
   END_IF;
   IF #_w4 AND ("DB8000_PART_STATUS".HMI.PART_STATUS_PART_STATUS_LIST = 14) THEN
       "DB8000_PART_STATUS".UNIT_01.FIXTURE_2.PART_A.STATUS.UNIT_02_STATUS.FACE_R_STATION_4_DONE := TRUE;
   END_IF;
   IF #_w4 AND ("DB8000_PART_STATUS".HMI.PART_STATUS_PART_STATUS_LIST = 15) THEN
       "DB8000_PART_STATUS".UNIT_01.FIXTURE_2.PART_A.STATUS.CELL_STATUS.U02_DONE_IN_TRANSIT := TRUE;
   END_IF;
   IF #_w4 AND ("DB8000_PART_STATUS".HMI.PART_STATUS_PART_STATUS_LIST = 16) THEN
       "DB8000_PART_STATUS".UNIT_01.FIXTURE_2.PART_A.STATUS.CELL_STATUS.COOLING_DONE := TRUE;
   END_IF;
   IF #_w4 AND ("DB8000_PART_STATUS".HMI.PART_STATUS_PART_STATUS_LIST = 17) THEN
       "DB8000_PART_STATUS".UNIT_01.FIXTURE_2.PART_A.STATUS.CELL_STATUS.INSPECTION_DONE := TRUE;
   END_IF;
   IF #_w4 AND ("DB8000_PART_STATUS".HMI.PART_STATUS_PART_STATUS_LIST = 99) THEN
       "DB8000_PART_STATUS".UNIT_01.FIXTURE_2.PART_A.STATUS.MASTER_PART := TRUE;
   END_IF;
   IF #_w3 AND "DB8000_PART_STATUS".HMI.UNIT_01_REMOVE_PART THEN
       "DB2600_UNIT_01_FIXTURE_2".INPUT_PART_A_PRESENT_MEM := FALSE;
       "DB8000_PART_STATUS".UNIT_01.FIXTURE_2.PART_A.STATUS.PRESENT := FALSE;
       "DB8000_PART_STATUS".UNIT_01.FIXTURE_2.PART_A.STATUS.PART_REJECTED := FALSE;
       "DB8000_PART_STATUS".UNIT_01.FIXTURE_2.PART_A.STATUS.MASTER_PART := FALSE;
       "DB8000_PART_STATUS".UNIT_01.FIXTURE_2.PART_A.STATUS.CELL_STATUS.NEW_IN_TRANSIT := FALSE;
       "DB8000_PART_STATUS".UNIT_01.FIXTURE_2.PART_A.STATUS.UNIT_01_STATUS.FACE_N_STATION_3_DONE := FALSE;
       "DB8000_PART_STATUS".UNIT_01.FIXTURE_2.PART_A.STATUS.UNIT_01_STATUS.FACE_N_STATION_4_DONE := FALSE;
       "DB8000_PART_STATUS".UNIT_01.FIXTURE_2.PART_A.STATUS.CELL_STATUS.U01_ONE_FACE_DONE_ROTATED := FALSE;
       "DB8000_PART_STATUS".UNIT_01.FIXTURE_2.PART_A.STATUS.UNIT_01_STATUS.FACE_R_STATION_3_DONE := FALSE;
       "DB8000_PART_STATUS".UNIT_01.FIXTURE_2.PART_A.STATUS.UNIT_01_STATUS.FACE_R_STATION_4_DONE := FALSE;
       "DB8000_PART_STATUS".UNIT_01.FIXTURE_2.PART_A.STATUS.CELL_STATUS.U01_DONE_IN_TRANSIT := FALSE;
       "DB8000_PART_STATUS".UNIT_01.FIXTURE_2.PART_A.STATUS.UNIT_02_STATUS.FACE_N_STATION_2_DONE := FALSE;
       "DB8000_PART_STATUS".UNIT_01.FIXTURE_2.PART_A.STATUS.UNIT_02_STATUS.FACE_N_STATION_3_DONE := FALSE;
       "DB8000_PART_STATUS".UNIT_01.FIXTURE_2.PART_A.STATUS.UNIT_02_STATUS.FACE_N_STATION_4_DONE := FALSE;
       "DB8000_PART_STATUS".UNIT_01.FIXTURE_2.PART_A.STATUS.CELL_STATUS.U02_ONE_FACE_DONE_ROTATED := FALSE;
       "DB8000_PART_STATUS".UNIT_01.FIXTURE_2.PART_A.STATUS.UNIT_02_STATUS.FACE_R_STATION_2_DONE := FALSE;
       "DB8000_PART_STATUS".UNIT_01.FIXTURE_2.PART_A.STATUS.UNIT_02_STATUS.FACE_R_STATION_3_DONE := FALSE;
       "DB8000_PART_STATUS".UNIT_01.FIXTURE_2.PART_A.STATUS.UNIT_02_STATUS.FACE_R_STATION_4_DONE := FALSE;
       "DB8000_PART_STATUS".UNIT_01.FIXTURE_2.PART_A.STATUS.CELL_STATUS.U02_DONE_IN_TRANSIT := FALSE;
       "DB8000_PART_STATUS".UNIT_01.FIXTURE_2.PART_A.STATUS.CELL_STATUS.COOLING_DONE := FALSE;
       "DB8000_PART_STATUS".UNIT_01.FIXTURE_2.PART_A.STATUS.CELL_STATUS.INSPECTION_DONE := FALSE;
       "DB8000_PART_STATUS".UNIT_01.FIXTURE_2.PART_A.STATUS.UNIT_01_STATUS.PROCESSED_IN_F2 := FALSE;
       "DB8000_PART_STATUS".UNIT_01.FIXTURE_2.PART_A.STATUS.CELL_STATUS.U01_ONE_FACE_DONE := FALSE;
       "DB8000_PART_STATUS".UNIT_01.FIXTURE_2.PART_A.STATUS.CELL_STATUS.U01_DONE := FALSE;
   END_IF;
   IF #_w3 AND "DB8000_PART_STATUS".HMI.UNIT_01_GOOD_PART AND "DB8000_PART_STATUS".UNIT_01.FIXTURE_2.PART_A.STATUS.PRESENT THEN
       "DB8000_PART_STATUS".UNIT_01.FIXTURE_2.PART_A.STATUS.OK := TRUE;
       "DB8000_PART_STATUS".UNIT_01.FIXTURE_2.PART_A.STATUS.PART_REJECTED := FALSE;
   END_IF;
   IF #_w3 AND "DB8000_PART_STATUS".HMI.UNIT_01_REJECT_PART AND "DB8000_PART_STATUS".UNIT_01.FIXTURE_2.PART_A.STATUS.PRESENT THEN
       "DB8000_PART_STATUS".UNIT_01.FIXTURE_2.PART_A.STATUS.PART_REJECTED := TRUE;
       "DB8000_PART_STATUS".UNIT_01.FIXTURE_2.PART_A.STATUS.OK := FALSE;
   END_IF;
   IF #_w3 AND "DB8000_PART_STATUS".HMI.UNIT_01_MASTER_PART AND "DB8000_PART_STATUS".UNIT_01.FIXTURE_2.PART_A.STATUS.PRESENT THEN
       "DB8000_PART_STATUS".UNIT_01.FIXTURE_2.PART_A.STATUS.MASTER_PART := TRUE;
   END_IF;
   #_w5 := "DB2001_MODES_GENERAL".GENERAL.MANUAL_SELECTED AND ("DB8000_PART_STATUS".HMI.PART_STATUS_FIXTURES_LIST = 3) AND ("DB4000_FIX_TABLE_POSITIONS".UNIT_01.FIXTURE_3.IN_LOAD_UNLOAD_STATION_1 OR "M_DUMMY_ON");
   #_w6 := #_w5 AND "DB8000_PART_STATUS".HMI.UNIT_01_PART_PRESENT;
   IF #_w6 THEN
       "DB8000_PART_STATUS".UNIT_01.FIXTURE_3.PART_A.PART_ID := "DB2099_MANUAL_LOAD_DMC".DMC_ARRAY_CHAR_UNIT_01;
       "DB8000_PART_STATUS".UNIT_01.FIXTURE_3.PART_A.STATUS.PRESENT := TRUE;
       "DB8000_PART_STATUS".UNIT_01.FIXTURE_3.PART_A.STATUS.PART_REJECTED := TRUE;
   END_IF;
   IF #_w6 AND ("DB8000_PART_STATUS".HMI.PART_STATUS_PART_STATUS_LIST = 1) THEN
       "DB8000_PART_STATUS".UNIT_01.FIXTURE_3.PART_A.STATUS.CELL_STATUS.NEW_IN_TRANSIT := TRUE;
   END_IF;
   IF #_w6 AND ("DB8000_PART_STATUS".HMI.PART_STATUS_PART_STATUS_LIST = 2) THEN
       "DB8000_PART_STATUS".UNIT_01.FIXTURE_3.PART_A.STATUS.UNIT_01_STATUS.FACE_N_STATION_3_DONE := TRUE;
   END_IF;
   IF #_w6 AND ("DB8000_PART_STATUS".HMI.PART_STATUS_PART_STATUS_LIST = 3) THEN
       "DB8000_PART_STATUS".UNIT_01.FIXTURE_3.PART_A.STATUS.UNIT_01_STATUS.FACE_N_STATION_4_DONE := TRUE;
   END_IF;
   IF #_w6 AND ("DB8000_PART_STATUS".HMI.PART_STATUS_PART_STATUS_LIST = 4) THEN
       "DB8000_PART_STATUS".UNIT_01.FIXTURE_3.PART_A.STATUS.CELL_STATUS.U01_ONE_FACE_DONE_ROTATED := TRUE;
   END_IF;
   IF #_w6 AND ("DB8000_PART_STATUS".HMI.PART_STATUS_PART_STATUS_LIST = 5) THEN
       "DB8000_PART_STATUS".UNIT_01.FIXTURE_3.PART_A.STATUS.UNIT_01_STATUS.FACE_R_STATION_3_DONE := TRUE;
   END_IF;
   IF #_w6 AND ("DB8000_PART_STATUS".HMI.PART_STATUS_PART_STATUS_LIST = 6) THEN
       "DB8000_PART_STATUS".UNIT_01.FIXTURE_3.PART_A.STATUS.UNIT_01_STATUS.FACE_R_STATION_4_DONE := TRUE;
   END_IF;
   IF #_w6 AND ("DB8000_PART_STATUS".HMI.PART_STATUS_PART_STATUS_LIST = 7) THEN
       "DB8000_PART_STATUS".UNIT_01.FIXTURE_3.PART_A.STATUS.CELL_STATUS.U01_DONE_IN_TRANSIT := TRUE;
   END_IF;
   IF #_w6 AND ("DB8000_PART_STATUS".HMI.PART_STATUS_PART_STATUS_LIST = 8) THEN
       "DB8000_PART_STATUS".UNIT_01.FIXTURE_3.PART_A.STATUS.UNIT_02_STATUS.FACE_N_STATION_2_DONE := TRUE;
   END_IF;
   IF #_w6 AND ("DB8000_PART_STATUS".HMI.PART_STATUS_PART_STATUS_LIST = 9) THEN
       "DB8000_PART_STATUS".UNIT_01.FIXTURE_3.PART_A.STATUS.UNIT_02_STATUS.FACE_N_STATION_3_DONE := TRUE;
   END_IF;
   IF #_w6 AND ("DB8000_PART_STATUS".HMI.PART_STATUS_PART_STATUS_LIST = 10) THEN
       "DB8000_PART_STATUS".UNIT_01.FIXTURE_3.PART_A.STATUS.UNIT_02_STATUS.FACE_N_STATION_4_DONE := TRUE;
   END_IF;
   IF #_w6 AND ("DB8000_PART_STATUS".HMI.PART_STATUS_PART_STATUS_LIST = 11) THEN
       "DB8000_PART_STATUS".UNIT_01.FIXTURE_3.PART_A.STATUS.CELL_STATUS.U02_ONE_FACE_DONE_ROTATED := TRUE;
   END_IF;
   IF #_w6 AND ("DB8000_PART_STATUS".HMI.PART_STATUS_PART_STATUS_LIST = 12) THEN
       "DB8000_PART_STATUS".UNIT_01.FIXTURE_3.PART_A.STATUS.UNIT_02_STATUS.FACE_R_STATION_2_DONE := TRUE;
   END_IF;
   IF #_w6 AND ("DB8000_PART_STATUS".HMI.PART_STATUS_PART_STATUS_LIST = 13) THEN
       "DB8000_PART_STATUS".UNIT_01.FIXTURE_3.PART_A.STATUS.UNIT_02_STATUS.FACE_R_STATION_3_DONE := TRUE;
   END_IF;
   IF #_w6 AND ("DB8000_PART_STATUS".HMI.PART_STATUS_PART_STATUS_LIST = 14) THEN
       "DB8000_PART_STATUS".UNIT_01.FIXTURE_3.PART_A.STATUS.UNIT_02_STATUS.FACE_R_STATION_4_DONE := TRUE;
   END_IF;
   IF #_w6 AND ("DB8000_PART_STATUS".HMI.PART_STATUS_PART_STATUS_LIST = 15) THEN
       "DB8000_PART_STATUS".UNIT_01.FIXTURE_3.PART_A.STATUS.CELL_STATUS.U02_DONE_IN_TRANSIT := TRUE;
   END_IF;
   IF #_w6 AND ("DB8000_PART_STATUS".HMI.PART_STATUS_PART_STATUS_LIST = 16) THEN
       "DB8000_PART_STATUS".UNIT_01.FIXTURE_3.PART_A.STATUS.CELL_STATUS.COOLING_DONE := TRUE;
   END_IF;
   IF #_w6 AND ("DB8000_PART_STATUS".HMI.PART_STATUS_PART_STATUS_LIST = 17) THEN
       "DB8000_PART_STATUS".UNIT_01.FIXTURE_3.PART_A.STATUS.CELL_STATUS.INSPECTION_DONE := TRUE;
   END_IF;
   IF #_w6 AND ("DB8000_PART_STATUS".HMI.PART_STATUS_PART_STATUS_LIST = 99) THEN
       "DB8000_PART_STATUS".UNIT_01.FIXTURE_3.PART_A.STATUS.MASTER_PART := TRUE;
   END_IF;
   IF #_w5 AND "DB8000_PART_STATUS".HMI.UNIT_01_REMOVE_PART THEN
       "DB2700_UNIT_01_FIXTURE_3".INPUT_PART_A_PRESENT_MEM := FALSE;
       "DB8000_PART_STATUS".UNIT_01.FIXTURE_3.PART_A.STATUS.PRESENT := FALSE;
       "DB8000_PART_STATUS".UNIT_01.FIXTURE_3.PART_A.STATUS.PART_REJECTED := FALSE;
       "DB8000_PART_STATUS".UNIT_01.FIXTURE_3.PART_A.STATUS.MASTER_PART := FALSE;
       "DB8000_PART_STATUS".UNIT_01.FIXTURE_3.PART_A.STATUS.CELL_STATUS.NEW_IN_TRANSIT := FALSE;
       "DB8000_PART_STATUS".UNIT_01.FIXTURE_3.PART_A.STATUS.UNIT_01_STATUS.FACE_N_STATION_3_DONE := FALSE;
       "DB8000_PART_STATUS".UNIT_01.FIXTURE_3.PART_A.STATUS.UNIT_01_STATUS.FACE_N_STATION_4_DONE := FALSE;
       "DB8000_PART_STATUS".UNIT_01.FIXTURE_3.PART_A.STATUS.CELL_STATUS.U01_ONE_FACE_DONE_ROTATED := FALSE;
       "DB8000_PART_STATUS".UNIT_01.FIXTURE_3.PART_A.STATUS.UNIT_01_STATUS.FACE_R_STATION_3_DONE := FALSE;
       "DB8000_PART_STATUS".UNIT_01.FIXTURE_3.PART_A.STATUS.UNIT_01_STATUS.FACE_R_STATION_4_DONE := FALSE;
       "DB8000_PART_STATUS".UNIT_01.FIXTURE_3.PART_A.STATUS.CELL_STATUS.U01_DONE_IN_TRANSIT := FALSE;
       "DB8000_PART_STATUS".UNIT_01.FIXTURE_3.PART_A.STATUS.UNIT_02_STATUS.FACE_N_STATION_2_DONE := FALSE;
       "DB8000_PART_STATUS".UNIT_01.FIXTURE_3.PART_A.STATUS.UNIT_02_STATUS.FACE_N_STATION_3_DONE := FALSE;
       "DB8000_PART_STATUS".UNIT_01.FIXTURE_3.PART_A.STATUS.UNIT_02_STATUS.FACE_N_STATION_4_DONE := FALSE;
       "DB8000_PART_STATUS".UNIT_01.FIXTURE_3.PART_A.STATUS.CELL_STATUS.U02_ONE_FACE_DONE_ROTATED := FALSE;
       "DB8000_PART_STATUS".UNIT_01.FIXTURE_3.PART_A.STATUS.UNIT_02_STATUS.FACE_R_STATION_2_DONE := FALSE;
       "DB8000_PART_STATUS".UNIT_01.FIXTURE_3.PART_A.STATUS.UNIT_02_STATUS.FACE_R_STATION_3_DONE := FALSE;
       "DB8000_PART_STATUS".UNIT_01.FIXTURE_3.PART_A.STATUS.UNIT_02_STATUS.FACE_R_STATION_4_DONE := FALSE;
       "DB8000_PART_STATUS".UNIT_01.FIXTURE_3.PART_A.STATUS.CELL_STATUS.U02_DONE_IN_TRANSIT := FALSE;
       "DB8000_PART_STATUS".UNIT_01.FIXTURE_3.PART_A.STATUS.CELL_STATUS.COOLING_DONE := FALSE;
       "DB8000_PART_STATUS".UNIT_01.FIXTURE_3.PART_A.STATUS.CELL_STATUS.INSPECTION_DONE := FALSE;
       "DB8000_PART_STATUS".UNIT_01.FIXTURE_3.PART_A.STATUS.UNIT_01_STATUS.PROCESSED_IN_F3 := FALSE;
       "DB8000_PART_STATUS".UNIT_01.FIXTURE_3.PART_A.STATUS.CELL_STATUS.U01_ONE_FACE_DONE := FALSE;
       "DB8000_PART_STATUS".UNIT_01.FIXTURE_3.PART_A.STATUS.CELL_STATUS.U01_DONE := FALSE;
   END_IF;
   IF #_w5 AND "DB8000_PART_STATUS".HMI.UNIT_01_GOOD_PART AND "DB8000_PART_STATUS".UNIT_01.FIXTURE_3.PART_A.STATUS.PRESENT THEN
       "DB8000_PART_STATUS".UNIT_01.FIXTURE_3.PART_A.STATUS.OK := TRUE;
       "DB8000_PART_STATUS".UNIT_01.FIXTURE_3.PART_A.STATUS.PART_REJECTED := FALSE;
   END_IF;
   IF #_w5 AND "DB8000_PART_STATUS".HMI.UNIT_01_REJECT_PART AND "DB8000_PART_STATUS".UNIT_01.FIXTURE_3.PART_A.STATUS.PRESENT THEN
       "DB8000_PART_STATUS".UNIT_01.FIXTURE_3.PART_A.STATUS.PART_REJECTED := TRUE;
       "DB8000_PART_STATUS".UNIT_01.FIXTURE_3.PART_A.STATUS.OK := FALSE;
   END_IF;
   IF #_w5 AND "DB8000_PART_STATUS".HMI.UNIT_01_MASTER_PART AND "DB8000_PART_STATUS".UNIT_01.FIXTURE_3.PART_A.STATUS.PRESENT THEN
       "DB8000_PART_STATUS".UNIT_01.FIXTURE_3.PART_A.STATUS.MASTER_PART := TRUE;
   END_IF;
   #_w7 := "DB2001_MODES_GENERAL".GENERAL.MANUAL_SELECTED AND ("DB8000_PART_STATUS".HMI.PART_STATUS_FIXTURES_LIST = 4) AND ("DB4000_FIX_TABLE_POSITIONS".UNIT_01.FIXTURE_4.IN_LOAD_UNLOAD_STATION_1 OR "M_DUMMY_ON");
   #_w8 := #_w7 AND "DB8000_PART_STATUS".HMI.UNIT_01_PART_PRESENT;
   IF #_w8 THEN
       "DB8000_PART_STATUS".UNIT_01.FIXTURE_4.PART_A.PART_ID := "DB2099_MANUAL_LOAD_DMC".DMC_ARRAY_CHAR_UNIT_01;
       "DB8000_PART_STATUS".UNIT_01.FIXTURE_4.PART_A.STATUS.PRESENT := TRUE;
       "DB8000_PART_STATUS".UNIT_01.FIXTURE_4.PART_A.STATUS.PART_REJECTED := TRUE;
   END_IF;
   IF #_w8 AND ("DB8000_PART_STATUS".HMI.PART_STATUS_PART_STATUS_LIST = 1) THEN
       "DB8000_PART_STATUS".UNIT_01.FIXTURE_4.PART_A.STATUS.CELL_STATUS.NEW_IN_TRANSIT := TRUE;
   END_IF;
   IF #_w8 AND ("DB8000_PART_STATUS".HMI.PART_STATUS_PART_STATUS_LIST = 2) THEN
       "DB8000_PART_STATUS".UNIT_01.FIXTURE_4.PART_A.STATUS.UNIT_01_STATUS.FACE_N_STATION_3_DONE := TRUE;
   END_IF;
   IF #_w8 AND ("DB8000_PART_STATUS".HMI.PART_STATUS_PART_STATUS_LIST = 3) THEN
       "DB8000_PART_STATUS".UNIT_01.FIXTURE_4.PART_A.STATUS.UNIT_01_STATUS.FACE_N_STATION_4_DONE := TRUE;
   END_IF;
   IF #_w8 AND ("DB8000_PART_STATUS".HMI.PART_STATUS_PART_STATUS_LIST = 4) THEN
       "DB8000_PART_STATUS".UNIT_01.FIXTURE_4.PART_A.STATUS.CELL_STATUS.U01_ONE_FACE_DONE_ROTATED := TRUE;
   END_IF;
   IF #_w8 AND ("DB8000_PART_STATUS".HMI.PART_STATUS_PART_STATUS_LIST = 5) THEN
       "DB8000_PART_STATUS".UNIT_01.FIXTURE_4.PART_A.STATUS.UNIT_01_STATUS.FACE_R_STATION_3_DONE := TRUE;
   END_IF;
   IF #_w8 AND ("DB8000_PART_STATUS".HMI.PART_STATUS_PART_STATUS_LIST = 6) THEN
       "DB8000_PART_STATUS".UNIT_01.FIXTURE_4.PART_A.STATUS.UNIT_01_STATUS.FACE_R_STATION_4_DONE := TRUE;
   END_IF;
   IF #_w8 AND ("DB8000_PART_STATUS".HMI.PART_STATUS_PART_STATUS_LIST = 7) THEN
       "DB8000_PART_STATUS".UNIT_01.FIXTURE_4.PART_A.STATUS.CELL_STATUS.U01_DONE_IN_TRANSIT := TRUE;
   END_IF;
   IF #_w8 AND ("DB8000_PART_STATUS".HMI.PART_STATUS_PART_STATUS_LIST = 8) THEN
       "DB8000_PART_STATUS".UNIT_01.FIXTURE_4.PART_A.STATUS.UNIT_02_STATUS.FACE_N_STATION_2_DONE := TRUE;
   END_IF;
   IF #_w8 AND ("DB8000_PART_STATUS".HMI.PART_STATUS_PART_STATUS_LIST = 9) THEN
       "DB8000_PART_STATUS".UNIT_01.FIXTURE_4.PART_A.STATUS.UNIT_02_STATUS.FACE_N_STATION_3_DONE := TRUE;
   END_IF;
   IF #_w8 AND ("DB8000_PART_STATUS".HMI.PART_STATUS_PART_STATUS_LIST = 10) THEN
       "DB8000_PART_STATUS".UNIT_01.FIXTURE_4.PART_A.STATUS.UNIT_02_STATUS.FACE_N_STATION_4_DONE := TRUE;
   END_IF;
   IF #_w8 AND ("DB8000_PART_STATUS".HMI.PART_STATUS_PART_STATUS_LIST = 11) THEN
       "DB8000_PART_STATUS".UNIT_01.FIXTURE_4.PART_A.STATUS.CELL_STATUS.U02_ONE_FACE_DONE_ROTATED := TRUE;
   END_IF;
   IF #_w8 AND ("DB8000_PART_STATUS".HMI.PART_STATUS_PART_STATUS_LIST = 12) THEN
       "DB8000_PART_STATUS".UNIT_01.FIXTURE_4.PART_A.STATUS.UNIT_02_STATUS.FACE_R_STATION_2_DONE := TRUE;
   END_IF;
   IF #_w8 AND ("DB8000_PART_STATUS".HMI.PART_STATUS_PART_STATUS_LIST = 13) THEN
       "DB8000_PART_STATUS".UNIT_01.FIXTURE_4.PART_A.STATUS.UNIT_02_STATUS.FACE_R_STATION_3_DONE := TRUE;
   END_IF;
   IF #_w8 AND ("DB8000_PART_STATUS".HMI.PART_STATUS_PART_STATUS_LIST = 14) THEN
       "DB8000_PART_STATUS".UNIT_01.FIXTURE_4.PART_A.STATUS.UNIT_02_STATUS.FACE_R_STATION_4_DONE := TRUE;
   END_IF;
   IF #_w8 AND ("DB8000_PART_STATUS".HMI.PART_STATUS_PART_STATUS_LIST = 15) THEN
       "DB8000_PART_STATUS".UNIT_01.FIXTURE_4.PART_A.STATUS.CELL_STATUS.U02_DONE_IN_TRANSIT := TRUE;
   END_IF;
   IF #_w8 AND ("DB8000_PART_STATUS".HMI.PART_STATUS_PART_STATUS_LIST = 16) THEN
       "DB8000_PART_STATUS".UNIT_01.FIXTURE_4.PART_A.STATUS.CELL_STATUS.COOLING_DONE := TRUE;
   END_IF;
   IF #_w8 AND ("DB8000_PART_STATUS".HMI.PART_STATUS_PART_STATUS_LIST = 17) THEN
       "DB8000_PART_STATUS".UNIT_01.FIXTURE_4.PART_A.STATUS.CELL_STATUS.INSPECTION_DONE := TRUE;
   END_IF;
   IF #_w8 AND ("DB8000_PART_STATUS".HMI.PART_STATUS_PART_STATUS_LIST = 99) THEN
       "DB8000_PART_STATUS".UNIT_01.FIXTURE_4.PART_A.STATUS.MASTER_PART := TRUE;
   END_IF;
   IF #_w7 AND "DB8000_PART_STATUS".HMI.UNIT_01_REMOVE_PART THEN
       "DB2800_UNIT_01_FIXTURE_4".INPUT_PART_A_PRESENT_MEM := FALSE;
       "DB8000_PART_STATUS".UNIT_01.FIXTURE_4.PART_A.STATUS.PRESENT := FALSE;
       "DB8000_PART_STATUS".UNIT_01.FIXTURE_4.PART_A.STATUS.PART_REJECTED := FALSE;
       "DB8000_PART_STATUS".UNIT_01.FIXTURE_4.PART_A.STATUS.MASTER_PART := FALSE;
       "DB8000_PART_STATUS".UNIT_01.FIXTURE_4.PART_A.STATUS.CELL_STATUS.NEW_IN_TRANSIT := FALSE;
       "DB8000_PART_STATUS".UNIT_01.FIXTURE_4.PART_A.STATUS.UNIT_01_STATUS.FACE_N_STATION_3_DONE := FALSE;
       "DB8000_PART_STATUS".UNIT_01.FIXTURE_4.PART_A.STATUS.UNIT_01_STATUS.FACE_N_STATION_4_DONE := FALSE;
       "DB8000_PART_STATUS".UNIT_01.FIXTURE_4.PART_A.STATUS.CELL_STATUS.U01_ONE_FACE_DONE_ROTATED := FALSE;
       "DB8000_PART_STATUS".UNIT_01.FIXTURE_4.PART_A.STATUS.UNIT_01_STATUS.FACE_R_STATION_3_DONE := FALSE;
       "DB8000_PART_STATUS".UNIT_01.FIXTURE_4.PART_A.STATUS.UNIT_01_STATUS.FACE_R_STATION_4_DONE := FALSE;
       "DB8000_PART_STATUS".UNIT_01.FIXTURE_4.PART_A.STATUS.CELL_STATUS.U01_DONE_IN_TRANSIT := FALSE;
       "DB8000_PART_STATUS".UNIT_01.FIXTURE_4.PART_A.STATUS.UNIT_02_STATUS.FACE_N_STATION_2_DONE := FALSE;
       "DB8000_PART_STATUS".UNIT_01.FIXTURE_4.PART_A.STATUS.UNIT_02_STATUS.FACE_N_STATION_3_DONE := FALSE;
       "DB8000_PART_STATUS".UNIT_01.FIXTURE_4.PART_A.STATUS.UNIT_02_STATUS.FACE_N_STATION_4_DONE := FALSE;
       "DB8000_PART_STATUS".UNIT_01.FIXTURE_4.PART_A.STATUS.CELL_STATUS.U02_ONE_FACE_DONE_ROTATED := FALSE;
       "DB8000_PART_STATUS".UNIT_01.FIXTURE_4.PART_A.STATUS.UNIT_02_STATUS.FACE_R_STATION_2_DONE := FALSE;
       "DB8000_PART_STATUS".UNIT_01.FIXTURE_4.PART_A.STATUS.UNIT_02_STATUS.FACE_R_STATION_3_DONE := FALSE;
       "DB8000_PART_STATUS".UNIT_01.FIXTURE_4.PART_A.STATUS.UNIT_02_STATUS.FACE_R_STATION_4_DONE := FALSE;
       "DB8000_PART_STATUS".UNIT_01.FIXTURE_4.PART_A.STATUS.CELL_STATUS.U02_DONE_IN_TRANSIT := FALSE;
       "DB8000_PART_STATUS".UNIT_01.FIXTURE_4.PART_A.STATUS.CELL_STATUS.COOLING_DONE := FALSE;
       "DB8000_PART_STATUS".UNIT_01.FIXTURE_4.PART_A.STATUS.CELL_STATUS.INSPECTION_DONE := FALSE;
       "DB8000_PART_STATUS".UNIT_01.FIXTURE_4.PART_A.STATUS.UNIT_01_STATUS.PROCESSED_IN_F4 := FALSE;
       "DB8000_PART_STATUS".UNIT_01.FIXTURE_4.PART_A.STATUS.CELL_STATUS.U01_ONE_FACE_DONE := FALSE;
       "DB8000_PART_STATUS".UNIT_01.FIXTURE_4.PART_A.STATUS.CELL_STATUS.U01_DONE := FALSE;
   END_IF;
   IF #_w7 AND "DB8000_PART_STATUS".HMI.UNIT_01_GOOD_PART AND "DB8000_PART_STATUS".UNIT_01.FIXTURE_4.PART_A.STATUS.PRESENT THEN
       "DB8000_PART_STATUS".UNIT_01.FIXTURE_4.PART_A.STATUS.OK := TRUE;
       "DB8000_PART_STATUS".UNIT_01.FIXTURE_4.PART_A.STATUS.PART_REJECTED := FALSE;
   END_IF;
   IF #_w7 AND "DB8000_PART_STATUS".HMI.UNIT_01_REJECT_PART AND "DB8000_PART_STATUS".UNIT_01.FIXTURE_4.PART_A.STATUS.PRESENT THEN
       "DB8000_PART_STATUS".UNIT_01.FIXTURE_4.PART_A.STATUS.PART_REJECTED := TRUE;
       "DB8000_PART_STATUS".UNIT_01.FIXTURE_4.PART_A.STATUS.OK := FALSE;
   END_IF;
   IF #_w7 AND "DB8000_PART_STATUS".HMI.UNIT_01_MASTER_PART AND "DB8000_PART_STATUS".UNIT_01.FIXTURE_4.PART_A.STATUS.PRESENT THEN
       "DB8000_PART_STATUS".UNIT_02.FIXTURE_4.PART_A.STATUS.MASTER_PART := TRUE;
   END_IF;
END_REGION

REGION Network 3: OPERATOR HELP
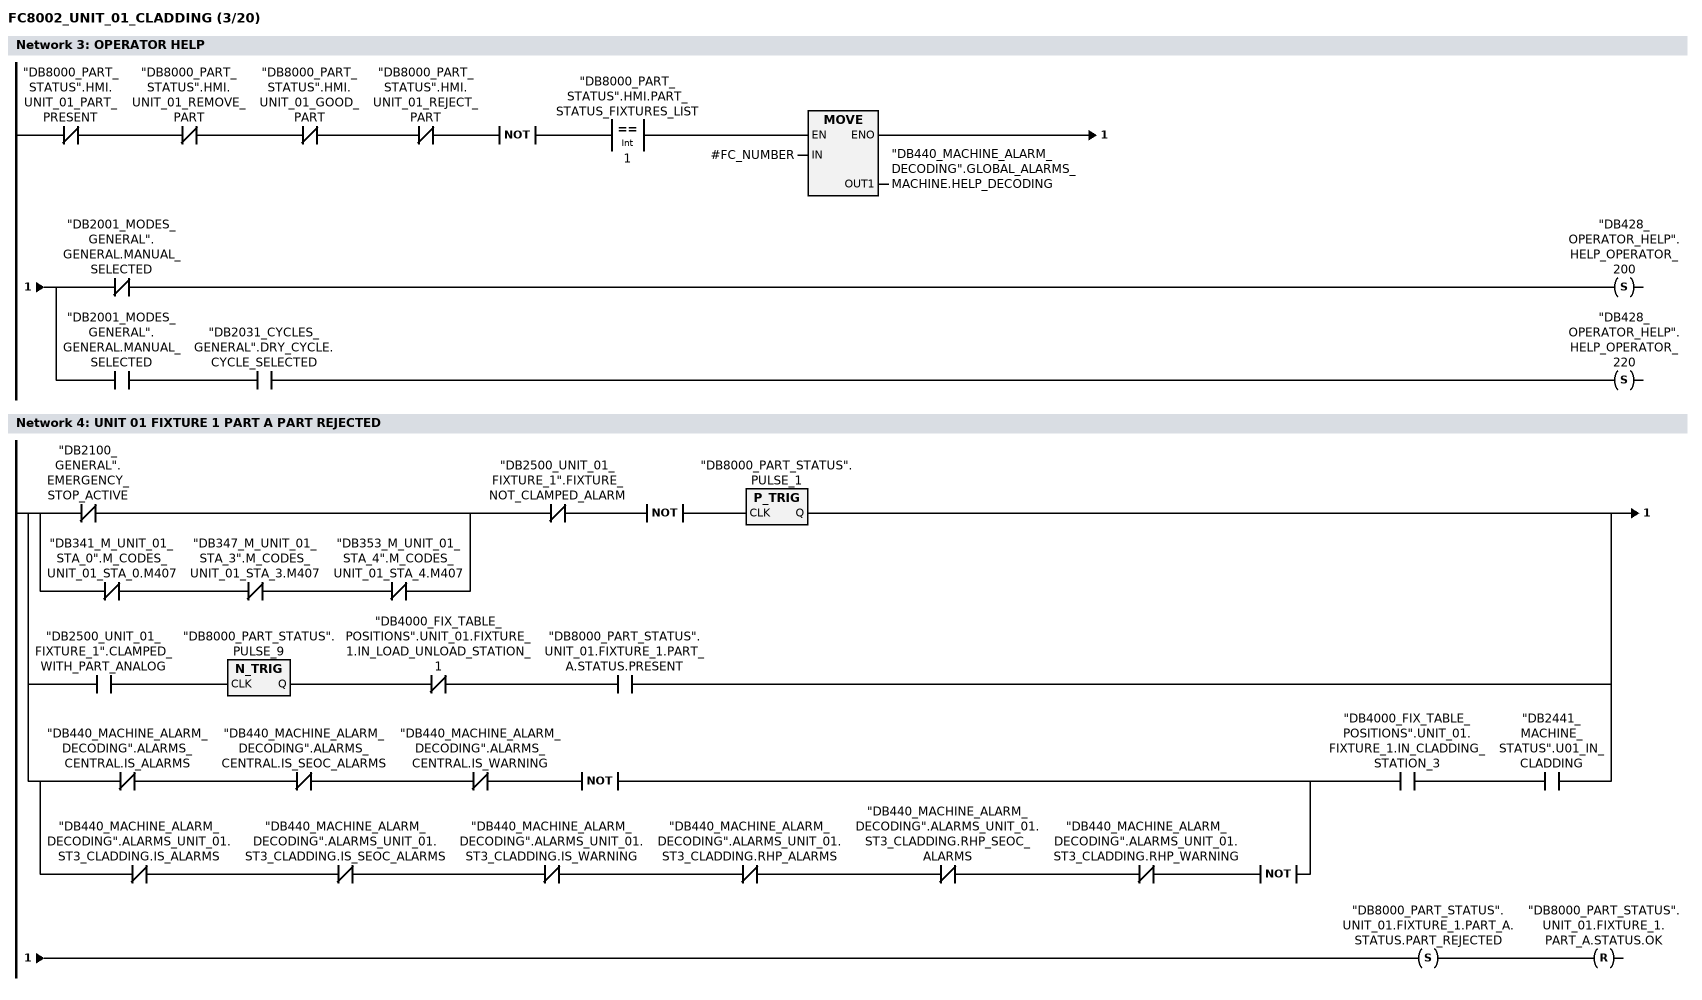
   RUNG wire#powerrail
      I_Contact( "DB8000_PART_STATUS".HMI.UNIT_01_PART_PRESENT )
      I_Contact( "DB8000_PART_STATUS".HMI.UNIT_01_REMOVE_PART )
      I_Contact( "DB8000_PART_STATUS".HMI.UNIT_01_GOOD_PART )
      I_Contact( "DB8000_PART_STATUS".HMI.UNIT_01_REJECT_PART )
      Not()
      { S7_Templates := "SrcType := Int" } EQ_Contact(in1 := "DB8000_PART_STATUS".HMI.PART_STATUS_FIXTURES_LIST, in2 := 1)
      { S7_GenerateENO := "TRUE" } Move(in := #FC_NUMBER, out1 => "DB440_MACHINE_ALARM_DECODING".GLOBAL_ALARMS_MACHINE.HELP_DECODING)
      wire#w1
      I_Contact( "DB2001_MODES_GENERAL".GENERAL.MANUAL_SELECTED )
      S_Coil( "DB428_OPERATOR_HELP".HELP_OPERATOR_200 )
   END_RUNG
   RUNG wire#w1
      Contact( "DB2001_MODES_GENERAL".GENERAL.MANUAL_SELECTED )
      Contact( "DB2031_CYCLES_GENERAL".DRY_CYCLE.CYCLE_SELECTED )
      S_Coil( "DB428_OPERATOR_HELP".HELP_OPERATOR_220 )
   END_RUNG
   // the same network as SCL:
   // ENO of a box is taken as its EN; it also drops when the box reports an error
   #_w1 := NOT (NOT "DB8000_PART_STATUS".HMI.UNIT_01_PART_PRESENT AND NOT "DB8000_PART_STATUS".HMI.UNIT_01_REMOVE_PART AND NOT "DB8000_PART_STATUS".HMI.UNIT_01_GOOD_PART AND NOT "DB8000_PART_STATUS".HMI.UNIT_01_REJECT_PART) AND ("DB8000_PART_STATUS".HMI.PART_STATUS_FIXTURES_LIST = 1);
   IF #_w1 THEN "DB440_MACHINE_ALARM_DECODING".GLOBAL_ALARMS_MACHINE.HELP_DECODING := #FC_NUMBER; END_IF;
   IF #_w1 AND NOT "DB2001_MODES_GENERAL".GENERAL.MANUAL_SELECTED THEN
       "DB428_OPERATOR_HELP".HELP_OPERATOR_200 := TRUE;
   END_IF;
   IF #_w1 AND "DB2001_MODES_GENERAL".GENERAL.MANUAL_SELECTED AND "DB2031_CYCLES_GENERAL".DRY_CYCLE.CYCLE_SELECTED THEN
       "DB428_OPERATOR_HELP".HELP_OPERATOR_220 := TRUE;
   END_IF;
END_REGION

REGION Network 4: UNIT 01 FIXTURE 1 PART A PART REJECTED
   RUNG wire#powerrail
      I_Contact( "DB2100_GENERAL".EMERGENCY_STOP_ACTIVE )
      wire#w1
      I_Contact( "DB2500_UNIT_01_FIXTURE_1".FIXTURE_NOT_CLAMPED_ALARM )
      Not()
      P_Trig( "DB8000_PART_STATUS".PULSE_1 )
      wire#w2
      S_Coil( "DB8000_PART_STATUS".UNIT_01.FIXTURE_1.PART_A.STATUS.PART_REJECTED )
      R_Coil( "DB8000_PART_STATUS".UNIT_01.FIXTURE_1.PART_A.STATUS.OK )
   END_RUNG
   RUNG wire#powerrail
      I_Contact( "DB341_M_UNIT_01_STA_0".M_CODES_UNIT_01_STA_0.M407 )
      I_Contact( "DB347_M_UNIT_01_STA_3".M_CODES_UNIT_01_STA_3.M407 )
      I_Contact( "DB353_M_UNIT_01_STA_4".M_CODES_UNIT_01_STA_4.M407 )
   END_RUNG wire#w1
   RUNG wire#powerrail
      Contact( "DB2500_UNIT_01_FIXTURE_1".CLAMPED_WITH_PART_ANALOG )
      N_Trig( "DB8000_PART_STATUS".PULSE_9 )
      I_Contact( "DB4000_FIX_TABLE_POSITIONS".UNIT_01.FIXTURE_1.IN_LOAD_UNLOAD_STATION_1 )
      Contact( "DB8000_PART_STATUS".UNIT_01.FIXTURE_1.PART_A.STATUS.PRESENT )
   END_RUNG wire#w2
   RUNG wire#powerrail
      I_Contact( "DB440_MACHINE_ALARM_DECODING".ALARMS_CENTRAL.IS_ALARMS )
      I_Contact( "DB440_MACHINE_ALARM_DECODING".ALARMS_CENTRAL.IS_SEOC_ALARMS )
      I_Contact( "DB440_MACHINE_ALARM_DECODING".ALARMS_CENTRAL.IS_WARNING )
      Not()
      wire#w3
      Contact( "DB4000_FIX_TABLE_POSITIONS".UNIT_01.FIXTURE_1.IN_CLADDING_STATION_3 )
      Contact( "DB2441_MACHINE_STATUS".U01_IN_CLADDING )
   END_RUNG wire#w2
   RUNG wire#powerrail
      I_Contact( "DB440_MACHINE_ALARM_DECODING".ALARMS_UNIT_01.ST3_CLADDING.IS_ALARMS )
      I_Contact( "DB440_MACHINE_ALARM_DECODING".ALARMS_UNIT_01.ST3_CLADDING.IS_SEOC_ALARMS )
      I_Contact( "DB440_MACHINE_ALARM_DECODING".ALARMS_UNIT_01.ST3_CLADDING.IS_WARNING )
      I_Contact( "DB440_MACHINE_ALARM_DECODING".ALARMS_UNIT_01.ST3_CLADDING.RHP_ALARMS )
      I_Contact( "DB440_MACHINE_ALARM_DECODING".ALARMS_UNIT_01.ST3_CLADDING.RHP_SEOC_ALARMS )
      I_Contact( "DB440_MACHINE_ALARM_DECODING".ALARMS_UNIT_01.ST3_CLADDING.RHP_WARNING )
      Not()
   END_RUNG wire#w3
   // the same network as SCL:
   #_w1 := NOT ((NOT "DB2100_GENERAL".EMERGENCY_STOP_ACTIVE OR (NOT "DB341_M_UNIT_01_STA_0".M_CODES_UNIT_01_STA_0.M407 AND NOT "DB347_M_UNIT_01_STA_3".M_CODES_UNIT_01_STA_3.M407 AND NOT "DB353_M_UNIT_01_STA_4".M_CODES_UNIT_01_STA_4.M407)) AND NOT "DB2500_UNIT_01_FIXTURE_1".FIXTURE_NOT_CLAMPED_ALARM);
   #_w2 := #_w1 AND NOT "DB8000_PART_STATUS".PULSE_1;   // rising edge
   "DB8000_PART_STATUS".PULSE_1 := #_w1;
   #_w3 := NOT "DB2500_UNIT_01_FIXTURE_1".CLAMPED_WITH_PART_ANALOG AND "DB8000_PART_STATUS".PULSE_9;   // falling edge
   "DB8000_PART_STATUS".PULSE_9 := "DB2500_UNIT_01_FIXTURE_1".CLAMPED_WITH_PART_ANALOG;
   IF #_w2 OR (#_w3 AND NOT "DB4000_FIX_TABLE_POSITIONS".UNIT_01.FIXTURE_1.IN_LOAD_UNLOAD_STATION_1 AND "DB8000_PART_STATUS".UNIT_01.FIXTURE_1.PART_A.STATUS.PRESENT) OR ((NOT (NOT "DB440_MACHINE_ALARM_DECODING".ALARMS_CENTRAL.IS_ALARMS AND NOT "DB440_MACHINE_ALARM_DECODING".ALARMS_CENTRAL.IS_SEOC_ALARMS AND NOT "DB440_MACHINE_ALARM_DECODING".ALARMS_CENTRAL.IS_WARNING) OR NOT (NOT "DB440_MACHINE_ALARM_DECODING".ALARMS_UNIT_01.ST3_CLADDING.IS_ALARMS AND NOT "DB440_MACHINE_ALARM_DECODING".ALARMS_UNIT_01.ST3_CLADDING.IS_SEOC_ALARMS AND NOT "DB440_MACHINE_ALARM_DECODING".ALARMS_UNIT_01.ST3_CLADDING.IS_WARNING AND NOT "DB440_MACHINE_ALARM_DECODING".ALARMS_UNIT_01.ST3_CLADDING.RHP_ALARMS AND NOT "DB440_MACHINE_ALARM_DECODING".ALARMS_UNIT_01.ST3_CLADDING.RHP_SEOC_ALARMS AND NOT "DB440_MACHINE_ALARM_DECODING".ALARMS_UNIT_01.ST3_CLADDING.RHP_WARNING)) AND "DB4000_FIX_TABLE_POSITIONS".UNIT_01.FIXTURE_1.IN_CLADDING_STATION_3 AND "DB2441_MACHINE_STATUS".U01_IN_CLADDING) THEN
       "DB8000_PART_STATUS".UNIT_01.FIXTURE_1.PART_A.STATUS.PART_REJECTED := TRUE;
       "DB8000_PART_STATUS".UNIT_01.FIXTURE_1.PART_A.STATUS.OK := FALSE;
   END_IF;
END_REGION

REGION Network 5: UNIT 01 FIXTURE 2 PART A PART REJECTED
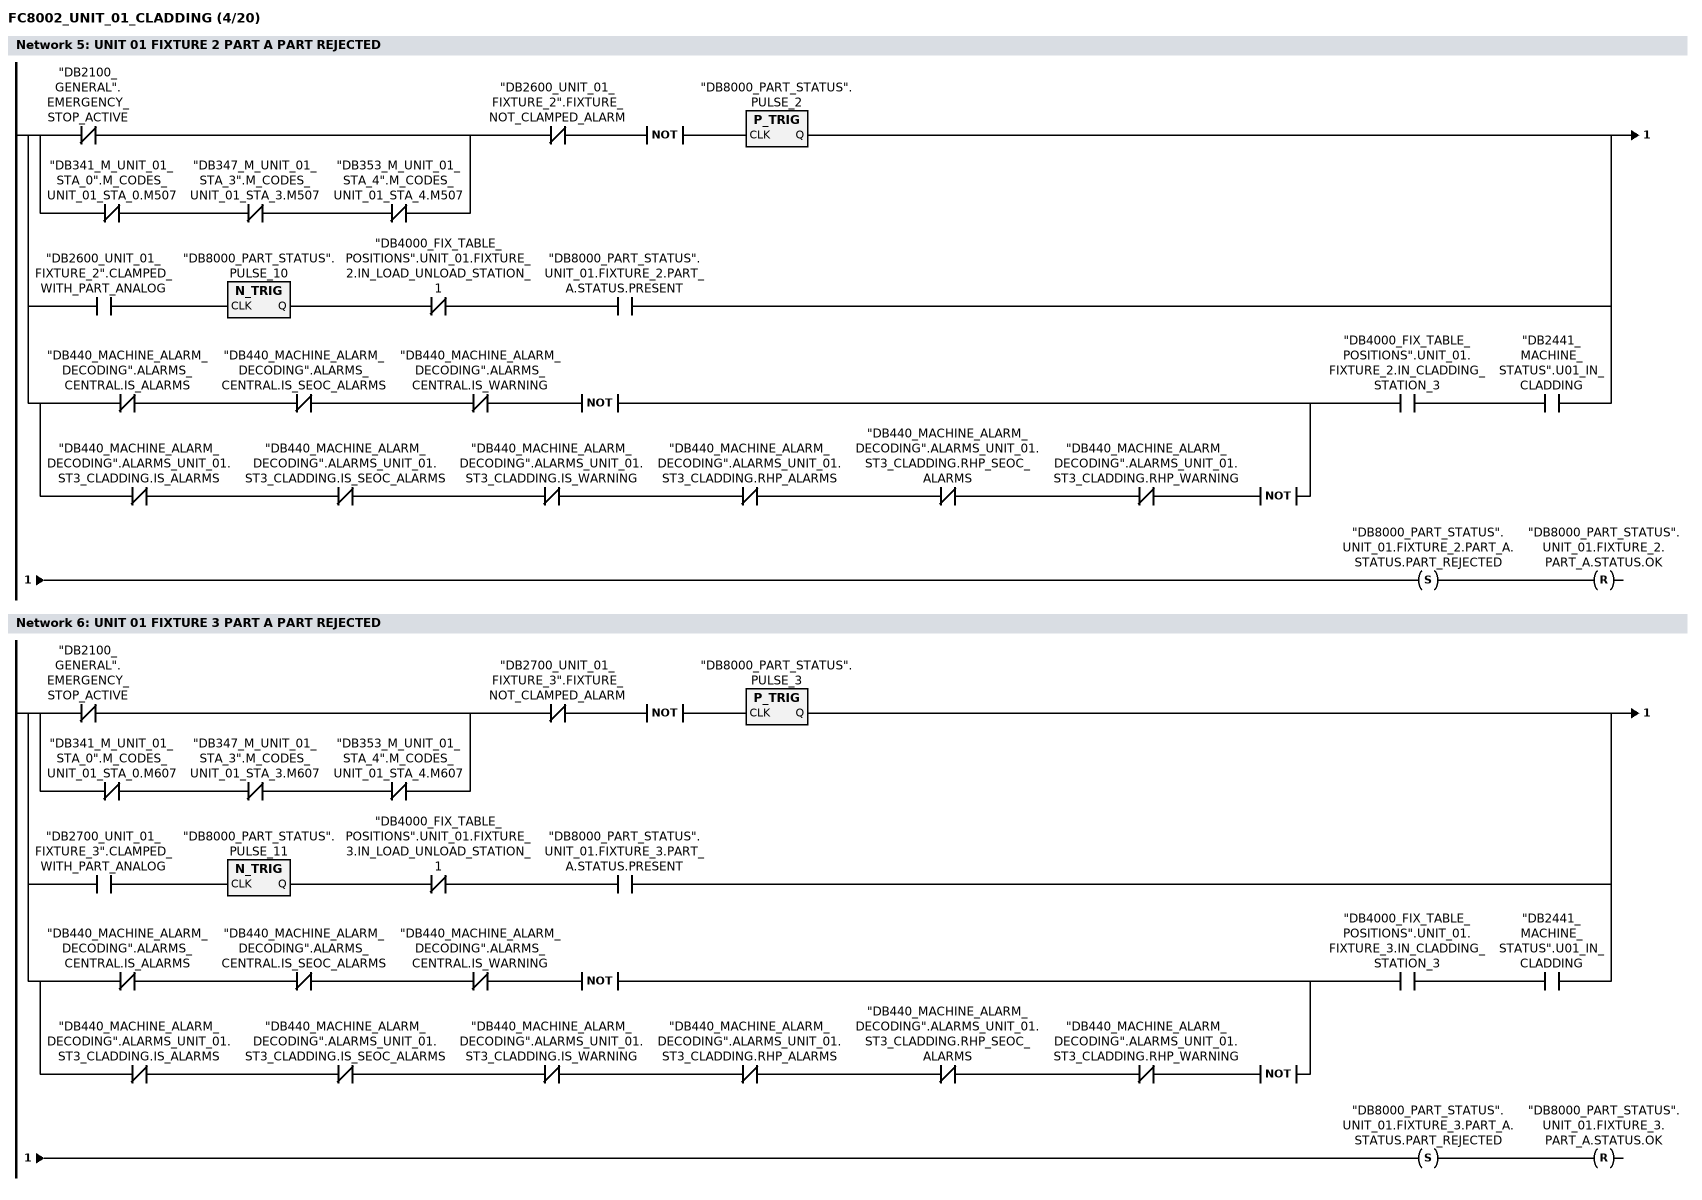
   RUNG wire#powerrail
      I_Contact( "DB2100_GENERAL".EMERGENCY_STOP_ACTIVE )
      wire#w1
      I_Contact( "DB2600_UNIT_01_FIXTURE_2".FIXTURE_NOT_CLAMPED_ALARM )
      Not()
      P_Trig( "DB8000_PART_STATUS".PULSE_2 )
      wire#w2
      S_Coil( "DB8000_PART_STATUS".UNIT_01.FIXTURE_2.PART_A.STATUS.PART_REJECTED )
      R_Coil( "DB8000_PART_STATUS".UNIT_01.FIXTURE_2.PART_A.STATUS.OK )
   END_RUNG
   RUNG wire#powerrail
      I_Contact( "DB341_M_UNIT_01_STA_0".M_CODES_UNIT_01_STA_0.M507 )
      I_Contact( "DB347_M_UNIT_01_STA_3".M_CODES_UNIT_01_STA_3.M507 )
      I_Contact( "DB353_M_UNIT_01_STA_4".M_CODES_UNIT_01_STA_4.M507 )
   END_RUNG wire#w1
   RUNG wire#powerrail
      Contact( "DB2600_UNIT_01_FIXTURE_2".CLAMPED_WITH_PART_ANALOG )
      N_Trig( "DB8000_PART_STATUS".PULSE_10 )
      I_Contact( "DB4000_FIX_TABLE_POSITIONS".UNIT_01.FIXTURE_2.IN_LOAD_UNLOAD_STATION_1 )
      Contact( "DB8000_PART_STATUS".UNIT_01.FIXTURE_2.PART_A.STATUS.PRESENT )
   END_RUNG wire#w2
   RUNG wire#powerrail
      I_Contact( "DB440_MACHINE_ALARM_DECODING".ALARMS_CENTRAL.IS_ALARMS )
      I_Contact( "DB440_MACHINE_ALARM_DECODING".ALARMS_CENTRAL.IS_SEOC_ALARMS )
      I_Contact( "DB440_MACHINE_ALARM_DECODING".ALARMS_CENTRAL.IS_WARNING )
      Not()
      wire#w3
      Contact( "DB4000_FIX_TABLE_POSITIONS".UNIT_01.FIXTURE_2.IN_CLADDING_STATION_3 )
      Contact( "DB2441_MACHINE_STATUS".U01_IN_CLADDING )
   END_RUNG wire#w2
   RUNG wire#powerrail
      I_Contact( "DB440_MACHINE_ALARM_DECODING".ALARMS_UNIT_01.ST3_CLADDING.IS_ALARMS )
      I_Contact( "DB440_MACHINE_ALARM_DECODING".ALARMS_UNIT_01.ST3_CLADDING.IS_SEOC_ALARMS )
      I_Contact( "DB440_MACHINE_ALARM_DECODING".ALARMS_UNIT_01.ST3_CLADDING.IS_WARNING )
      I_Contact( "DB440_MACHINE_ALARM_DECODING".ALARMS_UNIT_01.ST3_CLADDING.RHP_ALARMS )
      I_Contact( "DB440_MACHINE_ALARM_DECODING".ALARMS_UNIT_01.ST3_CLADDING.RHP_SEOC_ALARMS )
      I_Contact( "DB440_MACHINE_ALARM_DECODING".ALARMS_UNIT_01.ST3_CLADDING.RHP_WARNING )
      Not()
   END_RUNG wire#w3
   // the same network as SCL:
   #_w1 := NOT ((NOT "DB2100_GENERAL".EMERGENCY_STOP_ACTIVE OR (NOT "DB341_M_UNIT_01_STA_0".M_CODES_UNIT_01_STA_0.M507 AND NOT "DB347_M_UNIT_01_STA_3".M_CODES_UNIT_01_STA_3.M507 AND NOT "DB353_M_UNIT_01_STA_4".M_CODES_UNIT_01_STA_4.M507)) AND NOT "DB2600_UNIT_01_FIXTURE_2".FIXTURE_NOT_CLAMPED_ALARM);
   #_w2 := #_w1 AND NOT "DB8000_PART_STATUS".PULSE_2;   // rising edge
   "DB8000_PART_STATUS".PULSE_2 := #_w1;
   #_w3 := NOT "DB2600_UNIT_01_FIXTURE_2".CLAMPED_WITH_PART_ANALOG AND "DB8000_PART_STATUS".PULSE_10;   // falling edge
   "DB8000_PART_STATUS".PULSE_10 := "DB2600_UNIT_01_FIXTURE_2".CLAMPED_WITH_PART_ANALOG;
   IF #_w2 OR (#_w3 AND NOT "DB4000_FIX_TABLE_POSITIONS".UNIT_01.FIXTURE_2.IN_LOAD_UNLOAD_STATION_1 AND "DB8000_PART_STATUS".UNIT_01.FIXTURE_2.PART_A.STATUS.PRESENT) OR ((NOT (NOT "DB440_MACHINE_ALARM_DECODING".ALARMS_CENTRAL.IS_ALARMS AND NOT "DB440_MACHINE_ALARM_DECODING".ALARMS_CENTRAL.IS_SEOC_ALARMS AND NOT "DB440_MACHINE_ALARM_DECODING".ALARMS_CENTRAL.IS_WARNING) OR NOT (NOT "DB440_MACHINE_ALARM_DECODING".ALARMS_UNIT_01.ST3_CLADDING.IS_ALARMS AND NOT "DB440_MACHINE_ALARM_DECODING".ALARMS_UNIT_01.ST3_CLADDING.IS_SEOC_ALARMS AND NOT "DB440_MACHINE_ALARM_DECODING".ALARMS_UNIT_01.ST3_CLADDING.IS_WARNING AND NOT "DB440_MACHINE_ALARM_DECODING".ALARMS_UNIT_01.ST3_CLADDING.RHP_ALARMS AND NOT "DB440_MACHINE_ALARM_DECODING".ALARMS_UNIT_01.ST3_CLADDING.RHP_SEOC_ALARMS AND NOT "DB440_MACHINE_ALARM_DECODING".ALARMS_UNIT_01.ST3_CLADDING.RHP_WARNING)) AND "DB4000_FIX_TABLE_POSITIONS".UNIT_01.FIXTURE_2.IN_CLADDING_STATION_3 AND "DB2441_MACHINE_STATUS".U01_IN_CLADDING) THEN
       "DB8000_PART_STATUS".UNIT_01.FIXTURE_2.PART_A.STATUS.PART_REJECTED := TRUE;
       "DB8000_PART_STATUS".UNIT_01.FIXTURE_2.PART_A.STATUS.OK := FALSE;
   END_IF;
END_REGION

REGION Network 6: UNIT 01 FIXTURE 3 PART A PART REJECTED
   RUNG wire#powerrail
      I_Contact( "DB2100_GENERAL".EMERGENCY_STOP_ACTIVE )
      wire#w1
      I_Contact( "DB2700_UNIT_01_FIXTURE_3".FIXTURE_NOT_CLAMPED_ALARM )
      Not()
      P_Trig( "DB8000_PART_STATUS".PULSE_3 )
      wire#w2
      S_Coil( "DB8000_PART_STATUS".UNIT_01.FIXTURE_3.PART_A.STATUS.PART_REJECTED )
      R_Coil( "DB8000_PART_STATUS".UNIT_01.FIXTURE_3.PART_A.STATUS.OK )
   END_RUNG
   RUNG wire#powerrail
      I_Contact( "DB341_M_UNIT_01_STA_0".M_CODES_UNIT_01_STA_0.M607 )
      I_Contact( "DB347_M_UNIT_01_STA_3".M_CODES_UNIT_01_STA_3.M607 )
      I_Contact( "DB353_M_UNIT_01_STA_4".M_CODES_UNIT_01_STA_4.M607 )
   END_RUNG wire#w1
   RUNG wire#powerrail
      Contact( "DB2700_UNIT_01_FIXTURE_3".CLAMPED_WITH_PART_ANALOG )
      N_Trig( "DB8000_PART_STATUS".PULSE_11 )
      I_Contact( "DB4000_FIX_TABLE_POSITIONS".UNIT_01.FIXTURE_3.IN_LOAD_UNLOAD_STATION_1 )
      Contact( "DB8000_PART_STATUS".UNIT_01.FIXTURE_3.PART_A.STATUS.PRESENT )
   END_RUNG wire#w2
   RUNG wire#powerrail
      I_Contact( "DB440_MACHINE_ALARM_DECODING".ALARMS_CENTRAL.IS_ALARMS )
      I_Contact( "DB440_MACHINE_ALARM_DECODING".ALARMS_CENTRAL.IS_SEOC_ALARMS )
      I_Contact( "DB440_MACHINE_ALARM_DECODING".ALARMS_CENTRAL.IS_WARNING )
      Not()
      wire#w3
      Contact( "DB4000_FIX_TABLE_POSITIONS".UNIT_01.FIXTURE_3.IN_CLADDING_STATION_3 )
      Contact( "DB2441_MACHINE_STATUS".U01_IN_CLADDING )
   END_RUNG wire#w2
   RUNG wire#powerrail
      I_Contact( "DB440_MACHINE_ALARM_DECODING".ALARMS_UNIT_01.ST3_CLADDING.IS_ALARMS )
      I_Contact( "DB440_MACHINE_ALARM_DECODING".ALARMS_UNIT_01.ST3_CLADDING.IS_SEOC_ALARMS )
      I_Contact( "DB440_MACHINE_ALARM_DECODING".ALARMS_UNIT_01.ST3_CLADDING.IS_WARNING )
      I_Contact( "DB440_MACHINE_ALARM_DECODING".ALARMS_UNIT_01.ST3_CLADDING.RHP_ALARMS )
      I_Contact( "DB440_MACHINE_ALARM_DECODING".ALARMS_UNIT_01.ST3_CLADDING.RHP_SEOC_ALARMS )
      I_Contact( "DB440_MACHINE_ALARM_DECODING".ALARMS_UNIT_01.ST3_CLADDING.RHP_WARNING )
      Not()
   END_RUNG wire#w3
   // the same network as SCL:
   #_w1 := NOT ((NOT "DB2100_GENERAL".EMERGENCY_STOP_ACTIVE OR (NOT "DB341_M_UNIT_01_STA_0".M_CODES_UNIT_01_STA_0.M607 AND NOT "DB347_M_UNIT_01_STA_3".M_CODES_UNIT_01_STA_3.M607 AND NOT "DB353_M_UNIT_01_STA_4".M_CODES_UNIT_01_STA_4.M607)) AND NOT "DB2700_UNIT_01_FIXTURE_3".FIXTURE_NOT_CLAMPED_ALARM);
   #_w2 := #_w1 AND NOT "DB8000_PART_STATUS".PULSE_3;   // rising edge
   "DB8000_PART_STATUS".PULSE_3 := #_w1;
   #_w3 := NOT "DB2700_UNIT_01_FIXTURE_3".CLAMPED_WITH_PART_ANALOG AND "DB8000_PART_STATUS".PULSE_11;   // falling edge
   "DB8000_PART_STATUS".PULSE_11 := "DB2700_UNIT_01_FIXTURE_3".CLAMPED_WITH_PART_ANALOG;
   IF #_w2 OR (#_w3 AND NOT "DB4000_FIX_TABLE_POSITIONS".UNIT_01.FIXTURE_3.IN_LOAD_UNLOAD_STATION_1 AND "DB8000_PART_STATUS".UNIT_01.FIXTURE_3.PART_A.STATUS.PRESENT) OR ((NOT (NOT "DB440_MACHINE_ALARM_DECODING".ALARMS_CENTRAL.IS_ALARMS AND NOT "DB440_MACHINE_ALARM_DECODING".ALARMS_CENTRAL.IS_SEOC_ALARMS AND NOT "DB440_MACHINE_ALARM_DECODING".ALARMS_CENTRAL.IS_WARNING) OR NOT (NOT "DB440_MACHINE_ALARM_DECODING".ALARMS_UNIT_01.ST3_CLADDING.IS_ALARMS AND NOT "DB440_MACHINE_ALARM_DECODING".ALARMS_UNIT_01.ST3_CLADDING.IS_SEOC_ALARMS AND NOT "DB440_MACHINE_ALARM_DECODING".ALARMS_UNIT_01.ST3_CLADDING.IS_WARNING AND NOT "DB440_MACHINE_ALARM_DECODING".ALARMS_UNIT_01.ST3_CLADDING.RHP_ALARMS AND NOT "DB440_MACHINE_ALARM_DECODING".ALARMS_UNIT_01.ST3_CLADDING.RHP_SEOC_ALARMS AND NOT "DB440_MACHINE_ALARM_DECODING".ALARMS_UNIT_01.ST3_CLADDING.RHP_WARNING)) AND "DB4000_FIX_TABLE_POSITIONS".UNIT_01.FIXTURE_3.IN_CLADDING_STATION_3 AND "DB2441_MACHINE_STATUS".U01_IN_CLADDING) THEN
       "DB8000_PART_STATUS".UNIT_01.FIXTURE_3.PART_A.STATUS.PART_REJECTED := TRUE;
       "DB8000_PART_STATUS".UNIT_01.FIXTURE_3.PART_A.STATUS.OK := FALSE;
   END_IF;
END_REGION

REGION Network 7: UNIT 01 FIXTURE 4 PART A PART REJECTED
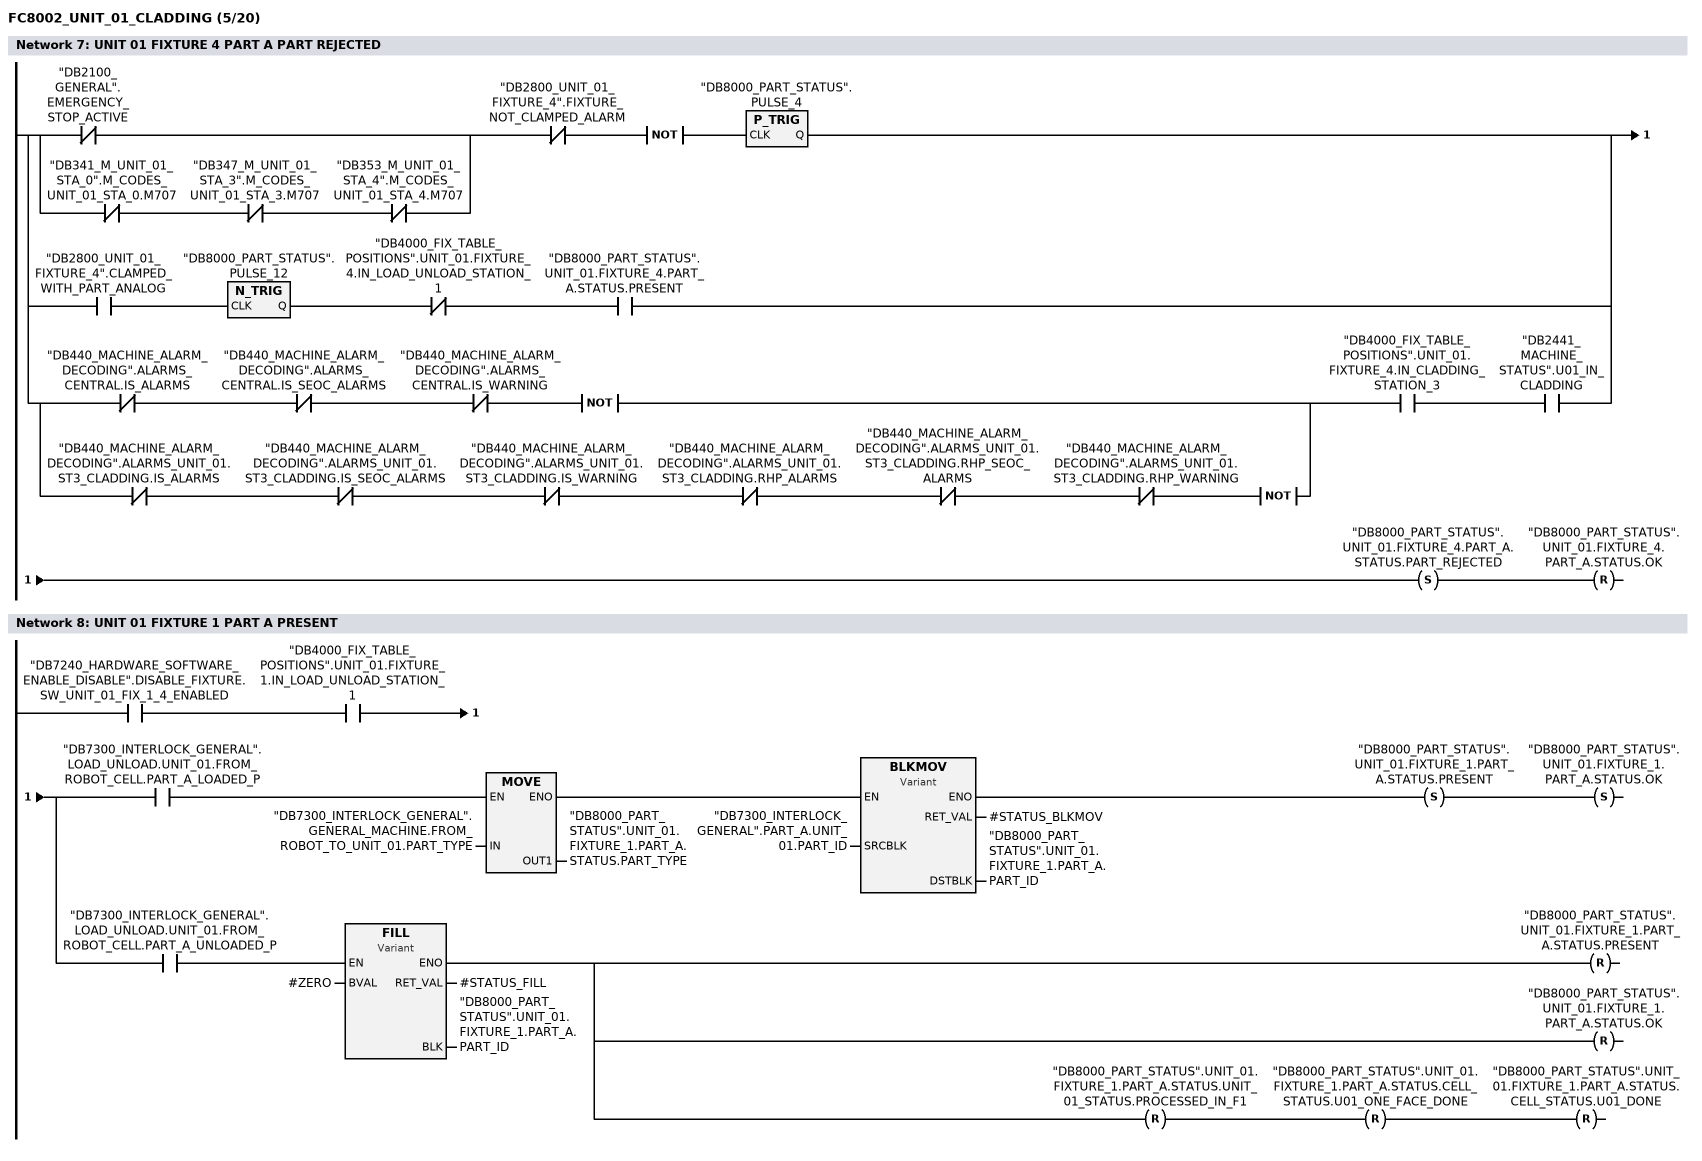
   RUNG wire#powerrail
      I_Contact( "DB2100_GENERAL".EMERGENCY_STOP_ACTIVE )
      wire#w1
      I_Contact( "DB2800_UNIT_01_FIXTURE_4".FIXTURE_NOT_CLAMPED_ALARM )
      Not()
      P_Trig( "DB8000_PART_STATUS".PULSE_4 )
      wire#w2
      S_Coil( "DB8000_PART_STATUS".UNIT_01.FIXTURE_4.PART_A.STATUS.PART_REJECTED )
      R_Coil( "DB8000_PART_STATUS".UNIT_01.FIXTURE_4.PART_A.STATUS.OK )
   END_RUNG
   RUNG wire#powerrail
      I_Contact( "DB341_M_UNIT_01_STA_0".M_CODES_UNIT_01_STA_0.M707 )
      I_Contact( "DB347_M_UNIT_01_STA_3".M_CODES_UNIT_01_STA_3.M707 )
      I_Contact( "DB353_M_UNIT_01_STA_4".M_CODES_UNIT_01_STA_4.M707 )
   END_RUNG wire#w1
   RUNG wire#powerrail
      Contact( "DB2800_UNIT_01_FIXTURE_4".CLAMPED_WITH_PART_ANALOG )
      N_Trig( "DB8000_PART_STATUS".PULSE_12 )
      I_Contact( "DB4000_FIX_TABLE_POSITIONS".UNIT_01.FIXTURE_4.IN_LOAD_UNLOAD_STATION_1 )
      Contact( "DB8000_PART_STATUS".UNIT_01.FIXTURE_4.PART_A.STATUS.PRESENT )
   END_RUNG wire#w2
   RUNG wire#powerrail
      I_Contact( "DB440_MACHINE_ALARM_DECODING".ALARMS_CENTRAL.IS_ALARMS )
      I_Contact( "DB440_MACHINE_ALARM_DECODING".ALARMS_CENTRAL.IS_SEOC_ALARMS )
      I_Contact( "DB440_MACHINE_ALARM_DECODING".ALARMS_CENTRAL.IS_WARNING )
      Not()
      wire#w3
      Contact( "DB4000_FIX_TABLE_POSITIONS".UNIT_01.FIXTURE_4.IN_CLADDING_STATION_3 )
      Contact( "DB2441_MACHINE_STATUS".U01_IN_CLADDING )
   END_RUNG wire#w2
   RUNG wire#powerrail
      I_Contact( "DB440_MACHINE_ALARM_DECODING".ALARMS_UNIT_01.ST3_CLADDING.IS_ALARMS )
      I_Contact( "DB440_MACHINE_ALARM_DECODING".ALARMS_UNIT_01.ST3_CLADDING.IS_SEOC_ALARMS )
      I_Contact( "DB440_MACHINE_ALARM_DECODING".ALARMS_UNIT_01.ST3_CLADDING.IS_WARNING )
      I_Contact( "DB440_MACHINE_ALARM_DECODING".ALARMS_UNIT_01.ST3_CLADDING.RHP_ALARMS )
      I_Contact( "DB440_MACHINE_ALARM_DECODING".ALARMS_UNIT_01.ST3_CLADDING.RHP_SEOC_ALARMS )
      I_Contact( "DB440_MACHINE_ALARM_DECODING".ALARMS_UNIT_01.ST3_CLADDING.RHP_WARNING )
      Not()
   END_RUNG wire#w3
   // the same network as SCL:
   #_w1 := NOT ((NOT "DB2100_GENERAL".EMERGENCY_STOP_ACTIVE OR (NOT "DB341_M_UNIT_01_STA_0".M_CODES_UNIT_01_STA_0.M707 AND NOT "DB347_M_UNIT_01_STA_3".M_CODES_UNIT_01_STA_3.M707 AND NOT "DB353_M_UNIT_01_STA_4".M_CODES_UNIT_01_STA_4.M707)) AND NOT "DB2800_UNIT_01_FIXTURE_4".FIXTURE_NOT_CLAMPED_ALARM);
   #_w2 := #_w1 AND NOT "DB8000_PART_STATUS".PULSE_4;   // rising edge
   "DB8000_PART_STATUS".PULSE_4 := #_w1;
   #_w3 := NOT "DB2800_UNIT_01_FIXTURE_4".CLAMPED_WITH_PART_ANALOG AND "DB8000_PART_STATUS".PULSE_12;   // falling edge
   "DB8000_PART_STATUS".PULSE_12 := "DB2800_UNIT_01_FIXTURE_4".CLAMPED_WITH_PART_ANALOG;
   IF #_w2 OR (#_w3 AND NOT "DB4000_FIX_TABLE_POSITIONS".UNIT_01.FIXTURE_4.IN_LOAD_UNLOAD_STATION_1 AND "DB8000_PART_STATUS".UNIT_01.FIXTURE_4.PART_A.STATUS.PRESENT) OR ((NOT (NOT "DB440_MACHINE_ALARM_DECODING".ALARMS_CENTRAL.IS_ALARMS AND NOT "DB440_MACHINE_ALARM_DECODING".ALARMS_CENTRAL.IS_SEOC_ALARMS AND NOT "DB440_MACHINE_ALARM_DECODING".ALARMS_CENTRAL.IS_WARNING) OR NOT (NOT "DB440_MACHINE_ALARM_DECODING".ALARMS_UNIT_01.ST3_CLADDING.IS_ALARMS AND NOT "DB440_MACHINE_ALARM_DECODING".ALARMS_UNIT_01.ST3_CLADDING.IS_SEOC_ALARMS AND NOT "DB440_MACHINE_ALARM_DECODING".ALARMS_UNIT_01.ST3_CLADDING.IS_WARNING AND NOT "DB440_MACHINE_ALARM_DECODING".ALARMS_UNIT_01.ST3_CLADDING.RHP_ALARMS AND NOT "DB440_MACHINE_ALARM_DECODING".ALARMS_UNIT_01.ST3_CLADDING.RHP_SEOC_ALARMS AND NOT "DB440_MACHINE_ALARM_DECODING".ALARMS_UNIT_01.ST3_CLADDING.RHP_WARNING)) AND "DB4000_FIX_TABLE_POSITIONS".UNIT_01.FIXTURE_4.IN_CLADDING_STATION_3 AND "DB2441_MACHINE_STATUS".U01_IN_CLADDING) THEN
       "DB8000_PART_STATUS".UNIT_01.FIXTURE_4.PART_A.STATUS.PART_REJECTED := TRUE;
       "DB8000_PART_STATUS".UNIT_01.FIXTURE_4.PART_A.STATUS.OK := FALSE;
   END_IF;
END_REGION

REGION Network 8: UNIT 01 FIXTURE 1 PART A PRESENT
   RUNG wire#powerrail
      Contact( "DB7240_HARDWARE_SOFTWARE_ENABLE_DISABLE".DISABLE_FIXTURE.SW_UNIT_01_FIX_1_4_ENABLED )
      Contact( "DB4000_FIX_TABLE_POSITIONS".UNIT_01.FIXTURE_1.IN_LOAD_UNLOAD_STATION_1 )
      wire#w1
      Contact( "DB7300_INTERLOCK_GENERAL".LOAD_UNLOAD.UNIT_01.FROM_ROBOT_CELL.PART_A_LOADED_P )
      { S7_GenerateENO := "TRUE" } Move(in := "DB7300_INTERLOCK_GENERAL".GENERAL_MACHINE.FROM_ROBOT_TO_UNIT_01.PART_TYPE, out1 => "DB8000_PART_STATUS".UNIT_01.FIXTURE_1.PART_A.STATUS.PART_TYPE)
      { S7_Templates := "blk_type := Variant" } BLKMOV(SRCBLK := "DB7300_INTERLOCK_GENERAL".PART_A.UNIT_01.PART_ID, RET_VAL => #STATUS_BLKMOV, DSTBLK => "DB8000_PART_STATUS".UNIT_01.FIXTURE_1.PART_A.PART_ID)
      S_Coil( "DB8000_PART_STATUS".UNIT_01.FIXTURE_1.PART_A.STATUS.PRESENT )
      S_Coil( "DB8000_PART_STATUS".UNIT_01.FIXTURE_1.PART_A.STATUS.OK )
   END_RUNG
   RUNG wire#w1
      Contact( "DB7300_INTERLOCK_GENERAL".LOAD_UNLOAD.UNIT_01.FROM_ROBOT_CELL.PART_A_UNLOADED_P )
      { S7_Templates := "ptr_type := Variant" } FILL(BVAL := #ZERO, RET_VAL => #STATUS_FILL, BLK => "DB8000_PART_STATUS".UNIT_01.FIXTURE_1.PART_A.PART_ID)
      wire#w2
      R_Coil( "DB8000_PART_STATUS".UNIT_01.FIXTURE_1.PART_A.STATUS.PRESENT )
   END_RUNG
   RUNG wire#w2
      R_Coil( "DB8000_PART_STATUS".UNIT_01.FIXTURE_1.PART_A.STATUS.OK )
   END_RUNG
   RUNG wire#w2
      R_Coil( "DB8000_PART_STATUS".UNIT_01.FIXTURE_1.PART_A.STATUS.UNIT_01_STATUS.PROCESSED_IN_F1 )
      R_Coil( "DB8000_PART_STATUS".UNIT_01.FIXTURE_1.PART_A.STATUS.CELL_STATUS.U01_ONE_FACE_DONE )
      R_Coil( "DB8000_PART_STATUS".UNIT_01.FIXTURE_1.PART_A.STATUS.CELL_STATUS.U01_DONE )
   END_RUNG
   // the same network as SCL:
   // ENO of a box is taken as its EN; it also drops when the box reports an error
   #_w1 := "DB7240_HARDWARE_SOFTWARE_ENABLE_DISABLE".DISABLE_FIXTURE.SW_UNIT_01_FIX_1_4_ENABLED AND "DB4000_FIX_TABLE_POSITIONS".UNIT_01.FIXTURE_1.IN_LOAD_UNLOAD_STATION_1;
   IF #_w1 AND "DB7300_INTERLOCK_GENERAL".LOAD_UNLOAD.UNIT_01.FROM_ROBOT_CELL.PART_A_LOADED_P THEN
       "DB8000_PART_STATUS".UNIT_01.FIXTURE_1.PART_A.STATUS.PART_TYPE := "DB7300_INTERLOCK_GENERAL".GENERAL_MACHINE.FROM_ROBOT_TO_UNIT_01.PART_TYPE;
   END_IF;
   #STATUS_BLKMOV := BLKMOV(EN := #_w1 AND "DB7300_INTERLOCK_GENERAL".LOAD_UNLOAD.UNIT_01.FROM_ROBOT_CELL.PART_A_LOADED_P,
                           SRCBLK := "DB7300_INTERLOCK_GENERAL".PART_A.UNIT_01.PART_ID,
                           DSTBLK => "DB8000_PART_STATUS".UNIT_01.FIXTURE_1.PART_A.PART_ID,
                           ENO => #_w2);
   IF #_w2 THEN
       "DB8000_PART_STATUS".UNIT_01.FIXTURE_1.PART_A.STATUS.PRESENT := TRUE;
       "DB8000_PART_STATUS".UNIT_01.FIXTURE_1.PART_A.STATUS.OK := TRUE;
   END_IF;
   #STATUS_FILL := FILL(EN := #_w1 AND "DB7300_INTERLOCK_GENERAL".LOAD_UNLOAD.UNIT_01.FROM_ROBOT_CELL.PART_A_UNLOADED_P,
                        BVAL := #ZERO,
                        BLK => "DB8000_PART_STATUS".UNIT_01.FIXTURE_1.PART_A.PART_ID,
                        ENO => #_w3);
   IF #_w3 THEN
       "DB8000_PART_STATUS".UNIT_01.FIXTURE_1.PART_A.STATUS.PRESENT := FALSE;
       "DB8000_PART_STATUS".UNIT_01.FIXTURE_1.PART_A.STATUS.OK := FALSE;
       "DB8000_PART_STATUS".UNIT_01.FIXTURE_1.PART_A.STATUS.UNIT_01_STATUS.PROCESSED_IN_F1 := FALSE;
       "DB8000_PART_STATUS".UNIT_01.FIXTURE_1.PART_A.STATUS.CELL_STATUS.U01_ONE_FACE_DONE := FALSE;
       "DB8000_PART_STATUS".UNIT_01.FIXTURE_1.PART_A.STATUS.CELL_STATUS.U01_DONE := FALSE;
   END_IF;
END_REGION

REGION Network 9: UNIT 01 FIXTURE 2 PART A PRESENT
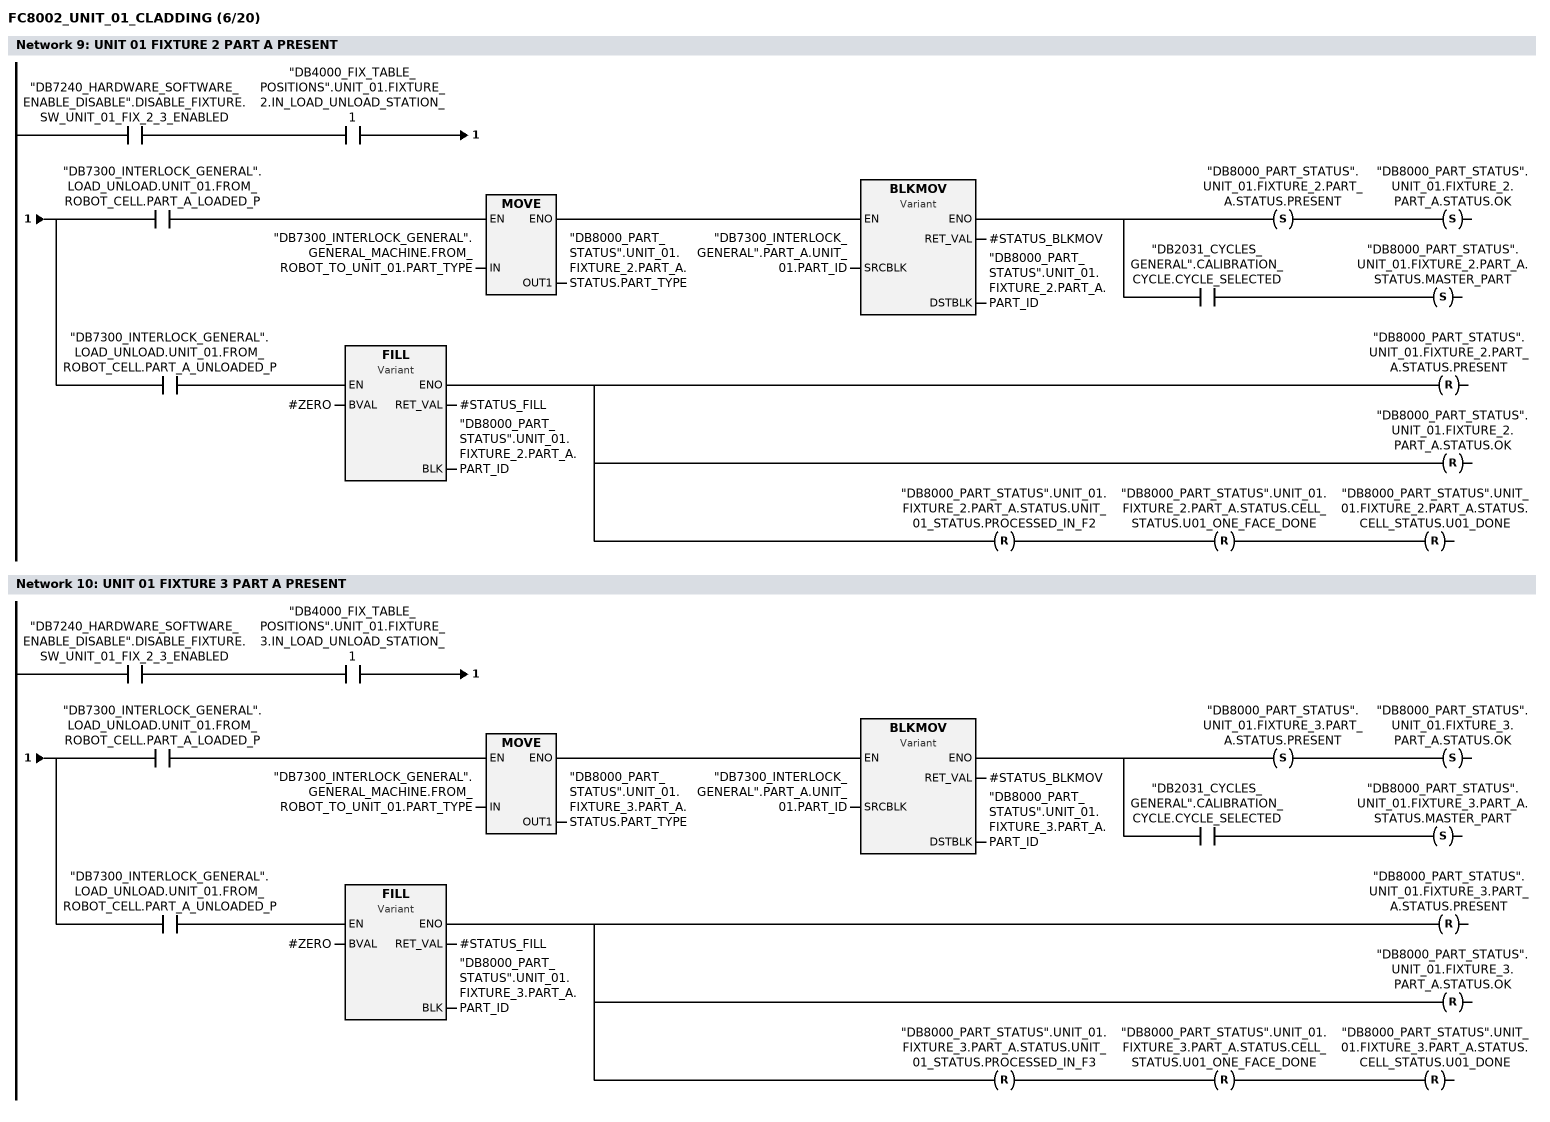
   RUNG wire#powerrail
      Contact( "DB7240_HARDWARE_SOFTWARE_ENABLE_DISABLE".DISABLE_FIXTURE.SW_UNIT_01_FIX_2_3_ENABLED )
      Contact( "DB4000_FIX_TABLE_POSITIONS".UNIT_01.FIXTURE_2.IN_LOAD_UNLOAD_STATION_1 )
      wire#w1
      Contact( "DB7300_INTERLOCK_GENERAL".LOAD_UNLOAD.UNIT_01.FROM_ROBOT_CELL.PART_A_LOADED_P )
      { S7_GenerateENO := "TRUE" } Move(in := "DB7300_INTERLOCK_GENERAL".GENERAL_MACHINE.FROM_ROBOT_TO_UNIT_01.PART_TYPE, out1 => "DB8000_PART_STATUS".UNIT_01.FIXTURE_2.PART_A.STATUS.PART_TYPE)
      { S7_Templates := "blk_type := Variant" } BLKMOV(SRCBLK := "DB7300_INTERLOCK_GENERAL".PART_A.UNIT_01.PART_ID, RET_VAL => #STATUS_BLKMOV, DSTBLK => "DB8000_PART_STATUS".UNIT_01.FIXTURE_2.PART_A.PART_ID)
      wire#w2
      S_Coil( "DB8000_PART_STATUS".UNIT_01.FIXTURE_2.PART_A.STATUS.PRESENT )
      S_Coil( "DB8000_PART_STATUS".UNIT_01.FIXTURE_2.PART_A.STATUS.OK )
   END_RUNG
   RUNG wire#w2
      Contact( "DB2031_CYCLES_GENERAL".CALIBRATION_CYCLE.CYCLE_SELECTED )
      S_Coil( "DB8000_PART_STATUS".UNIT_01.FIXTURE_2.PART_A.STATUS.MASTER_PART )
   END_RUNG
   RUNG wire#w1
      Contact( "DB7300_INTERLOCK_GENERAL".LOAD_UNLOAD.UNIT_01.FROM_ROBOT_CELL.PART_A_UNLOADED_P )
      { S7_Templates := "ptr_type := Variant" } FILL(BVAL := #ZERO, RET_VAL => #STATUS_FILL, BLK => "DB8000_PART_STATUS".UNIT_01.FIXTURE_2.PART_A.PART_ID)
      wire#w3
      R_Coil( "DB8000_PART_STATUS".UNIT_01.FIXTURE_2.PART_A.STATUS.PRESENT )
   END_RUNG
   RUNG wire#w3
      R_Coil( "DB8000_PART_STATUS".UNIT_01.FIXTURE_2.PART_A.STATUS.OK )
   END_RUNG
   RUNG wire#w3
      R_Coil( "DB8000_PART_STATUS".UNIT_01.FIXTURE_2.PART_A.STATUS.UNIT_01_STATUS.PROCESSED_IN_F2 )
      R_Coil( "DB8000_PART_STATUS".UNIT_01.FIXTURE_2.PART_A.STATUS.CELL_STATUS.U01_ONE_FACE_DONE )
      R_Coil( "DB8000_PART_STATUS".UNIT_01.FIXTURE_2.PART_A.STATUS.CELL_STATUS.U01_DONE )
   END_RUNG
   // the same network as SCL:
   // ENO of a box is taken as its EN; it also drops when the box reports an error
   #_w1 := "DB7240_HARDWARE_SOFTWARE_ENABLE_DISABLE".DISABLE_FIXTURE.SW_UNIT_01_FIX_2_3_ENABLED AND "DB4000_FIX_TABLE_POSITIONS".UNIT_01.FIXTURE_2.IN_LOAD_UNLOAD_STATION_1;
   #_w2 := #_w1 AND "DB7300_INTERLOCK_GENERAL".LOAD_UNLOAD.UNIT_01.FROM_ROBOT_CELL.PART_A_LOADED_P;
   IF #_w2 THEN
       "DB8000_PART_STATUS".UNIT_01.FIXTURE_2.PART_A.STATUS.PART_TYPE := "DB7300_INTERLOCK_GENERAL".GENERAL_MACHINE.FROM_ROBOT_TO_UNIT_01.PART_TYPE;
   END_IF;
   #STATUS_BLKMOV := BLKMOV(EN := #_w2,
                           SRCBLK := "DB7300_INTERLOCK_GENERAL".PART_A.UNIT_01.PART_ID,
                           DSTBLK => "DB8000_PART_STATUS".UNIT_01.FIXTURE_2.PART_A.PART_ID,
                           ENO => #_w3);
   IF #_w3 THEN
       "DB8000_PART_STATUS".UNIT_01.FIXTURE_2.PART_A.STATUS.PRESENT := TRUE;
       "DB8000_PART_STATUS".UNIT_01.FIXTURE_2.PART_A.STATUS.OK := TRUE;
   END_IF;
   IF #_w3 AND "DB2031_CYCLES_GENERAL".CALIBRATION_CYCLE.CYCLE_SELECTED THEN
       "DB8000_PART_STATUS".UNIT_01.FIXTURE_2.PART_A.STATUS.MASTER_PART := TRUE;
   END_IF;
   #STATUS_FILL := FILL(EN := #_w1 AND "DB7300_INTERLOCK_GENERAL".LOAD_UNLOAD.UNIT_01.FROM_ROBOT_CELL.PART_A_UNLOADED_P,
                        BVAL := #ZERO,
                        BLK => "DB8000_PART_STATUS".UNIT_01.FIXTURE_2.PART_A.PART_ID,
                        ENO => #_w4);
   IF #_w4 THEN
       "DB8000_PART_STATUS".UNIT_01.FIXTURE_2.PART_A.STATUS.PRESENT := FALSE;
       "DB8000_PART_STATUS".UNIT_01.FIXTURE_2.PART_A.STATUS.OK := FALSE;
       "DB8000_PART_STATUS".UNIT_01.FIXTURE_2.PART_A.STATUS.UNIT_01_STATUS.PROCESSED_IN_F2 := FALSE;
       "DB8000_PART_STATUS".UNIT_01.FIXTURE_2.PART_A.STATUS.CELL_STATUS.U01_ONE_FACE_DONE := FALSE;
       "DB8000_PART_STATUS".UNIT_01.FIXTURE_2.PART_A.STATUS.CELL_STATUS.U01_DONE := FALSE;
   END_IF;
END_REGION

REGION Network 10: UNIT 01 FIXTURE 3 PART A PRESENT
   RUNG wire#powerrail
      Contact( "DB7240_HARDWARE_SOFTWARE_ENABLE_DISABLE".DISABLE_FIXTURE.SW_UNIT_01_FIX_2_3_ENABLED )
      Contact( "DB4000_FIX_TABLE_POSITIONS".UNIT_01.FIXTURE_3.IN_LOAD_UNLOAD_STATION_1 )
      wire#w1
      Contact( "DB7300_INTERLOCK_GENERAL".LOAD_UNLOAD.UNIT_01.FROM_ROBOT_CELL.PART_A_LOADED_P )
      { S7_GenerateENO := "TRUE" } Move(in := "DB7300_INTERLOCK_GENERAL".GENERAL_MACHINE.FROM_ROBOT_TO_UNIT_01.PART_TYPE, out1 => "DB8000_PART_STATUS".UNIT_01.FIXTURE_3.PART_A.STATUS.PART_TYPE)
      { S7_Templates := "blk_type := Variant" } BLKMOV(SRCBLK := "DB7300_INTERLOCK_GENERAL".PART_A.UNIT_01.PART_ID, RET_VAL => #STATUS_BLKMOV, DSTBLK => "DB8000_PART_STATUS".UNIT_01.FIXTURE_3.PART_A.PART_ID)
      wire#w2
      S_Coil( "DB8000_PART_STATUS".UNIT_01.FIXTURE_3.PART_A.STATUS.PRESENT )
      S_Coil( "DB8000_PART_STATUS".UNIT_01.FIXTURE_3.PART_A.STATUS.OK )
   END_RUNG
   RUNG wire#w2
      Contact( "DB2031_CYCLES_GENERAL".CALIBRATION_CYCLE.CYCLE_SELECTED )
      S_Coil( "DB8000_PART_STATUS".UNIT_01.FIXTURE_3.PART_A.STATUS.MASTER_PART )
   END_RUNG
   RUNG wire#w1
      Contact( "DB7300_INTERLOCK_GENERAL".LOAD_UNLOAD.UNIT_01.FROM_ROBOT_CELL.PART_A_UNLOADED_P )
      { S7_Templates := "ptr_type := Variant" } FILL(BVAL := #ZERO, RET_VAL => #STATUS_FILL, BLK => "DB8000_PART_STATUS".UNIT_01.FIXTURE_3.PART_A.PART_ID)
      wire#w3
      R_Coil( "DB8000_PART_STATUS".UNIT_01.FIXTURE_3.PART_A.STATUS.PRESENT )
   END_RUNG
   RUNG wire#w3
      R_Coil( "DB8000_PART_STATUS".UNIT_01.FIXTURE_3.PART_A.STATUS.OK )
   END_RUNG
   RUNG wire#w3
      R_Coil( "DB8000_PART_STATUS".UNIT_01.FIXTURE_3.PART_A.STATUS.UNIT_01_STATUS.PROCESSED_IN_F3 )
      R_Coil( "DB8000_PART_STATUS".UNIT_01.FIXTURE_3.PART_A.STATUS.CELL_STATUS.U01_ONE_FACE_DONE )
      R_Coil( "DB8000_PART_STATUS".UNIT_01.FIXTURE_3.PART_A.STATUS.CELL_STATUS.U01_DONE )
   END_RUNG
   // the same network as SCL:
   // ENO of a box is taken as its EN; it also drops when the box reports an error
   #_w1 := "DB7240_HARDWARE_SOFTWARE_ENABLE_DISABLE".DISABLE_FIXTURE.SW_UNIT_01_FIX_2_3_ENABLED AND "DB4000_FIX_TABLE_POSITIONS".UNIT_01.FIXTURE_3.IN_LOAD_UNLOAD_STATION_1;
   #_w2 := #_w1 AND "DB7300_INTERLOCK_GENERAL".LOAD_UNLOAD.UNIT_01.FROM_ROBOT_CELL.PART_A_LOADED_P;
   IF #_w2 THEN
       "DB8000_PART_STATUS".UNIT_01.FIXTURE_3.PART_A.STATUS.PART_TYPE := "DB7300_INTERLOCK_GENERAL".GENERAL_MACHINE.FROM_ROBOT_TO_UNIT_01.PART_TYPE;
   END_IF;
   #STATUS_BLKMOV := BLKMOV(EN := #_w2,
                           SRCBLK := "DB7300_INTERLOCK_GENERAL".PART_A.UNIT_01.PART_ID,
                           DSTBLK => "DB8000_PART_STATUS".UNIT_01.FIXTURE_3.PART_A.PART_ID,
                           ENO => #_w3);
   IF #_w3 THEN
       "DB8000_PART_STATUS".UNIT_01.FIXTURE_3.PART_A.STATUS.PRESENT := TRUE;
       "DB8000_PART_STATUS".UNIT_01.FIXTURE_3.PART_A.STATUS.OK := TRUE;
   END_IF;
   IF #_w3 AND "DB2031_CYCLES_GENERAL".CALIBRATION_CYCLE.CYCLE_SELECTED THEN
       "DB8000_PART_STATUS".UNIT_01.FIXTURE_3.PART_A.STATUS.MASTER_PART := TRUE;
   END_IF;
   #STATUS_FILL := FILL(EN := #_w1 AND "DB7300_INTERLOCK_GENERAL".LOAD_UNLOAD.UNIT_01.FROM_ROBOT_CELL.PART_A_UNLOADED_P,
                        BVAL := #ZERO,
                        BLK => "DB8000_PART_STATUS".UNIT_01.FIXTURE_3.PART_A.PART_ID,
                        ENO => #_w4);
   IF #_w4 THEN
       "DB8000_PART_STATUS".UNIT_01.FIXTURE_3.PART_A.STATUS.PRESENT := FALSE;
       "DB8000_PART_STATUS".UNIT_01.FIXTURE_3.PART_A.STATUS.OK := FALSE;
       "DB8000_PART_STATUS".UNIT_01.FIXTURE_3.PART_A.STATUS.UNIT_01_STATUS.PROCESSED_IN_F3 := FALSE;
       "DB8000_PART_STATUS".UNIT_01.FIXTURE_3.PART_A.STATUS.CELL_STATUS.U01_ONE_FACE_DONE := FALSE;
       "DB8000_PART_STATUS".UNIT_01.FIXTURE_3.PART_A.STATUS.CELL_STATUS.U01_DONE := FALSE;
   END_IF;
END_REGION

REGION Network 11: UNIT 01 FIXTURE 4 PART A PRESENT
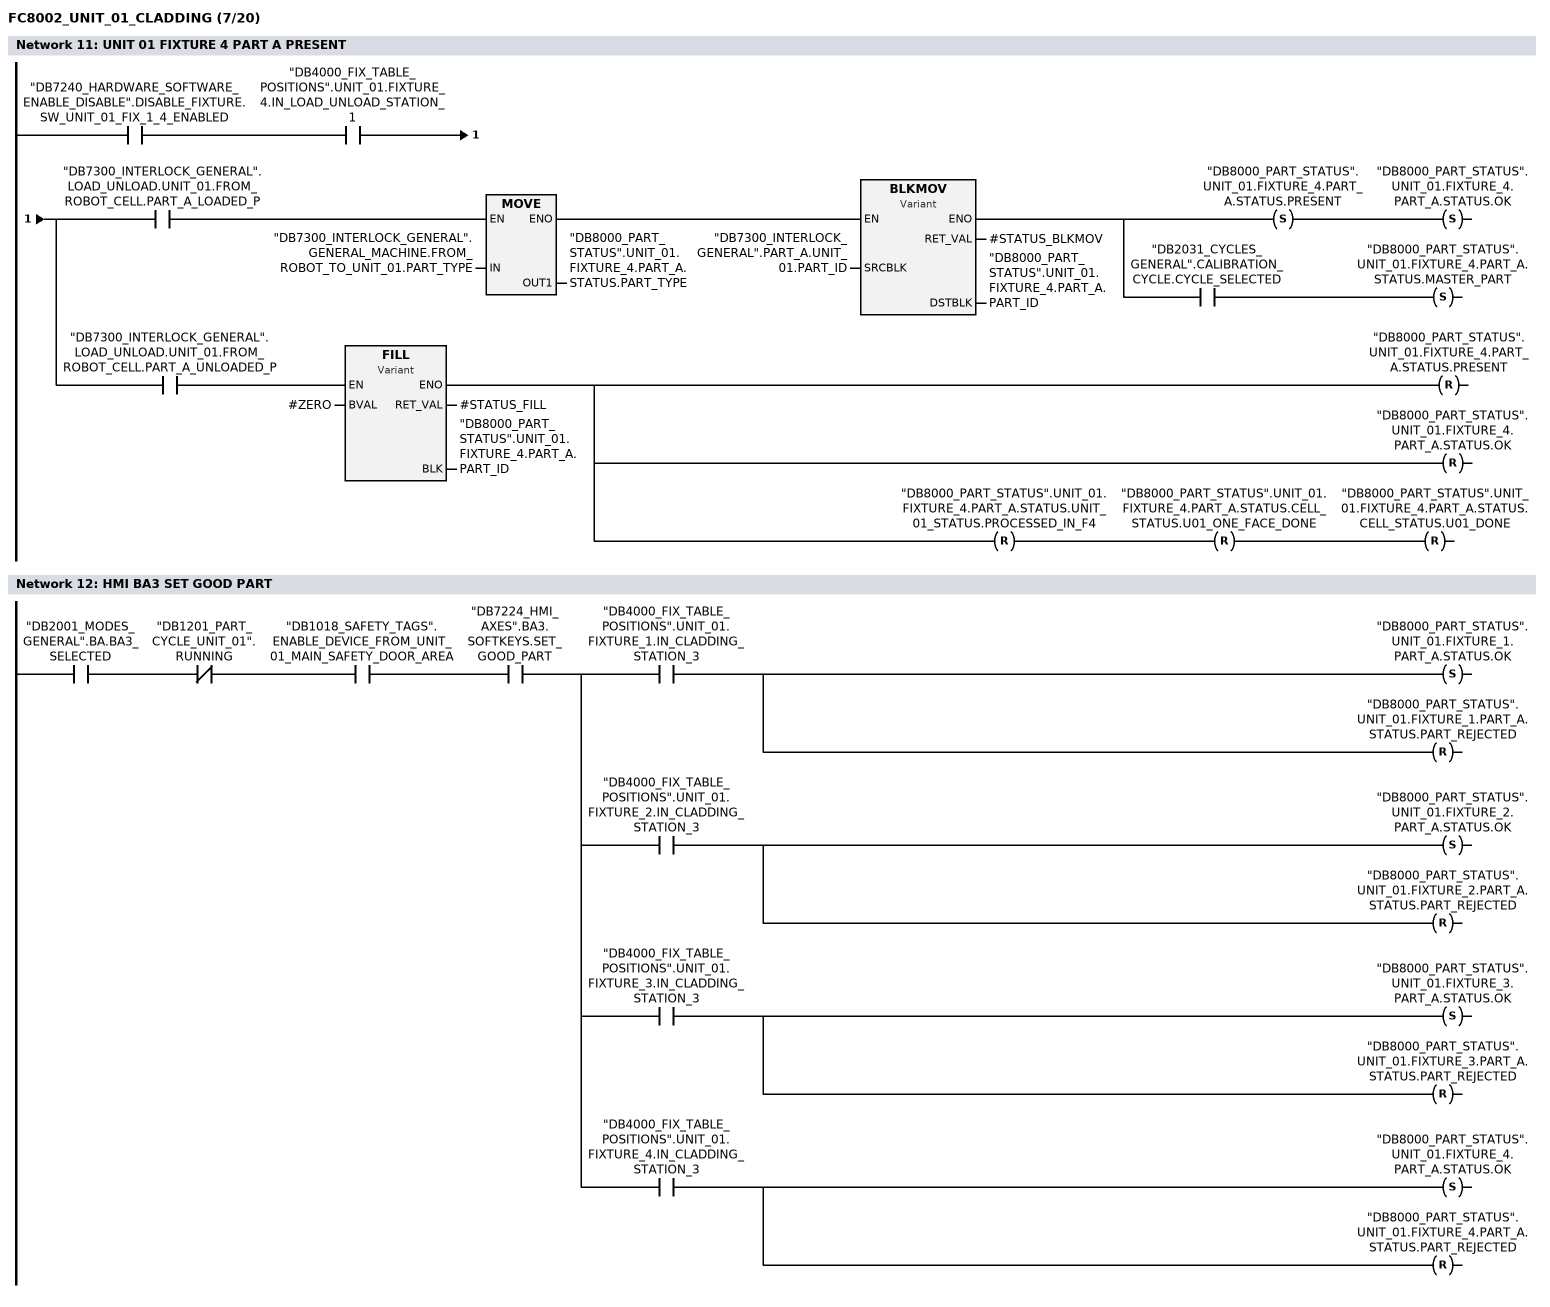
   RUNG wire#powerrail
      Contact( "DB7240_HARDWARE_SOFTWARE_ENABLE_DISABLE".DISABLE_FIXTURE.SW_UNIT_01_FIX_1_4_ENABLED )
      Contact( "DB4000_FIX_TABLE_POSITIONS".UNIT_01.FIXTURE_4.IN_LOAD_UNLOAD_STATION_1 )
      wire#w1
      Contact( "DB7300_INTERLOCK_GENERAL".LOAD_UNLOAD.UNIT_01.FROM_ROBOT_CELL.PART_A_LOADED_P )
      { S7_GenerateENO := "TRUE" } Move(in := "DB7300_INTERLOCK_GENERAL".GENERAL_MACHINE.FROM_ROBOT_TO_UNIT_01.PART_TYPE, out1 => "DB8000_PART_STATUS".UNIT_01.FIXTURE_4.PART_A.STATUS.PART_TYPE)
      { S7_Templates := "blk_type := Variant" } BLKMOV(SRCBLK := "DB7300_INTERLOCK_GENERAL".PART_A.UNIT_01.PART_ID, RET_VAL => #STATUS_BLKMOV, DSTBLK => "DB8000_PART_STATUS".UNIT_01.FIXTURE_4.PART_A.PART_ID)
      wire#w2
      S_Coil( "DB8000_PART_STATUS".UNIT_01.FIXTURE_4.PART_A.STATUS.PRESENT )
      S_Coil( "DB8000_PART_STATUS".UNIT_01.FIXTURE_4.PART_A.STATUS.OK )
   END_RUNG
   RUNG wire#w2
      Contact( "DB2031_CYCLES_GENERAL".CALIBRATION_CYCLE.CYCLE_SELECTED )
      S_Coil( "DB8000_PART_STATUS".UNIT_01.FIXTURE_4.PART_A.STATUS.MASTER_PART )
   END_RUNG
   RUNG wire#w1
      Contact( "DB7300_INTERLOCK_GENERAL".LOAD_UNLOAD.UNIT_01.FROM_ROBOT_CELL.PART_A_UNLOADED_P )
      { S7_Templates := "ptr_type := Variant" } FILL(BVAL := #ZERO, RET_VAL => #STATUS_FILL, BLK => "DB8000_PART_STATUS".UNIT_01.FIXTURE_4.PART_A.PART_ID)
      wire#w3
      R_Coil( "DB8000_PART_STATUS".UNIT_01.FIXTURE_4.PART_A.STATUS.PRESENT )
   END_RUNG
   RUNG wire#w3
      R_Coil( "DB8000_PART_STATUS".UNIT_01.FIXTURE_4.PART_A.STATUS.OK )
   END_RUNG
   RUNG wire#w3
      R_Coil( "DB8000_PART_STATUS".UNIT_01.FIXTURE_4.PART_A.STATUS.UNIT_01_STATUS.PROCESSED_IN_F4 )
      R_Coil( "DB8000_PART_STATUS".UNIT_01.FIXTURE_4.PART_A.STATUS.CELL_STATUS.U01_ONE_FACE_DONE )
      R_Coil( "DB8000_PART_STATUS".UNIT_01.FIXTURE_4.PART_A.STATUS.CELL_STATUS.U01_DONE )
   END_RUNG
   // the same network as SCL:
   // ENO of a box is taken as its EN; it also drops when the box reports an error
   #_w1 := "DB7240_HARDWARE_SOFTWARE_ENABLE_DISABLE".DISABLE_FIXTURE.SW_UNIT_01_FIX_1_4_ENABLED AND "DB4000_FIX_TABLE_POSITIONS".UNIT_01.FIXTURE_4.IN_LOAD_UNLOAD_STATION_1;
   #_w2 := #_w1 AND "DB7300_INTERLOCK_GENERAL".LOAD_UNLOAD.UNIT_01.FROM_ROBOT_CELL.PART_A_LOADED_P;
   IF #_w2 THEN
       "DB8000_PART_STATUS".UNIT_01.FIXTURE_4.PART_A.STATUS.PART_TYPE := "DB7300_INTERLOCK_GENERAL".GENERAL_MACHINE.FROM_ROBOT_TO_UNIT_01.PART_TYPE;
   END_IF;
   #STATUS_BLKMOV := BLKMOV(EN := #_w2,
                           SRCBLK := "DB7300_INTERLOCK_GENERAL".PART_A.UNIT_01.PART_ID,
                           DSTBLK => "DB8000_PART_STATUS".UNIT_01.FIXTURE_4.PART_A.PART_ID,
                           ENO => #_w3);
   IF #_w3 THEN
       "DB8000_PART_STATUS".UNIT_01.FIXTURE_4.PART_A.STATUS.PRESENT := TRUE;
       "DB8000_PART_STATUS".UNIT_01.FIXTURE_4.PART_A.STATUS.OK := TRUE;
   END_IF;
   IF #_w3 AND "DB2031_CYCLES_GENERAL".CALIBRATION_CYCLE.CYCLE_SELECTED THEN
       "DB8000_PART_STATUS".UNIT_01.FIXTURE_4.PART_A.STATUS.MASTER_PART := TRUE;
   END_IF;
   #STATUS_FILL := FILL(EN := #_w1 AND "DB7300_INTERLOCK_GENERAL".LOAD_UNLOAD.UNIT_01.FROM_ROBOT_CELL.PART_A_UNLOADED_P,
                        BVAL := #ZERO,
                        BLK => "DB8000_PART_STATUS".UNIT_01.FIXTURE_4.PART_A.PART_ID,
                        ENO => #_w4);
   IF #_w4 THEN
       "DB8000_PART_STATUS".UNIT_01.FIXTURE_4.PART_A.STATUS.PRESENT := FALSE;
       "DB8000_PART_STATUS".UNIT_01.FIXTURE_4.PART_A.STATUS.OK := FALSE;
       "DB8000_PART_STATUS".UNIT_01.FIXTURE_4.PART_A.STATUS.UNIT_01_STATUS.PROCESSED_IN_F4 := FALSE;
       "DB8000_PART_STATUS".UNIT_01.FIXTURE_4.PART_A.STATUS.CELL_STATUS.U01_ONE_FACE_DONE := FALSE;
       "DB8000_PART_STATUS".UNIT_01.FIXTURE_4.PART_A.STATUS.CELL_STATUS.U01_DONE := FALSE;
   END_IF;
END_REGION

